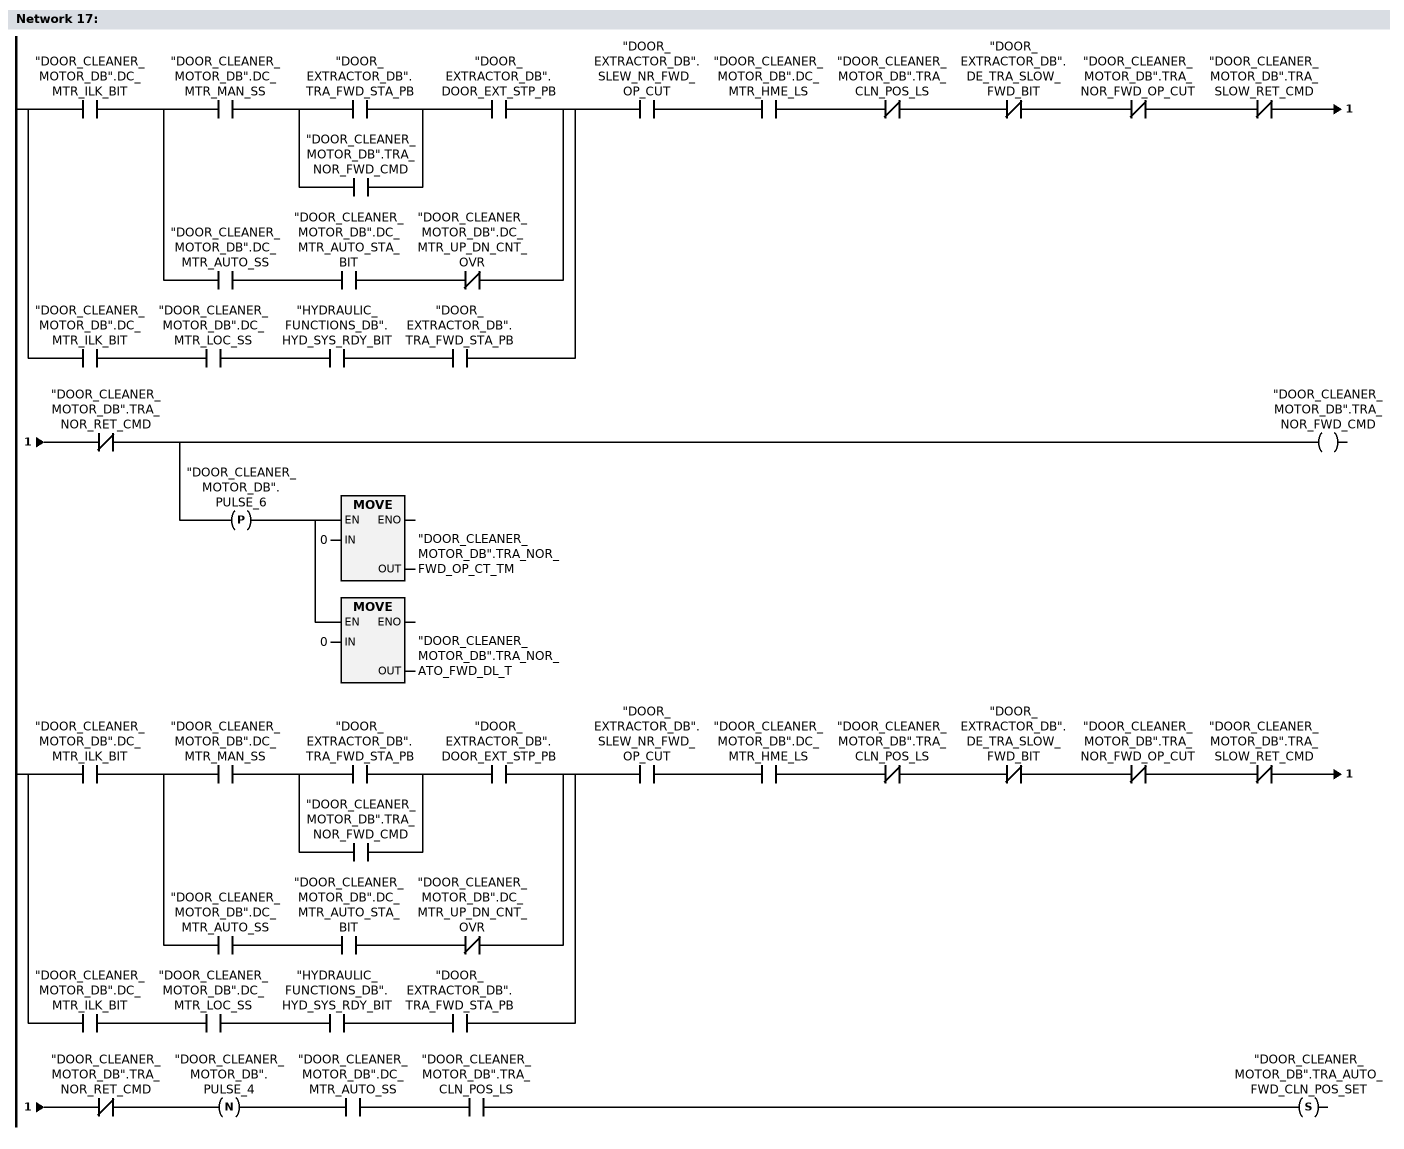
NETWORK
TITLE =
      A(;
      A     "DOOR_CLEANER_MOTOR_DB".DC_MTR_ILK_BIT;
      A(;
      A     "DOOR_CLEANER_MOTOR_DB".DC_MTR_MAN_SS;
      A(;
      O     "DOOR_EXTRACTOR_DB".TRA_FWD_STA_PB;
      O     "DOOR_CLEANER_MOTOR_DB".TRA_NOR_FWD_CMD;
      );
      A     "DOOR_EXTRACTOR_DB".DOOR_EXT_STP_PB;
      O;
      A     "DOOR_CLEANER_MOTOR_DB".DC_MTR_AUTO_SS;
      A     "DOOR_CLEANER_MOTOR_DB".DC_MTR_AUTO_STA_BIT;
      AN    "DOOR_CLEANER_MOTOR_DB".DC_MTR_UP_DN_CNT_OVR;
      );
      O;
      A     "DOOR_CLEANER_MOTOR_DB".DC_MTR_ILK_BIT;
      A     "DOOR_CLEANER_MOTOR_DB".DC_MTR_LOC_SS;
      A     "HYDRAULIC_FUNCTIONS_DB".HYD_SYS_RDY_BIT;
      A     "DOOR_EXTRACTOR_DB".TRA_FWD_STA_PB;
      );
      A     "DOOR_EXTRACTOR_DB".SLEW_NR_FWD_OP_CUT;
      A     "DOOR_CLEANER_MOTOR_DB".DC_MTR_HME_LS;
      AN    "DOOR_CLEANER_MOTOR_DB".TRA_CLN_POS_LS;
      AN    "DOOR_EXTRACTOR_DB".DE_TRA_SLOW_FWD_BIT;
      AN    "DOOR_CLEANER_MOTOR_DB".TRA_NOR_FWD_OP_CUT;
      AN    "DOOR_CLEANER_MOTOR_DB".TRA_SLOW_RET_CMD;
      AN    "DOOR_CLEANER_MOTOR_DB".TRA_NOR_RET_CMD;
      =     L 0.0;
      A     L 0.0;
      BLD   102;
      =     "DOOR_CLEANER_MOTOR_DB".TRA_NOR_FWD_CMD;
      A(;
      A     L 0.0;
      FN    "DOOR_CLEANER_MOTOR_DB".PULSE_4;
      );
      A     "DOOR_CLEANER_MOTOR_DB".DC_MTR_AUTO_SS;
      A     "DOOR_CLEANER_MOTOR_DB".TRA_CLN_POS_LS;
      S     "DOOR_CLEANER_MOTOR_DB".TRA_AUTO_FWD_CLN_POS_SET;
      A     L 0.0;
      FP    "DOOR_CLEANER_MOTOR_DB".PULSE_6;
      =     L 0.1;
      A     L 0.1;
      JNB   M012;
      L     0;
      T     "DOOR_CLEANER_MOTOR_DB".TRA_NOR_FWD_OP_CT_TM;
M012: NOP   0;
      A     L 0.1;
      JNB   M013;
      L     0;
      T     "DOOR_CLEANER_MOTOR_DB".TRA_NOR_ATO_FWD_DL_T;
M013: NOP   0;
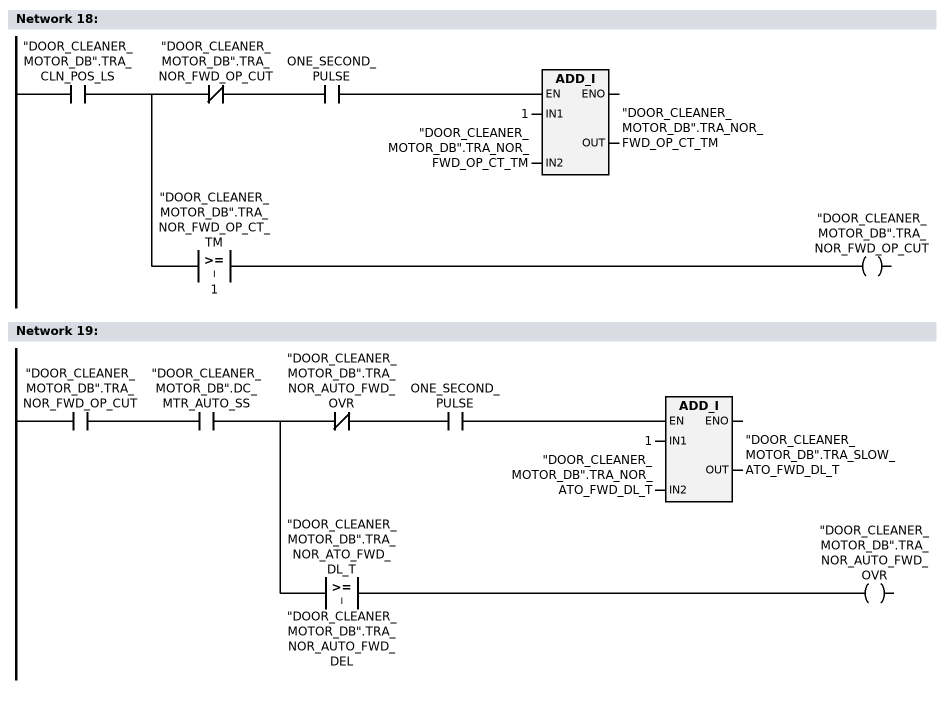
NETWORK
TITLE =
      A     "DOOR_CLEANER_MOTOR_DB".TRA_CLN_POS_LS;
      =     L 0.0;
      A     L 0.0;
      AN    "DOOR_CLEANER_MOTOR_DB".TRA_NOR_FWD_OP_CUT;
      A     "ONE_SECOND_PULSE";
      JNB   M014;
      L     1;
      L     "DOOR_CLEANER_MOTOR_DB".TRA_NOR_FWD_OP_CT_TM;
      +I;
      T     "DOOR_CLEANER_MOTOR_DB".TRA_NOR_FWD_OP_CT_TM;
M014: NOP   0;
      A     L 0.0;
      A(;
      L     "DOOR_CLEANER_MOTOR_DB".TRA_NOR_FWD_OP_CT_TM;
      L     1;
      >=I;
      );
      =     "DOOR_CLEANER_MOTOR_DB".TRA_NOR_FWD_OP_CUT;
NETWORK
TITLE =
      A     "DOOR_CLEANER_MOTOR_DB".TRA_NOR_FWD_OP_CUT;
      A     "DOOR_CLEANER_MOTOR_DB".DC_MTR_AUTO_SS;
      =     L 0.0;
      A     L 0.0;
      AN    "DOOR_CLEANER_MOTOR_DB".TRA_NOR_AUTO_FWD_OVR;
      A     "ONE_SECOND_PULSE";
      JNB   M015;
      L     1;
      L     "DOOR_CLEANER_MOTOR_DB".TRA_NOR_ATO_FWD_DL_T;
      +I;
      T     "DOOR_CLEANER_MOTOR_DB".TRA_SLOW_ATO_FWD_DL_T;
M015: NOP   0;
      A     L 0.0;
      A(;
      L     "DOOR_CLEANER_MOTOR_DB".TRA_NOR_ATO_FWD_DL_T;
      L     "DOOR_CLEANER_MOTOR_DB".TRA_NOR_AUTO_FWD_DEL;
      >=I;
      );
      =     "DOOR_CLEANER_MOTOR_DB".TRA_NOR_AUTO_FWD_OVR;
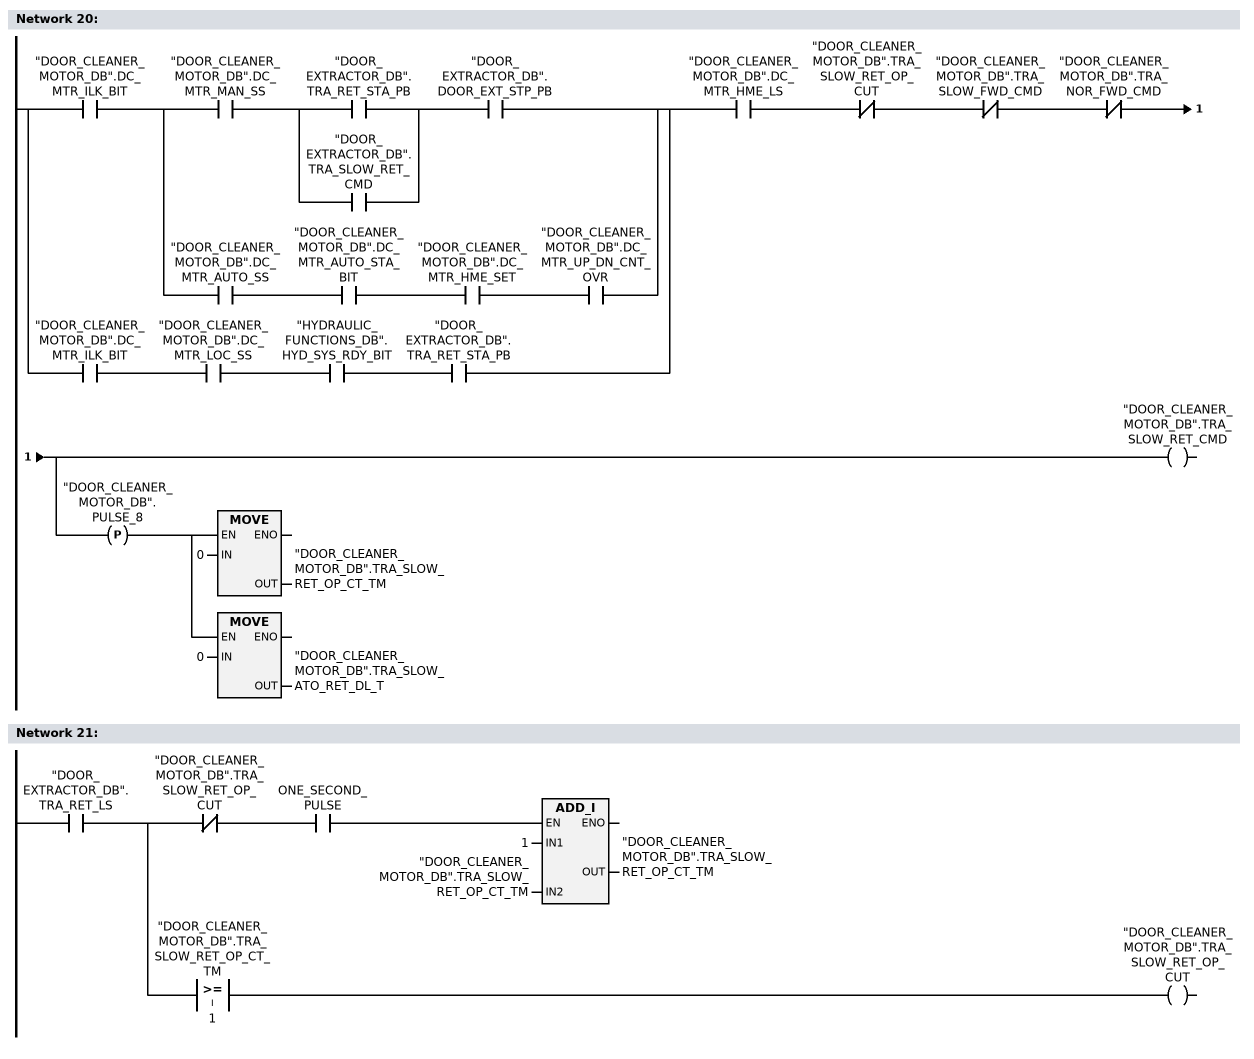
NETWORK
TITLE =
      A(;
      A     "DOOR_CLEANER_MOTOR_DB".DC_MTR_ILK_BIT;
      A(;
      A     "DOOR_CLEANER_MOTOR_DB".DC_MTR_MAN_SS;
      A(;
      O     "DOOR_EXTRACTOR_DB".TRA_RET_STA_PB;
      O     "DOOR_EXTRACTOR_DB".TRA_SLOW_RET_CMD;
      );
      A     "DOOR_EXTRACTOR_DB".DOOR_EXT_STP_PB;
      O;
      A     "DOOR_CLEANER_MOTOR_DB".DC_MTR_AUTO_SS;
      A     "DOOR_CLEANER_MOTOR_DB".DC_MTR_AUTO_STA_BIT;
      A     "DOOR_CLEANER_MOTOR_DB".DC_MTR_HME_SET;
      A     "DOOR_CLEANER_MOTOR_DB".DC_MTR_UP_DN_CNT_OVR;
      );
      O;
      A     "DOOR_CLEANER_MOTOR_DB".DC_MTR_ILK_BIT;
      A     "DOOR_CLEANER_MOTOR_DB".DC_MTR_LOC_SS;
      A     "HYDRAULIC_FUNCTIONS_DB".HYD_SYS_RDY_BIT;
      A     "DOOR_EXTRACTOR_DB".TRA_RET_STA_PB;
      );
      A     "DOOR_CLEANER_MOTOR_DB".DC_MTR_HME_LS;
      AN    "DOOR_CLEANER_MOTOR_DB".TRA_SLOW_RET_OP_CUT;
      AN    "DOOR_CLEANER_MOTOR_DB".TRA_SLOW_FWD_CMD;
      AN    "DOOR_CLEANER_MOTOR_DB".TRA_NOR_FWD_CMD;
      =     L 0.0;
      A     L 0.0;
      BLD   102;
      =     "DOOR_CLEANER_MOTOR_DB".TRA_SLOW_RET_CMD;
      A     L 0.0;
      FP    "DOOR_CLEANER_MOTOR_DB".PULSE_8;
      =     L 0.1;
      A     L 0.1;
      JNB   M016;
      L     0;
      T     "DOOR_CLEANER_MOTOR_DB".TRA_SLOW_RET_OP_CT_TM;
M016: NOP   0;
      A     L 0.1;
      JNB   M017;
      L     0;
      T     "DOOR_CLEANER_MOTOR_DB".TRA_SLOW_ATO_RET_DL_T;
M017: NOP   0;
NETWORK
TITLE =
      A     "DOOR_EXTRACTOR_DB".TRA_RET_LS;
      =     L 0.0;
      A     L 0.0;
      AN    "DOOR_CLEANER_MOTOR_DB".TRA_SLOW_RET_OP_CUT;
      A     "ONE_SECOND_PULSE";
      JNB   M018;
      L     1;
      L     "DOOR_CLEANER_MOTOR_DB".TRA_SLOW_RET_OP_CT_TM;
      +I;
      T     "DOOR_CLEANER_MOTOR_DB".TRA_SLOW_RET_OP_CT_TM;
M018: NOP   0;
      A     L 0.0;
      A(;
      L     "DOOR_CLEANER_MOTOR_DB".TRA_SLOW_RET_OP_CT_TM;
      L     1;
      >=I;
      );
      =     "DOOR_CLEANER_MOTOR_DB".TRA_SLOW_RET_OP_CUT;
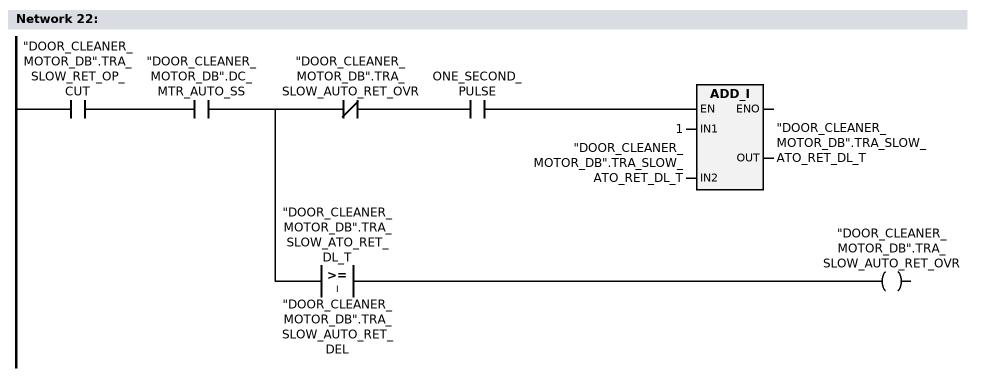
NETWORK
TITLE =
      A     "DOOR_CLEANER_MOTOR_DB".TRA_SLOW_RET_OP_CUT;
      A     "DOOR_CLEANER_MOTOR_DB".DC_MTR_AUTO_SS;
      =     L 0.0;
      A     L 0.0;
      AN    "DOOR_CLEANER_MOTOR_DB".TRA_SLOW_AUTO_RET_OVR;
      A     "ONE_SECOND_PULSE";
      JNB   M019;
      L     1;
      L     "DOOR_CLEANER_MOTOR_DB".TRA_SLOW_ATO_RET_DL_T;
      +I;
      T     "DOOR_CLEANER_MOTOR_DB".TRA_SLOW_ATO_RET_DL_T;
M019: NOP   0;
      A     L 0.0;
      A(;
      L     "DOOR_CLEANER_MOTOR_DB".TRA_SLOW_ATO_RET_DL_T;
      L     "DOOR_CLEANER_MOTOR_DB".TRA_SLOW_AUTO_RET_DEL;
      >=I;
      );
      =     "DOOR_CLEANER_MOTOR_DB".TRA_SLOW_AUTO_RET_OVR;
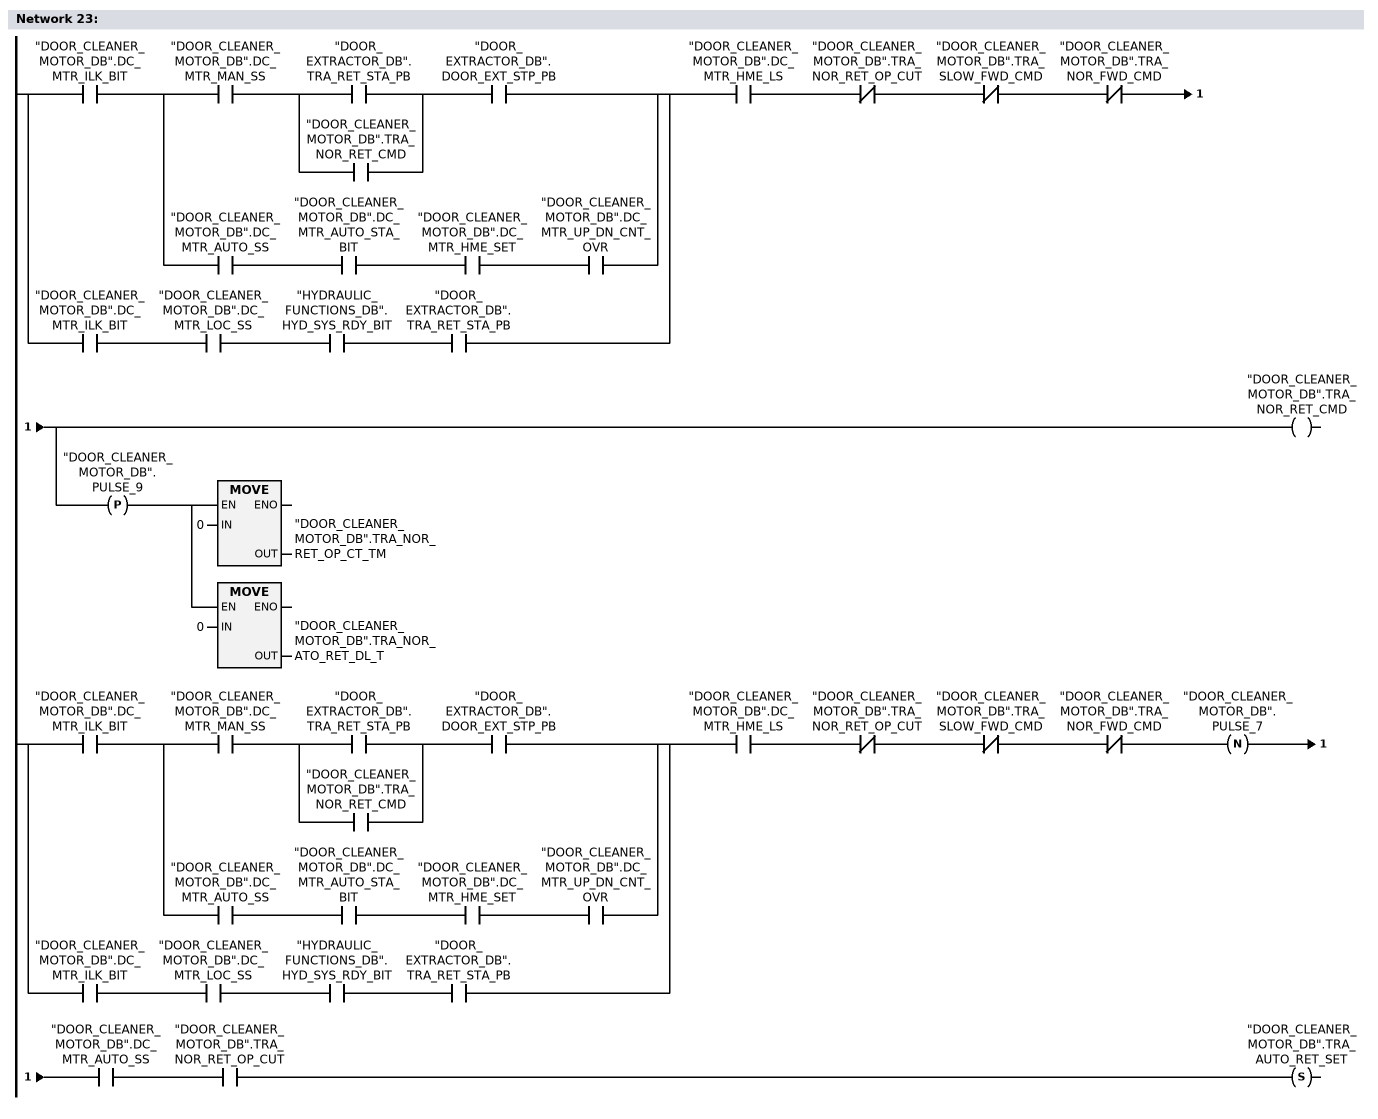
NETWORK
TITLE =
      A(;
      A     "DOOR_CLEANER_MOTOR_DB".DC_MTR_ILK_BIT;
      A(;
      A     "DOOR_CLEANER_MOTOR_DB".DC_MTR_MAN_SS;
      A(;
      O     "DOOR_EXTRACTOR_DB".TRA_RET_STA_PB;
      O     "DOOR_CLEANER_MOTOR_DB".TRA_NOR_RET_CMD;
      );
      A     "DOOR_EXTRACTOR_DB".DOOR_EXT_STP_PB;
      O;
      A     "DOOR_CLEANER_MOTOR_DB".DC_MTR_AUTO_SS;
      A     "DOOR_CLEANER_MOTOR_DB".DC_MTR_AUTO_STA_BIT;
      A     "DOOR_CLEANER_MOTOR_DB".DC_MTR_HME_SET;
      A     "DOOR_CLEANER_MOTOR_DB".DC_MTR_UP_DN_CNT_OVR;
      );
      O;
      A     "DOOR_CLEANER_MOTOR_DB".DC_MTR_ILK_BIT;
      A     "DOOR_CLEANER_MOTOR_DB".DC_MTR_LOC_SS;
      A     "HYDRAULIC_FUNCTIONS_DB".HYD_SYS_RDY_BIT;
      A     "DOOR_EXTRACTOR_DB".TRA_RET_STA_PB;
      );
      A     "DOOR_CLEANER_MOTOR_DB".DC_MTR_HME_LS;
      AN    "DOOR_CLEANER_MOTOR_DB".TRA_NOR_RET_OP_CUT;
      AN    "DOOR_CLEANER_MOTOR_DB".TRA_SLOW_FWD_CMD;
      AN    "DOOR_CLEANER_MOTOR_DB".TRA_NOR_FWD_CMD;
      =     L 0.0;
      A     L 0.0;
      BLD   102;
      =     "DOOR_CLEANER_MOTOR_DB".TRA_NOR_RET_CMD;
      A(;
      A     L 0.0;
      FN    "DOOR_CLEANER_MOTOR_DB".PULSE_7;
      );
      A     "DOOR_CLEANER_MOTOR_DB".DC_MTR_AUTO_SS;
      A     "DOOR_CLEANER_MOTOR_DB".TRA_NOR_RET_OP_CUT;
      S     "DOOR_CLEANER_MOTOR_DB".TRA_AUTO_RET_SET;
      A     L 0.0;
      FP    "DOOR_CLEANER_MOTOR_DB".PULSE_9;
      =     L 0.1;
      A     L 0.1;
      JNB   M020;
      L     0;
      T     "DOOR_CLEANER_MOTOR_DB".TRA_NOR_RET_OP_CT_TM;
M020: NOP   0;
      A     L 0.1;
      JNB   M021;
      L     0;
      T     "DOOR_CLEANER_MOTOR_DB".TRA_NOR_ATO_RET_DL_T;
M021: NOP   0;
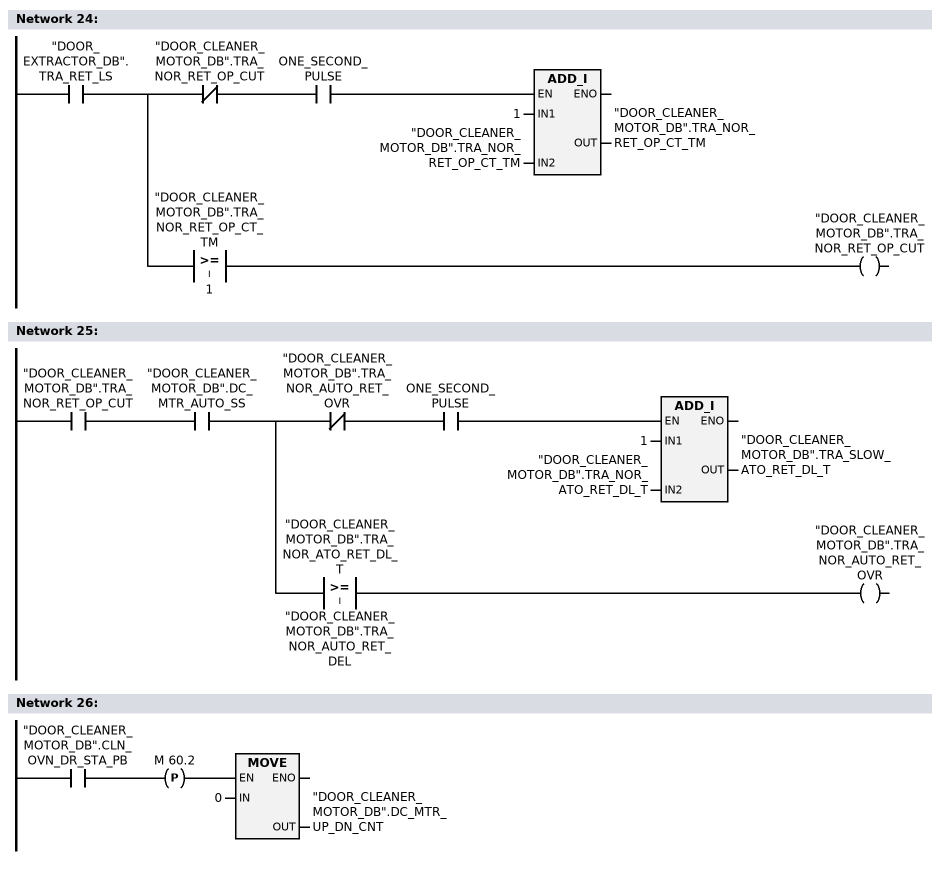
NETWORK
TITLE =
      A     "DOOR_EXTRACTOR_DB".TRA_RET_LS;
      =     L 0.0;
      A     L 0.0;
      AN    "DOOR_CLEANER_MOTOR_DB".TRA_NOR_RET_OP_CUT;
      A     "ONE_SECOND_PULSE";
      JNB   M022;
      L     1;
      L     "DOOR_CLEANER_MOTOR_DB".TRA_NOR_RET_OP_CT_TM;
      +I;
      T     "DOOR_CLEANER_MOTOR_DB".TRA_NOR_RET_OP_CT_TM;
M022: NOP   0;
      A     L 0.0;
      A(;
      L     "DOOR_CLEANER_MOTOR_DB".TRA_NOR_RET_OP_CT_TM;
      L     1;
      >=I;
      );
      =     "DOOR_CLEANER_MOTOR_DB".TRA_NOR_RET_OP_CUT;
NETWORK
TITLE =
      A     "DOOR_CLEANER_MOTOR_DB".TRA_NOR_RET_OP_CUT;
      A     "DOOR_CLEANER_MOTOR_DB".DC_MTR_AUTO_SS;
      =     L 0.0;
      A     L 0.0;
      AN    "DOOR_CLEANER_MOTOR_DB".TRA_NOR_AUTO_RET_OVR;
      A     "ONE_SECOND_PULSE";
      JNB   M023;
      L     1;
      L     "DOOR_CLEANER_MOTOR_DB".TRA_NOR_ATO_RET_DL_T;
      +I;
      T     "DOOR_CLEANER_MOTOR_DB".TRA_SLOW_ATO_RET_DL_T;
M023: NOP   0;
      A     L 0.0;
      A(;
      L     "DOOR_CLEANER_MOTOR_DB".TRA_NOR_ATO_RET_DL_T;
      L     "DOOR_CLEANER_MOTOR_DB".TRA_NOR_AUTO_RET_DEL;
      >=I;
      );
      =     "DOOR_CLEANER_MOTOR_DB".TRA_NOR_AUTO_RET_OVR;
NETWORK
TITLE =
      A     "DOOR_CLEANER_MOTOR_DB".CLN_OVN_DR_STA_PB;
      FP    M 60.2;
      JNB   M024;
      L     0;
      T     "DOOR_CLEANER_MOTOR_DB".DC_MTR_UP_DN_CNT;
M024: NOP   0;
END_FUNCTION

FUNCTION "PROFIBUS_COMMUNICATION" : VOID	// FC 13
AUTHOR : Kamillas
VERSION : 0.1
BEGIN
// (block stored without names or comments; labels and parameter names are numbered)
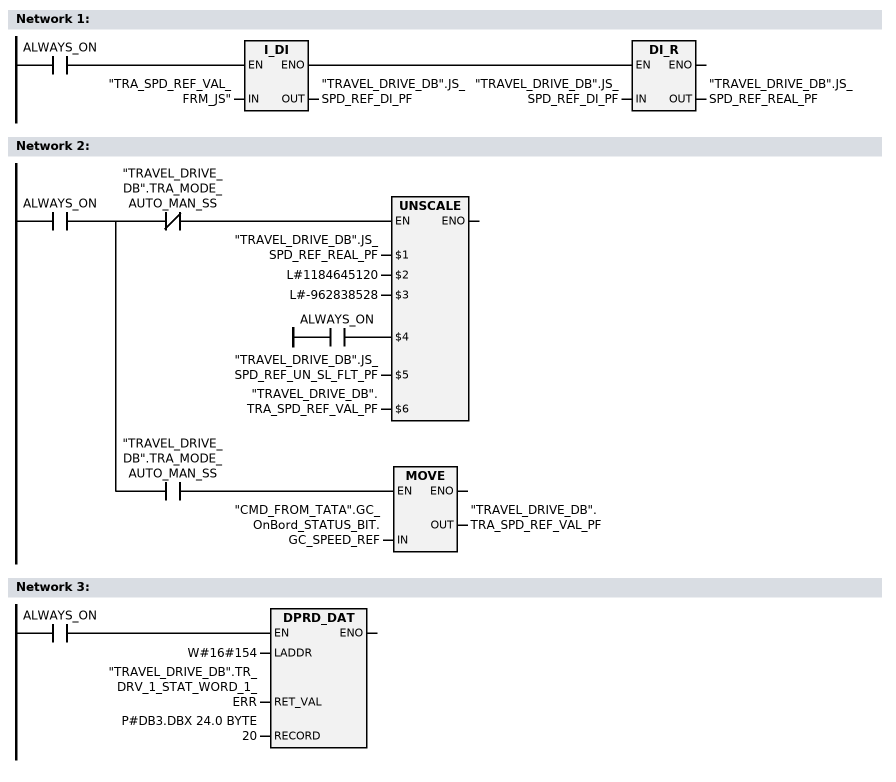
NETWORK
TITLE =
      A(;
      A     "ALWAYS_ON";
      JNB   M001;
      L     "TRA_SPD_REF_VAL_FRM_JS";
      ITD;
      T     "TRAVEL_DRIVE_DB".JS_SPD_REF_DI_PF;
      SET;
      SAVE;
      CLR;
M001: A     BR;
      );
      JNB   M002;
      L     "TRAVEL_DRIVE_DB".JS_SPD_REF_DI_PF;
      DTR;
      T     "TRAVEL_DRIVE_DB".JS_SPD_REF_REAL_PF;
M002: NOP   0;
NETWORK
TITLE =
      A     "ALWAYS_ON";
      =     L 0.0;
      A     "ALWAYS_ON";
      =     L 0.1;
      BLD   103;
      A     L 0.0;
      AN    "TRAVEL_DRIVE_DB".TRA_MODE_AUTO_MAN_SS;
      JNB   M003;
      CALL  "UNSCALE" (
           $1                       := "TRAVEL_DRIVE_DB".JS_SPD_REF_REAL_PF,
           $2                       := L#1184645120,
           $3                       := L#-962838528,
           $4                       := L 0.1,
           $5                       := "TRAVEL_DRIVE_DB".JS_SPD_REF_UN_SL_FLT_PF,
           $6                       := "TRAVEL_DRIVE_DB".TRA_SPD_REF_VAL_PF);
M003: NOP   0;
      A     L 0.0;
      A     "TRAVEL_DRIVE_DB".TRA_MODE_AUTO_MAN_SS;
      JNB   M004;
      L     "CMD_FROM_TATA".GC_OnBord_STATUS_BIT.GC_SPEED_REF;
      T     "TRAVEL_DRIVE_DB".TRA_SPD_REF_VAL_PF;
M004: NOP   0;
NETWORK
TITLE =
      A     "ALWAYS_ON";
      JNB   M005;
      CALL  "DPRD_DAT" (
           LADDR                    := W#16#154,
           RET_VAL                  := "TRAVEL_DRIVE_DB".TR_DRV_1_STAT_WORD_1_ERR,
           RECORD                   := P#DB3.DBX 24.0 BYTE 20);
M005: NOP   0;
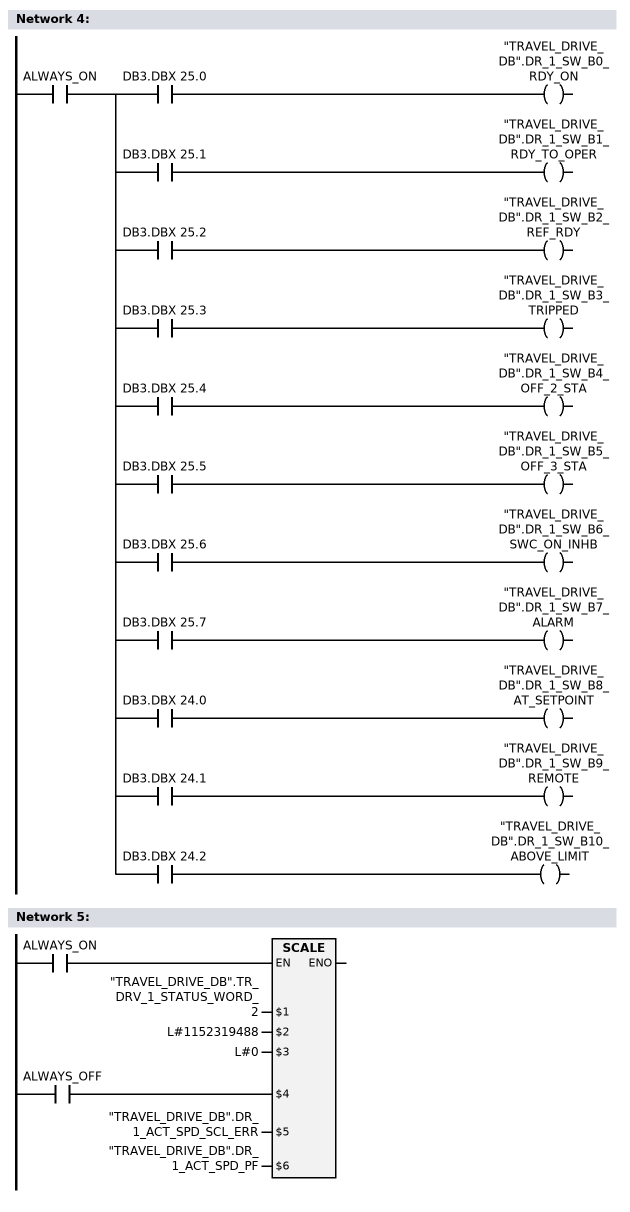
NETWORK
TITLE =
      A     "ALWAYS_ON";
      =     L 0.0;
      A     L 0.0;
      A     DB3.DBX 25.0;
      =     "TRAVEL_DRIVE_DB".DR_1_SW_B0_RDY_ON;
      A     L 0.0;
      A     DB3.DBX 25.1;
      =     "TRAVEL_DRIVE_DB".DR_1_SW_B1_RDY_TO_OPER;
      A     L 0.0;
      A     DB3.DBX 25.2;
      =     "TRAVEL_DRIVE_DB".DR_1_SW_B2_REF_RDY;
      A     L 0.0;
      A     DB3.DBX 25.3;
      =     "TRAVEL_DRIVE_DB".DR_1_SW_B3_TRIPPED;
      A     L 0.0;
      A     DB3.DBX 25.4;
      =     "TRAVEL_DRIVE_DB".DR_1_SW_B4_OFF_2_STA;
      A     L 0.0;
      A     DB3.DBX 25.5;
      =     "TRAVEL_DRIVE_DB".DR_1_SW_B5_OFF_3_STA;
      A     L 0.0;
      A     DB3.DBX 25.6;
      =     "TRAVEL_DRIVE_DB".DR_1_SW_B6_SWC_ON_INHB;
      A     L 0.0;
      A     DB3.DBX 25.7;
      =     "TRAVEL_DRIVE_DB".DR_1_SW_B7_ALARM;
      A     L 0.0;
      A     DB3.DBX 24.0;
      =     "TRAVEL_DRIVE_DB".DR_1_SW_B8_AT_SETPOINT;
      A     L 0.0;
      A     DB3.DBX 24.1;
      =     "TRAVEL_DRIVE_DB".DR_1_SW_B9_REMOTE;
      A     L 0.0;
      A     DB3.DBX 24.2;
      =     "TRAVEL_DRIVE_DB".DR_1_SW_B10_ABOVE_LIMIT;
NETWORK
TITLE =
      A     "ALWAYS_OFF";
      =     L 0.0;
      BLD   103;
      A     "ALWAYS_ON";
      JNB   M006;
      CALL  "SCALE" (
           $1                       := "TRAVEL_DRIVE_DB".TR_DRV_1_STATUS_WORD_2,
           $2                       := L#1152319488,
           $3                       := L#0,
           $4                       := L 0.0,
           $5                       := "TRAVEL_DRIVE_DB".DR_1_ACT_SPD_SCL_ERR,
           $6                       := "TRAVEL_DRIVE_DB".DR_1_ACT_SPD_PF);
M006: NOP   0;
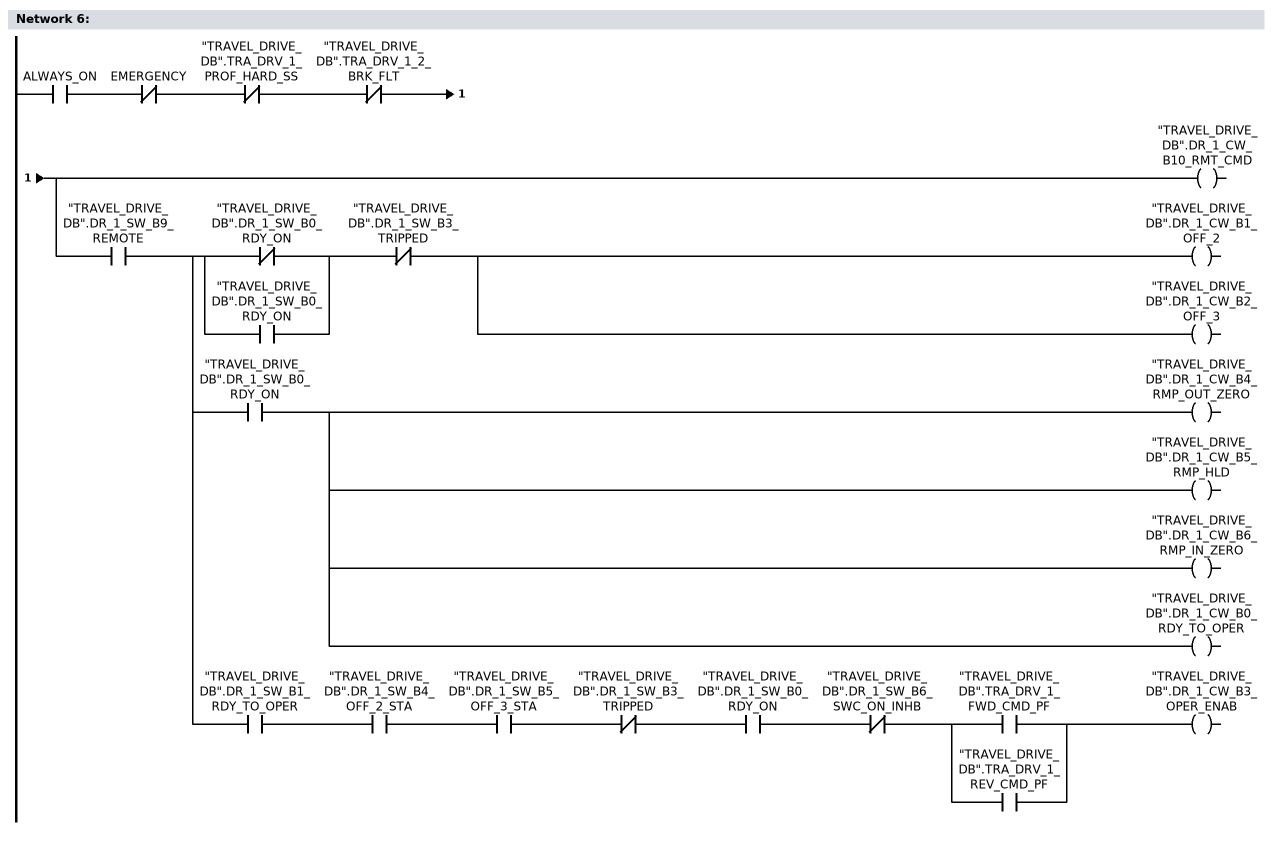
NETWORK
TITLE =
      A     "ALWAYS_ON";
      AN    "EMERGENCY";
      AN    "TRAVEL_DRIVE_DB".TRA_DRV_1_PROF_HARD_SS;
      AN    "TRAVEL_DRIVE_DB".TRA_DRV_1_2_BRK_FLT;
      =     L 0.0;
      A     L 0.0;
      BLD   102;
      =     "TRAVEL_DRIVE_DB".DR_1_CW_B10_RMT_CMD;
      A     L 0.0;
      A     "TRAVEL_DRIVE_DB".DR_1_SW_B9_REMOTE;
      =     L 0.1;
      A     L 0.1;
      A(;
      ON    "TRAVEL_DRIVE_DB".DR_1_SW_B0_RDY_ON;
      O     "TRAVEL_DRIVE_DB".DR_1_SW_B0_RDY_ON;
      );
      AN    "TRAVEL_DRIVE_DB".DR_1_SW_B3_TRIPPED;
      =     "TRAVEL_DRIVE_DB".DR_1_CW_B1_OFF_2;
      =     "TRAVEL_DRIVE_DB".DR_1_CW_B2_OFF_3;
      A     L 0.1;
      A     "TRAVEL_DRIVE_DB".DR_1_SW_B0_RDY_ON;
      =     "TRAVEL_DRIVE_DB".DR_1_CW_B4_RMP_OUT_ZERO;
      =     "TRAVEL_DRIVE_DB".DR_1_CW_B5_RMP_HLD;
      =     "TRAVEL_DRIVE_DB".DR_1_CW_B6_RMP_IN_ZERO;
      =     "TRAVEL_DRIVE_DB".DR_1_CW_B0_RDY_TO_OPER;
      A     L 0.1;
      A     "TRAVEL_DRIVE_DB".DR_1_SW_B1_RDY_TO_OPER;
      A     "TRAVEL_DRIVE_DB".DR_1_SW_B4_OFF_2_STA;
      A     "TRAVEL_DRIVE_DB".DR_1_SW_B5_OFF_3_STA;
      AN    "TRAVEL_DRIVE_DB".DR_1_SW_B3_TRIPPED;
      A     "TRAVEL_DRIVE_DB".DR_1_SW_B0_RDY_ON;
      AN    "TRAVEL_DRIVE_DB".DR_1_SW_B6_SWC_ON_INHB;
      A(;
      O     "TRAVEL_DRIVE_DB".TRA_DRV_1_FWD_CMD_PF;
      O     "TRAVEL_DRIVE_DB".TRA_DRV_1_REV_CMD_PF;
      );
      =     "TRAVEL_DRIVE_DB".DR_1_CW_B3_OPER_ENAB;
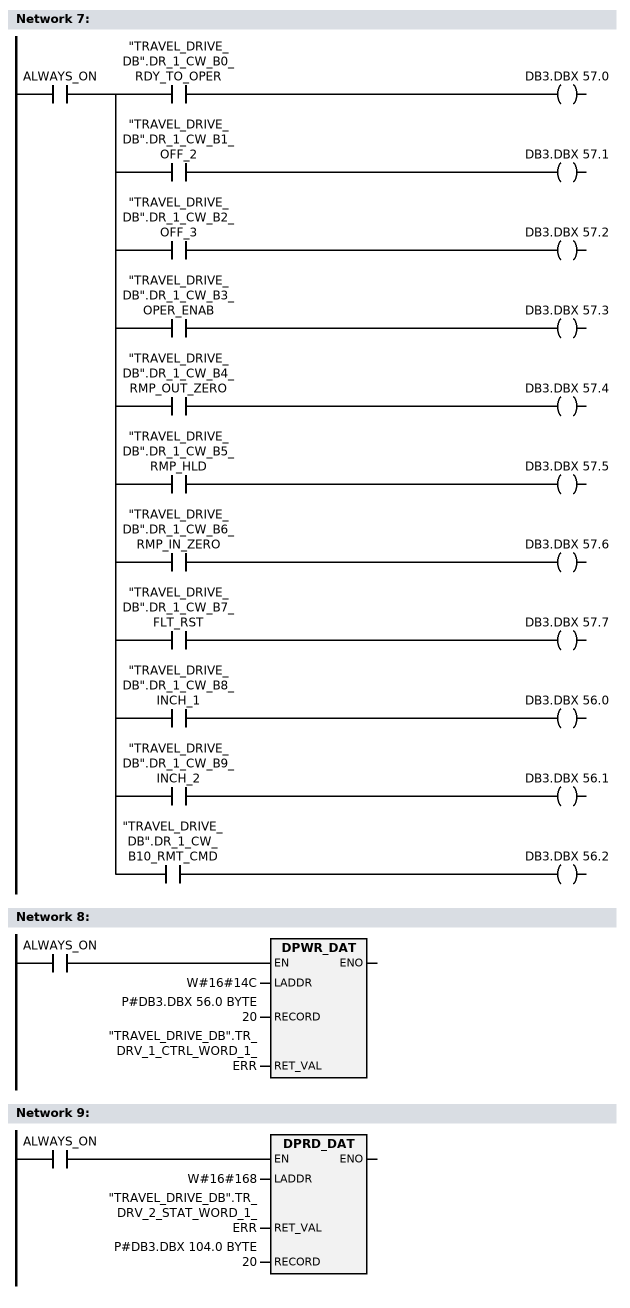
NETWORK
TITLE =
      A     "ALWAYS_ON";
      =     L 0.0;
      A     L 0.0;
      A     "TRAVEL_DRIVE_DB".DR_1_CW_B0_RDY_TO_OPER;
      =     DB3.DBX 57.0;
      A     L 0.0;
      A     "TRAVEL_DRIVE_DB".DR_1_CW_B1_OFF_2;
      =     DB3.DBX 57.1;
      A     L 0.0;
      A     "TRAVEL_DRIVE_DB".DR_1_CW_B2_OFF_3;
      =     DB3.DBX 57.2;
      A     L 0.0;
      A     "TRAVEL_DRIVE_DB".DR_1_CW_B3_OPER_ENAB;
      =     DB3.DBX 57.3;
      A     L 0.0;
      A     "TRAVEL_DRIVE_DB".DR_1_CW_B4_RMP_OUT_ZERO;
      =     DB3.DBX 57.4;
      A     L 0.0;
      A     "TRAVEL_DRIVE_DB".DR_1_CW_B5_RMP_HLD;
      =     DB3.DBX 57.5;
      A     L 0.0;
      A     "TRAVEL_DRIVE_DB".DR_1_CW_B6_RMP_IN_ZERO;
      =     DB3.DBX 57.6;
      A     L 0.0;
      A     "TRAVEL_DRIVE_DB".DR_1_CW_B7_FLT_RST;
      =     DB3.DBX 57.7;
      A     L 0.0;
      A     "TRAVEL_DRIVE_DB".DR_1_CW_B8_INCH_1;
      =     DB3.DBX 56.0;
      A     L 0.0;
      A     "TRAVEL_DRIVE_DB".DR_1_CW_B9_INCH_2;
      =     DB3.DBX 56.1;
      A     L 0.0;
      A     "TRAVEL_DRIVE_DB".DR_1_CW_B10_RMT_CMD;
      =     DB3.DBX 56.2;
NETWORK
TITLE =
      A     "ALWAYS_ON";
      JNB   M007;
      CALL  "DPWR_DAT" (
           LADDR                    := W#16#14C,
           RECORD                   := P#DB3.DBX 56.0 BYTE 20,
           RET_VAL                  := "TRAVEL_DRIVE_DB".TR_DRV_1_CTRL_WORD_1_ERR);
M007: NOP   0;
NETWORK
TITLE =
      A     "ALWAYS_ON";
      JNB   M008;
      CALL  "DPRD_DAT" (
           LADDR                    := W#16#168,
           RET_VAL                  := "TRAVEL_DRIVE_DB".TR_DRV_2_STAT_WORD_1_ERR,
           RECORD                   := P#DB3.DBX 104.0 BYTE 20);
M008: NOP   0;
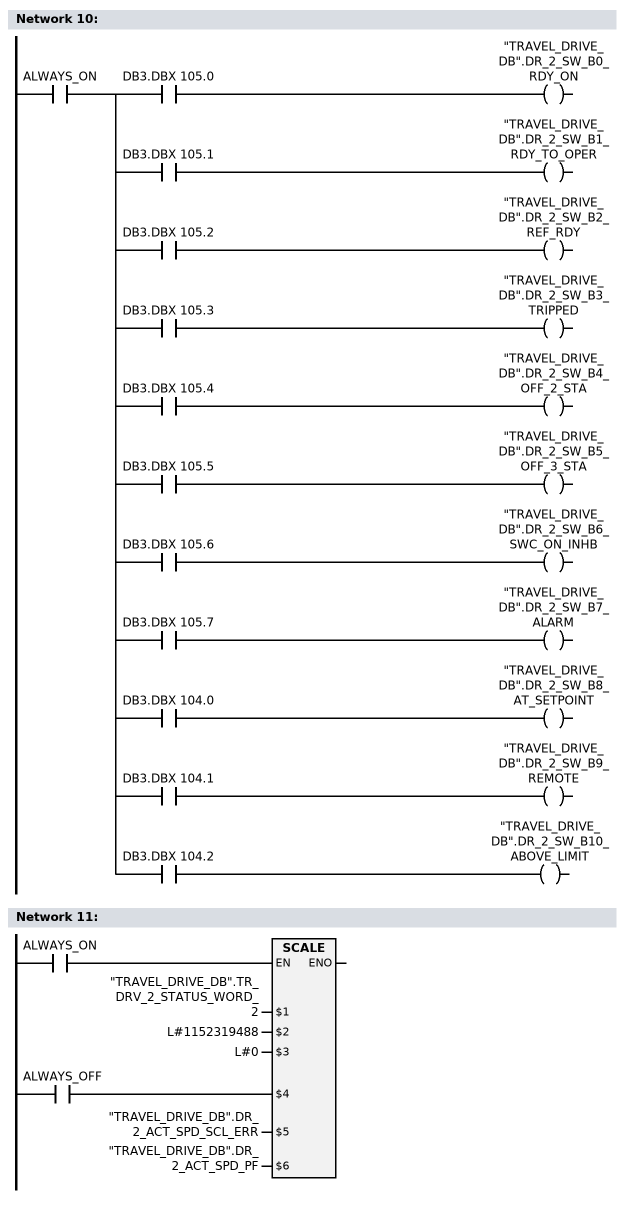
NETWORK
TITLE =
      A     "ALWAYS_ON";
      =     L 0.0;
      A     L 0.0;
      A     DB3.DBX 105.0;
      =     "TRAVEL_DRIVE_DB".DR_2_SW_B0_RDY_ON;
      A     L 0.0;
      A     DB3.DBX 105.1;
      =     "TRAVEL_DRIVE_DB".DR_2_SW_B1_RDY_TO_OPER;
      A     L 0.0;
      A     DB3.DBX 105.2;
      =     "TRAVEL_DRIVE_DB".DR_2_SW_B2_REF_RDY;
      A     L 0.0;
      A     DB3.DBX 105.3;
      =     "TRAVEL_DRIVE_DB".DR_2_SW_B3_TRIPPED;
      A     L 0.0;
      A     DB3.DBX 105.4;
      =     "TRAVEL_DRIVE_DB".DR_2_SW_B4_OFF_2_STA;
      A     L 0.0;
      A     DB3.DBX 105.5;
      =     "TRAVEL_DRIVE_DB".DR_2_SW_B5_OFF_3_STA;
      A     L 0.0;
      A     DB3.DBX 105.6;
      =     "TRAVEL_DRIVE_DB".DR_2_SW_B6_SWC_ON_INHB;
      A     L 0.0;
      A     DB3.DBX 105.7;
      =     "TRAVEL_DRIVE_DB".DR_2_SW_B7_ALARM;
      A     L 0.0;
      A     DB3.DBX 104.0;
      =     "TRAVEL_DRIVE_DB".DR_2_SW_B8_AT_SETPOINT;
      A     L 0.0;
      A     DB3.DBX 104.1;
      =     "TRAVEL_DRIVE_DB".DR_2_SW_B9_REMOTE;
      A     L 0.0;
      A     DB3.DBX 104.2;
      =     "TRAVEL_DRIVE_DB".DR_2_SW_B10_ABOVE_LIMIT;
NETWORK
TITLE =
      A     "ALWAYS_OFF";
      =     L 0.0;
      BLD   103;
      A     "ALWAYS_ON";
      JNB   M009;
      CALL  "SCALE" (
           $1                       := "TRAVEL_DRIVE_DB".TR_DRV_2_STATUS_WORD_2,
           $2                       := L#1152319488,
           $3                       := L#0,
           $4                       := L 0.0,
           $5                       := "TRAVEL_DRIVE_DB".DR_2_ACT_SPD_SCL_ERR,
           $6                       := "TRAVEL_DRIVE_DB".DR_2_ACT_SPD_PF);
M009: NOP   0;
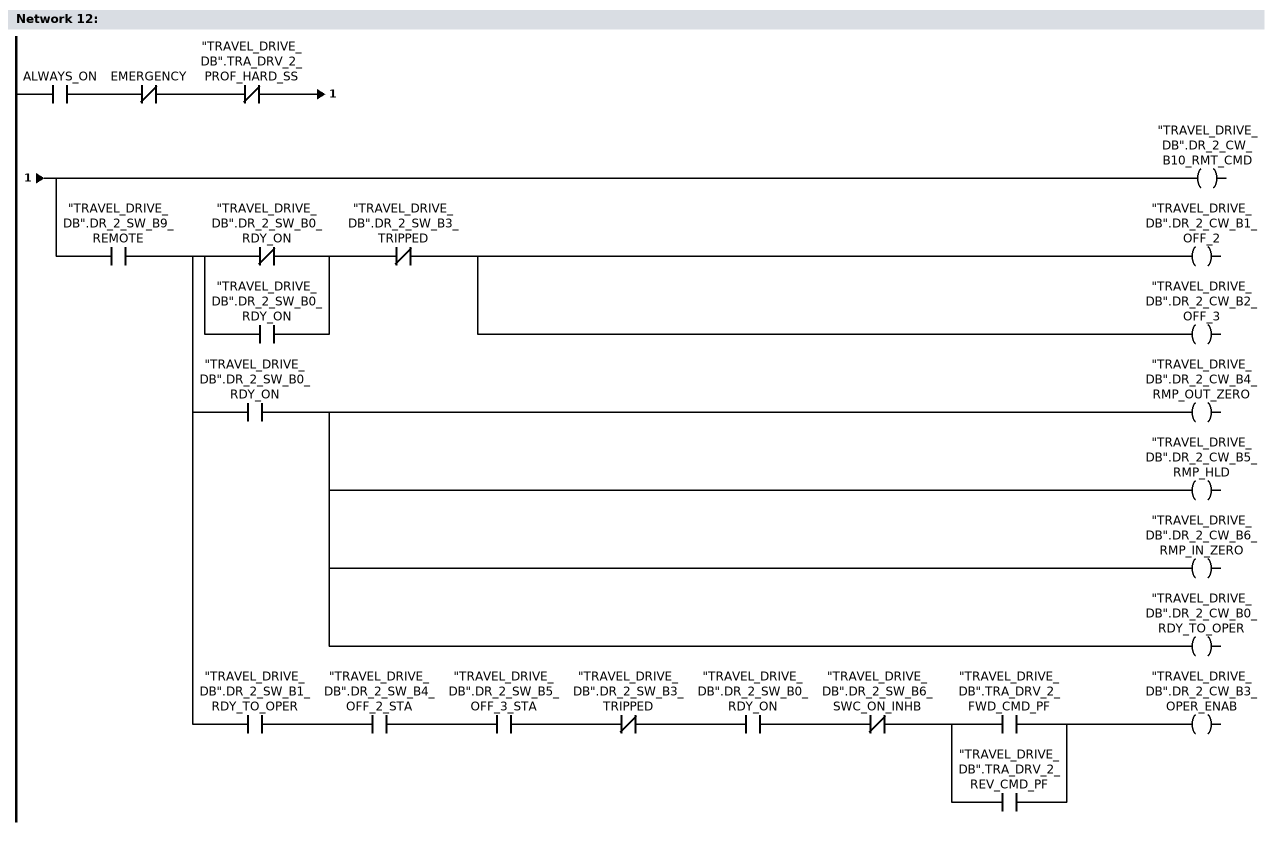
NETWORK
TITLE =
      A     "ALWAYS_ON";
      AN    "EMERGENCY";
      AN    "TRAVEL_DRIVE_DB".TRA_DRV_2_PROF_HARD_SS;
      =     L 0.0;
      A     L 0.0;
      BLD   102;
      =     "TRAVEL_DRIVE_DB".DR_2_CW_B10_RMT_CMD;
      A     L 0.0;
      A     "TRAVEL_DRIVE_DB".DR_2_SW_B9_REMOTE;
      =     L 0.1;
      A     L 0.1;
      A(;
      ON    "TRAVEL_DRIVE_DB".DR_2_SW_B0_RDY_ON;
      O     "TRAVEL_DRIVE_DB".DR_2_SW_B0_RDY_ON;
      );
      AN    "TRAVEL_DRIVE_DB".DR_2_SW_B3_TRIPPED;
      =     "TRAVEL_DRIVE_DB".DR_2_CW_B1_OFF_2;
      =     "TRAVEL_DRIVE_DB".DR_2_CW_B2_OFF_3;
      A     L 0.1;
      A     "TRAVEL_DRIVE_DB".DR_2_SW_B0_RDY_ON;
      =     "TRAVEL_DRIVE_DB".DR_2_CW_B4_RMP_OUT_ZERO;
      =     "TRAVEL_DRIVE_DB".DR_2_CW_B5_RMP_HLD;
      =     "TRAVEL_DRIVE_DB".DR_2_CW_B6_RMP_IN_ZERO;
      =     "TRAVEL_DRIVE_DB".DR_2_CW_B0_RDY_TO_OPER;
      A     L 0.1;
      A     "TRAVEL_DRIVE_DB".DR_2_SW_B1_RDY_TO_OPER;
      A     "TRAVEL_DRIVE_DB".DR_2_SW_B4_OFF_2_STA;
      A     "TRAVEL_DRIVE_DB".DR_2_SW_B5_OFF_3_STA;
      AN    "TRAVEL_DRIVE_DB".DR_2_SW_B3_TRIPPED;
      A     "TRAVEL_DRIVE_DB".DR_2_SW_B0_RDY_ON;
      AN    "TRAVEL_DRIVE_DB".DR_2_SW_B6_SWC_ON_INHB;
      A(;
      O     "TRAVEL_DRIVE_DB".TRA_DRV_2_FWD_CMD_PF;
      O     "TRAVEL_DRIVE_DB".TRA_DRV_2_REV_CMD_PF;
      );
      =     "TRAVEL_DRIVE_DB".DR_2_CW_B3_OPER_ENAB;
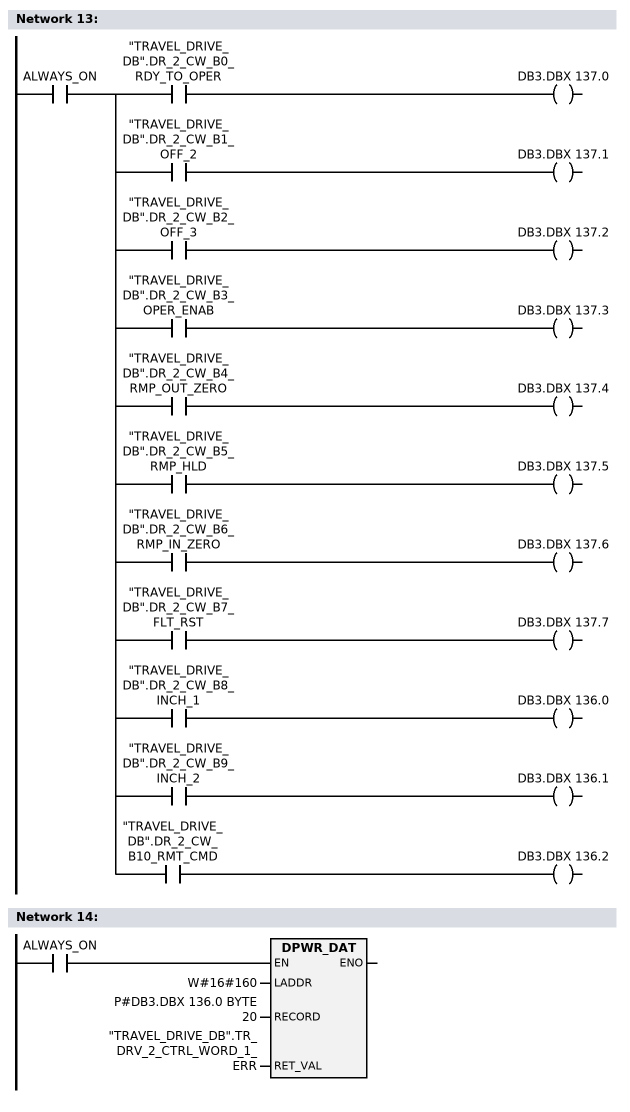
NETWORK
TITLE =
      A     "ALWAYS_ON";
      =     L 0.0;
      A     L 0.0;
      A     "TRAVEL_DRIVE_DB".DR_2_CW_B0_RDY_TO_OPER;
      =     DB3.DBX 137.0;
      A     L 0.0;
      A     "TRAVEL_DRIVE_DB".DR_2_CW_B1_OFF_2;
      =     DB3.DBX 137.1;
      A     L 0.0;
      A     "TRAVEL_DRIVE_DB".DR_2_CW_B2_OFF_3;
      =     DB3.DBX 137.2;
      A     L 0.0;
      A     "TRAVEL_DRIVE_DB".DR_2_CW_B3_OPER_ENAB;
      =     DB3.DBX 137.3;
      A     L 0.0;
      A     "TRAVEL_DRIVE_DB".DR_2_CW_B4_RMP_OUT_ZERO;
      =     DB3.DBX 137.4;
      A     L 0.0;
      A     "TRAVEL_DRIVE_DB".DR_2_CW_B5_RMP_HLD;
      =     DB3.DBX 137.5;
      A     L 0.0;
      A     "TRAVEL_DRIVE_DB".DR_2_CW_B6_RMP_IN_ZERO;
      =     DB3.DBX 137.6;
      A     L 0.0;
      A     "TRAVEL_DRIVE_DB".DR_2_CW_B7_FLT_RST;
      =     DB3.DBX 137.7;
      A     L 0.0;
      A     "TRAVEL_DRIVE_DB".DR_2_CW_B8_INCH_1;
      =     DB3.DBX 136.0;
      A     L 0.0;
      A     "TRAVEL_DRIVE_DB".DR_2_CW_B9_INCH_2;
      =     DB3.DBX 136.1;
      A     L 0.0;
      A     "TRAVEL_DRIVE_DB".DR_2_CW_B10_RMT_CMD;
      =     DB3.DBX 136.2;
NETWORK
TITLE =
      A     "ALWAYS_ON";
      JNB   M010;
      CALL  "DPWR_DAT" (
           LADDR                    := W#16#160,
           RECORD                   := P#DB3.DBX 136.0 BYTE 20,
           RET_VAL                  := "TRAVEL_DRIVE_DB".TR_DRV_2_CTRL_WORD_1_ERR);
M010: NOP   0;
END_FUNCTION

FUNCTION "TATA_COMMUNICATION" : VOID	// FC 14
VERSION : 0.1
BEGIN
// (block stored without names or comments; labels and parameter names are numbered)
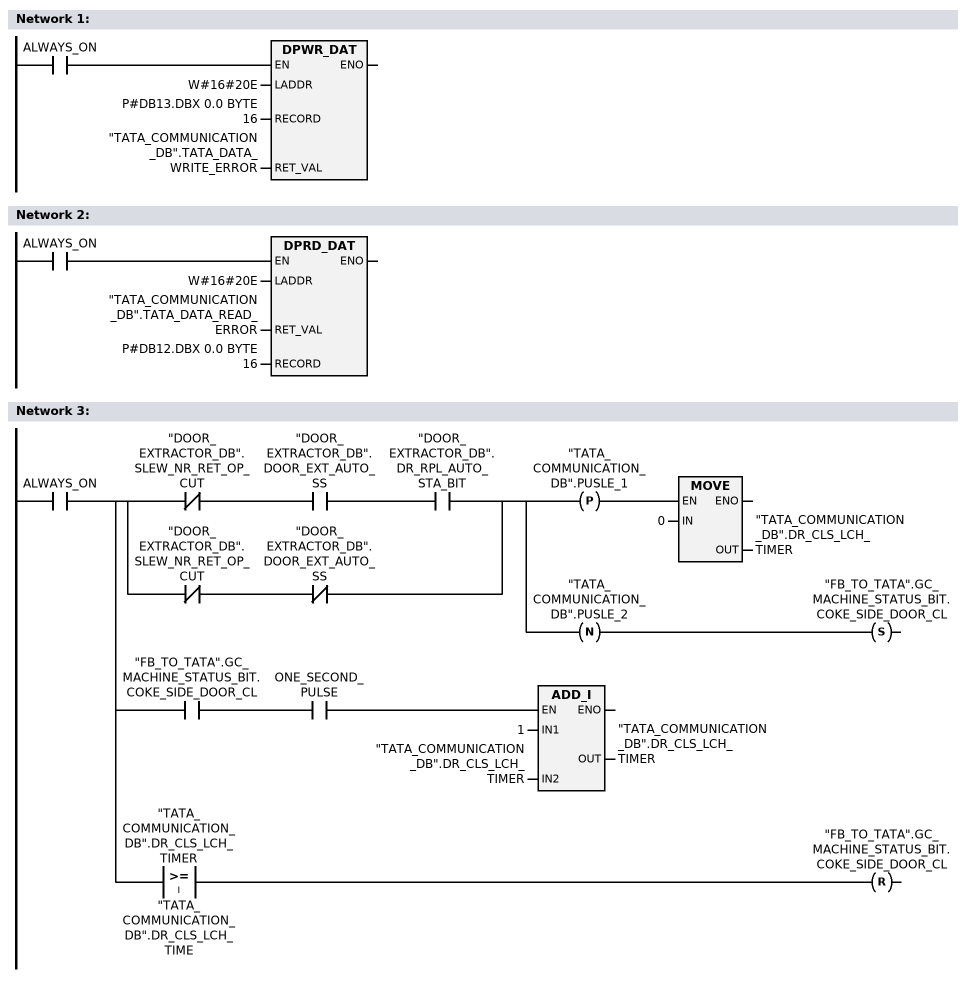
NETWORK
TITLE =
      A     "ALWAYS_ON";
      JNB   M001;
      CALL  "DPWR_DAT" (
           LADDR                    := W#16#20E,
           RECORD                   := P#DB13.DBX 0.0 BYTE 16,
           RET_VAL                  := "TATA_COMMUNICATION_DB".TATA_DATA_WRITE_ERROR);
M001: NOP   0;
NETWORK
TITLE =
      A     "ALWAYS_ON";
      JNB   M002;
      CALL  "DPRD_DAT" (
           LADDR                    := W#16#20E,
           RET_VAL                  := "TATA_COMMUNICATION_DB".TATA_DATA_READ_ERROR,
           RECORD                   := P#DB12.DBX 0.0 BYTE 16);
M002: NOP   0;
NETWORK
TITLE =
      A     "ALWAYS_ON";
      =     L 0.0;
      A     L 0.0;
      A(;
      AN    "DOOR_EXTRACTOR_DB".SLEW_NR_RET_OP_CUT;
      A     "DOOR_EXTRACTOR_DB".DOOR_EXT_AUTO_SS;
      A     "DOOR_EXTRACTOR_DB".DR_RPL_AUTO_STA_BIT;
      O;
      AN    "DOOR_EXTRACTOR_DB".SLEW_NR_RET_OP_CUT;
      AN    "DOOR_EXTRACTOR_DB".DOOR_EXT_AUTO_SS;
      );
      =     L 0.1;
      A     L 0.1;
      FP    "TATA_COMMUNICATION_DB".PUSLE_1;
      JNB   M003;
      L     0;
      T     "TATA_COMMUNICATION_DB".DR_CLS_LCH_TIMER;
M003: NOP   0;
      A     L 0.1;
      FN    "TATA_COMMUNICATION_DB".PUSLE_2;
      S     "FB_TO_TATA".GC_MACHINE_STATUS_BIT.COKE_SIDE_DOOR_CL;
      A     L 0.0;
      A     "FB_TO_TATA".GC_MACHINE_STATUS_BIT.COKE_SIDE_DOOR_CL;
      A     "ONE_SECOND_PULSE";
      JNB   M004;
      L     1;
      L     "TATA_COMMUNICATION_DB".DR_CLS_LCH_TIMER;
      +I;
      T     "TATA_COMMUNICATION_DB".DR_CLS_LCH_TIMER;
M004: NOP   0;
      A     L 0.0;
      A(;
      L     "TATA_COMMUNICATION_DB".DR_CLS_LCH_TIMER;
      L     "TATA_COMMUNICATION_DB".DR_CLS_LCH_TIME;
      >=I;
      );
      R     "FB_TO_TATA".GC_MACHINE_STATUS_BIT.COKE_SIDE_DOOR_CL;
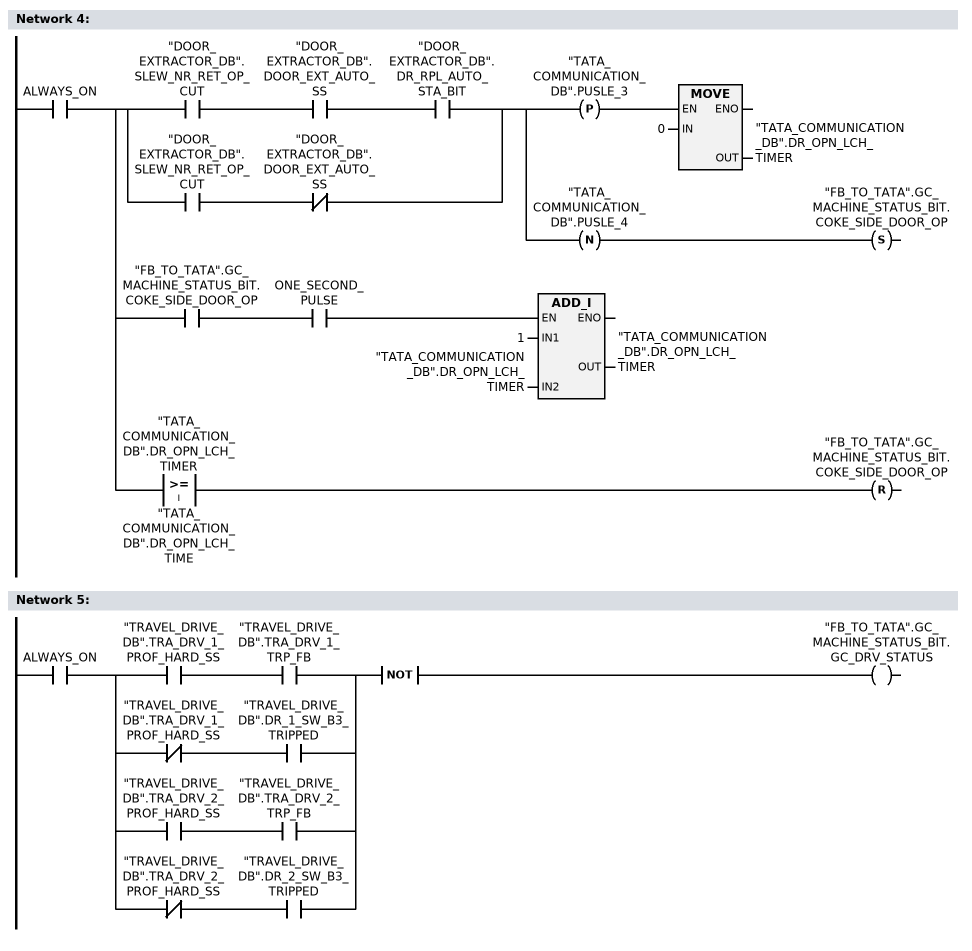
NETWORK
TITLE =
      A     "ALWAYS_ON";
      =     L 0.0;
      A     L 0.0;
      A(;
      A     "DOOR_EXTRACTOR_DB".SLEW_NR_RET_OP_CUT;
      A     "DOOR_EXTRACTOR_DB".DOOR_EXT_AUTO_SS;
      A     "DOOR_EXTRACTOR_DB".DR_RPL_AUTO_STA_BIT;
      O;
      A     "DOOR_EXTRACTOR_DB".SLEW_NR_RET_OP_CUT;
      AN    "DOOR_EXTRACTOR_DB".DOOR_EXT_AUTO_SS;
      );
      =     L 0.1;
      A     L 0.1;
      FP    "TATA_COMMUNICATION_DB".PUSLE_3;
      JNB   M005;
      L     0;
      T     "TATA_COMMUNICATION_DB".DR_OPN_LCH_TIMER;
M005: NOP   0;
      A     L 0.1;
      FN    "TATA_COMMUNICATION_DB".PUSLE_4;
      S     "FB_TO_TATA".GC_MACHINE_STATUS_BIT.COKE_SIDE_DOOR_OP;
      A     L 0.0;
      A     "FB_TO_TATA".GC_MACHINE_STATUS_BIT.COKE_SIDE_DOOR_OP;
      A     "ONE_SECOND_PULSE";
      JNB   M006;
      L     1;
      L     "TATA_COMMUNICATION_DB".DR_OPN_LCH_TIMER;
      +I;
      T     "TATA_COMMUNICATION_DB".DR_OPN_LCH_TIMER;
M006: NOP   0;
      A     L 0.0;
      A(;
      L     "TATA_COMMUNICATION_DB".DR_OPN_LCH_TIMER;
      L     "TATA_COMMUNICATION_DB".DR_OPN_LCH_TIME;
      >=I;
      );
      R     "FB_TO_TATA".GC_MACHINE_STATUS_BIT.COKE_SIDE_DOOR_OP;
NETWORK
TITLE =
      A     "ALWAYS_ON";
      A(;
      A     "TRAVEL_DRIVE_DB".TRA_DRV_1_PROF_HARD_SS;
      A     "TRAVEL_DRIVE_DB".TRA_DRV_1_TRP_FB;
      O;
      AN    "TRAVEL_DRIVE_DB".TRA_DRV_1_PROF_HARD_SS;
      A     "TRAVEL_DRIVE_DB".DR_1_SW_B3_TRIPPED;
      O;
      A     "TRAVEL_DRIVE_DB".TRA_DRV_2_PROF_HARD_SS;
      A     "TRAVEL_DRIVE_DB".TRA_DRV_2_TRP_FB;
      O;
      AN    "TRAVEL_DRIVE_DB".TRA_DRV_2_PROF_HARD_SS;
      A     "TRAVEL_DRIVE_DB".DR_2_SW_B3_TRIPPED;
      );
      NOT;
      =     "FB_TO_TATA".GC_MACHINE_STATUS_BIT.GC_DRV_STATUS;
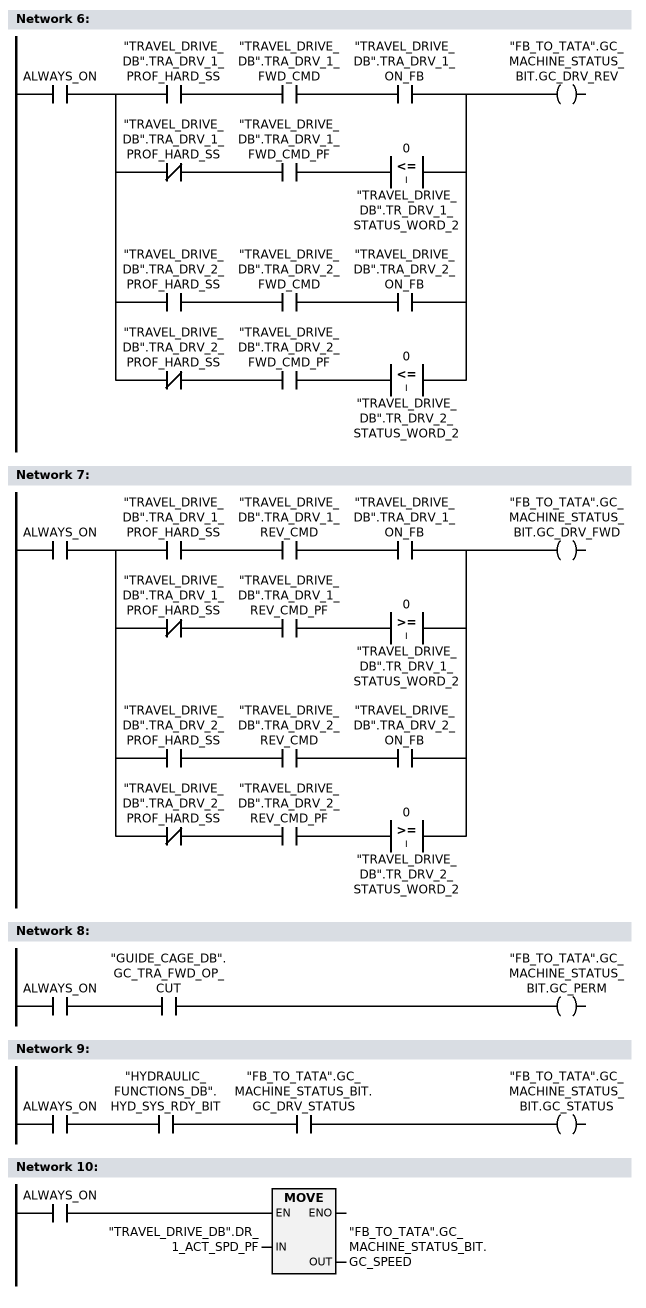
NETWORK
TITLE =
      A     "ALWAYS_ON";
      A(;
      A     "TRAVEL_DRIVE_DB".TRA_DRV_1_PROF_HARD_SS;
      A     "TRAVEL_DRIVE_DB".TRA_DRV_1_FWD_CMD;
      A     "TRAVEL_DRIVE_DB".TRA_DRV_1_ON_FB;
      O;
      AN    "TRAVEL_DRIVE_DB".TRA_DRV_1_PROF_HARD_SS;
      A     "TRAVEL_DRIVE_DB".TRA_DRV_1_FWD_CMD_PF;
      A(;
      L     0;
      L     "TRAVEL_DRIVE_DB".TR_DRV_1_STATUS_WORD_2;
      <=I;
      );
      O;
      A     "TRAVEL_DRIVE_DB".TRA_DRV_2_PROF_HARD_SS;
      A     "TRAVEL_DRIVE_DB".TRA_DRV_2_FWD_CMD;
      A     "TRAVEL_DRIVE_DB".TRA_DRV_2_ON_FB;
      O;
      AN    "TRAVEL_DRIVE_DB".TRA_DRV_2_PROF_HARD_SS;
      A     "TRAVEL_DRIVE_DB".TRA_DRV_2_FWD_CMD_PF;
      A(;
      L     0;
      L     "TRAVEL_DRIVE_DB".TR_DRV_2_STATUS_WORD_2;
      <=I;
      );
      );
      =     "FB_TO_TATA".GC_MACHINE_STATUS_BIT.GC_DRV_REV;
NETWORK
TITLE =
      A     "ALWAYS_ON";
      A(;
      A     "TRAVEL_DRIVE_DB".TRA_DRV_1_PROF_HARD_SS;
      A     "TRAVEL_DRIVE_DB".TRA_DRV_1_REV_CMD;
      A     "TRAVEL_DRIVE_DB".TRA_DRV_1_ON_FB;
      O;
      AN    "TRAVEL_DRIVE_DB".TRA_DRV_1_PROF_HARD_SS;
      A     "TRAVEL_DRIVE_DB".TRA_DRV_1_REV_CMD_PF;
      A(;
      L     0;
      L     "TRAVEL_DRIVE_DB".TR_DRV_1_STATUS_WORD_2;
      >=I;
      );
      O;
      A     "TRAVEL_DRIVE_DB".TRA_DRV_2_PROF_HARD_SS;
      A     "TRAVEL_DRIVE_DB".TRA_DRV_2_REV_CMD;
      A     "TRAVEL_DRIVE_DB".TRA_DRV_2_ON_FB;
      O;
      AN    "TRAVEL_DRIVE_DB".TRA_DRV_2_PROF_HARD_SS;
      A     "TRAVEL_DRIVE_DB".TRA_DRV_2_REV_CMD_PF;
      A(;
      L     0;
      L     "TRAVEL_DRIVE_DB".TR_DRV_2_STATUS_WORD_2;
      >=I;
      );
      );
      =     "FB_TO_TATA".GC_MACHINE_STATUS_BIT.GC_DRV_FWD;
NETWORK
TITLE =
      A     "ALWAYS_ON";
      A     "GUIDE_CAGE_DB".GC_TRA_FWD_OP_CUT;
      =     "FB_TO_TATA".GC_MACHINE_STATUS_BIT.GC_PERM;
NETWORK
TITLE =
      A     "ALWAYS_ON";
      A     "HYDRAULIC_FUNCTIONS_DB".HYD_SYS_RDY_BIT;
      A     "FB_TO_TATA".GC_MACHINE_STATUS_BIT.GC_DRV_STATUS;
      =     "FB_TO_TATA".GC_MACHINE_STATUS_BIT.GC_STATUS;
NETWORK
TITLE =
      A     "ALWAYS_ON";
      JNB   M007;
      L     "TRAVEL_DRIVE_DB".DR_1_ACT_SPD_PF;
      T     "FB_TO_TATA".GC_MACHINE_STATUS_BIT.GC_SPEED;
M007: NOP   0;
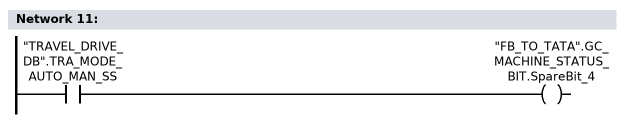
NETWORK
TITLE =
      A     "TRAVEL_DRIVE_DB".TRA_MODE_AUTO_MAN_SS;
      =     "FB_TO_TATA".GC_MACHINE_STATUS_BIT.SpareBit_4;
END_FUNCTION

// FC 105: know-how protected block, not included

// FC 106: know-how protected block, not included

DATA_BLOCK "MAIN_POWER_DB"	// DB 1
AUTHOR : Kamillas
VERSION : 0.1
  STRUCT
   MAIN_PWR_RDY_FOR_ON : BOOL ;	//MAIN POWER READY FOR ON
   MAIN_PWR_ON_FB : BOOL ;	//MAIN POWER ON FEED BACK
   CTRL_PWR_ON_FB : BOOL ;	//CONTROL POWER ON FEEDBACK
   MAIN_PWR_ON_PB : BOOL ;	//MAIN POWER ON PUSH BUTTON
   MAIN_PWR_OFF_PB : BOOL ;	//MAIN POWER OFF PUSH BUTTON
   LAMP_TEST_PB : BOOL ;	//LAMP TEST PUSH BUTTON
   ALARM_ACK_PB : BOOL ;	//ALARM ACKNOWLEDGE PUSH BUTTON
   MAIN_PWR_ON_CMD : BOOL ;	//MAIN POWER ON COMMAND
   MAIN_PWR_ON_IND : BOOL ;	//MAIN POWER ON INDICATOR
   CTRL_PWR_ON_IND : BOOL ;	//CONTROL POWER ON INDICATOR
   CTRL_SELECTION_CD : BOOL ;	//CONTROL SELECTRION CD
   MAIN_PWR_FLT : BOOL ;	//MAIN POWER FAULT
   CTRL_PWR_FLT : BOOL ;	//CTRL POWER FAULT
   MAIN_PWR_HEALTHY : BOOL ;	//MAIN POWER HEALTHY
   MAIN_PWR_FLT_TIMR : INT ;	//MAIN POWER FAULT TIMER
   MAIN_PWR_FLT_GEN_TIME : INT  := 3;	//MAIN POWER FAULT GENERATION TIME
   PULSE_1 : BOOL ;	//PULSE 1
   PULSE_2 : BOOL ;	//PULSE 2
   CTRL_PWR_FLT_TIMR : INT ;	//CONTROL POWER FAULT TIMER
   CTRL_PWR_FLT_GEN_TIME : INT  := 3;	//CONTROL POWER FAULT GENERATION TIME
   ALL_MECH_QUICK_STP : BOOL ;	//ALL MECHANICAL QUICK STOP
   CD_EMERGENCY_STOP : BOOL ;	//EMERGENCY STOP
   SERVICE_PF_STA_PB : BOOL ;	//SERVICE PLATFORM START PUSH BUTTON
   REP_MAN_SS : BOOL ;	//REPAIR MANUAL SELECTION
   SEMI_AUTO_SS : BOOL ;	//SEMI AUTO SELECTION
   TEST_BIT : BOOL ;	//TEST PURPOSE
  END_STRUCT ;	
BEGIN
   CTRL_PWR_FLT_GEN_TIME := 3;
END_DATA_BLOCK

DATA_BLOCK "HYDRAULIC_FUNCTIONS_DB"	// DB 2
AUTHOR : Kamillas
VERSION : 0.1
  STRUCT
   PUMP_1_RDY_FOR_STA : BOOL ;	//PUMP 1 READY FOR START
   PUMP_1_RUN_FB : BOOL ;	//PUMP 1 RUNNING FEEDBACK
   PUMP_1_OVR_LD_TRIP : BOOL ;	//PUMP 1 OVER LOAD TRIPPED
   PUMP_2_RDY_FOR_STA : BOOL ;	//PUMP 2 READY FOR START
   PUMP_2_RUN_FB : BOOL ;	//PUMP 2 RUNNING FEEDBACK
   PUMP_2_OVR_LD_TRIP : BOOL ;	//PUMP 2 OVER LOAD TRIPPED
   CIR_PUMP_RDY_FOR_STA : BOOL ;	//CIRCULATION PUMP READY FOR START
   CIR_PUMP_RUN_FB : BOOL ;	//CIRCULATION PUMP RUNNING FEEDBACK
   CIR_PUMP_OVR_LD_TRIP : BOOL ;	//CIRCULATION PUMP OVER LOAD TRIPPED
   COLR_FAN_RDY_FOR_STA : BOOL ;	//COOLER FAN READY FOR START
   COLR_FAN_RUN_FB : BOOL ;	//COOLER FAN RUNNING FEEDBACK
   COLR_FAN_OVR_LD_TRIP : BOOL ;	//COOLER FAN OVER LOAD TRIPPED
   CD_LCS_SS : BOOL ;	//CONTROL DESK / LOCAL CONTROL SELECTOR SWITCH
   PUMP_1_2_SS : BOOL ;	//PUMP 1 OR 2 SELECTOR SWITCH
   PUMP_1_STA_PB : BOOL ;	//PUMP 1 START PUSH BUTTON
   PUMP_1_STP_PB : BOOL ;	//PUMP 1 STOP PUSH BUTTON
   PUMP_2_STA_PB : BOOL ;	//PUMP 2 START PUSH BUTTON
   PUMP_2_STP_PB : BOOL ;	//PUMP 2 STOP PUSH BUTTON
   EMERGENCY_STOP_PB : BOOL ;	//EMERGENCY STOP PUSH BUTTON
   PUMP_1_2_SS_LCS : BOOL ;	//PUMP 1 OR 2 SELECTOR SWITCH LCS
   PUMP_1_STA_PB_LCS : BOOL ;	//PUMP 1 START PUSH BUTTON LCS
   PUMP_1_STP_PB_LCS : BOOL ;	//PUMP 1 STOP PUSH BUTTON LCS
   PUMP_2_STA_PB_LCS : BOOL ;	//PUMP 2 START PUSH BUTTON LCS
   PUMP_2_STP_PB_LCS : BOOL ;	//PUMP 2 STOP PUSH BUTTON LCS
   CIR_PUMP_STA_PB_LCS : BOOL ;	//CIRCULATION PUMP START PUSH BUTTON LCS
   CIR_PUMP_STP_PB_LCS : BOOL ;	//CIRCULATION PUMP STOP PUSH BUTTON LCS
   COLR_FAN_STA_PB_LCS : BOOL ;	//COOLER FAN START PUSH BUTTON LCS
   COLR_FAN_STP_PB_LCS : BOOL ;	//COOLER FAN STOP PUSH BUTTON LCS
   LAMP_TEST_PB_LCS_41 : BOOL ;	//LAMP TEST PUSH BUTTON LCS
   EMG_ACCM_STA_PB_LCS : BOOL ;	//EMERGENCY ACCUMULATOR START PB LCS
   EMG_ACCM_STP_PB_LCS : BOOL ;	//EMERGENCY ACCUMULATOR STOP PB LCS
   HTR_STA_PB_LCS : BOOL ;	//HEATER START PUSH BUTTON LCS
   HTR_STP_PB_LCS : BOOL ;	//HEATER STOP PUSH BUTTON LCS
   SHT_OF_VLV_LIN_1_FUL_OPN : BOOL ;	//SHUT OFF VALVE IN LINE 1 - FULLY OPEN
   SHT_OF_VLV_LIN_2_FUL_OPN : BOOL ;	//SHUT OFF VALVE IN LINE 2 - FULLY OPEN
   LOW_OIL_TEMP : BOOL ;	//LOW OIL TEMPERATURE - THERMOSTAT
   HIGH_OIL_TEMP : BOOL ;	//HIGH OIL TEMPERATURE - THERMOSTAT
   MAX_OIL_TEMP : BOOL ;	//MAXIMUM OIL TEMPERATURE - THERMOSTAT
   LOW_OIL_LEVEL : BOOL ;	//LOW OIL LEVEL - FLOAT SWITCH
   MIN_OIL_LEVEL : BOOL ;	//MINIMUM OIL LEVEL - FLOAT SWITCH
   RET_LIN_FLTR_CKD : BOOL ;	//RETURN LINE FILTER CHOKED
   LOW_OIL_PRESS : BOOL ;	//LOW OIL PRESSURE - PRESSURE SWITCH
   HIGH_OIL_PRESS : BOOL ;	//HIGH OIL PRESSURE - PRESSURE SWITCH
   PUMP_1_ON_CMD : BOOL ;	//PUMP 1 ON COMMAND
   PUMP_2_ON_CMD : BOOL ;	//PUMP 2 ON COMMAND
   CIR_PUMP_ON_CMD : BOOL ;	//CIRCULATION PUMP ON COMMAND
   CLR_FAN_ON_CMD : BOOL ;	//COOLER FAN ON COMMAND
   SYSTEM_RDY_IND : BOOL ;	//SYSTEM READY INDICATOR
   PUMP_1_ON_IND : BOOL ;	//PUMP 1 ON INDICATOR
   PUMP_2_ON_IND : BOOL ;	//PUMP 2 ON INDICATOR
   LCS_41_ON_IND_LCS : BOOL ;	//LCS 41 ON INDICATOR
   PUMP_1_ON_IND_LCS : BOOL ;	//PUMP 1 ON INDICATOR LCS
   PUMP_2_ON_IND_LCS : BOOL ;	//PUMP 2 ON INDICATOR LCS
   CIR_PUMP_ON_IND_LCS : BOOL ;	//CIRCULATION PUMP ON INDICATOR LCS
   CLR_FAN_ON_IND_LCS : BOOL ;	//COOLER FAN ON INDICATOR LCS
   HIGH_OIL_TEMP_IND_LCS : BOOL ;	//HIGH OIL TEMPERATURE INDICATOR LCS
   LOW_OIL_LEVEL_IND_LCS : BOOL ;	//LOW OIL LEVEL INDICATOR LCS
   LOW_OIL_TEMP_IND_LCS : BOOL ;	//LOW OIL TEMPERATURE INDICATOR LCS
   HTR_ON_IND_LCS : BOOL ;	//HEATER ON INDICATOR LCS
   FLTR_CHK_IND_LCS : BOOL ;	//FILTER CHOKE INDICATOR LCS
   ACCM_IN_OPER_IND_LCS : BOOL ;	//ACCUMULATOR IN OPERATION INDICATOR
   PRESS_REL_VLV_1_ON_CMD : BOOL ;	//PRESSURE RELIEF VALVE 1 ON COMMAND
   PRESS_REL_VLV_2_ON_CMD : BOOL ;	//PRESSURE RELIEF VALVE 2 ON COMMAND
   EMG_ACCM_ON_CMD : BOOL ;	//EMERGENCY ACCUMULLATOR ON COMMAND
   HYD_SYS_HEALTHY : BOOL ;	//HYDRAULIC SYSTEMS HEALTHY BIT
   PULSE_1 : BOOL ;	//PULSE 1
   PULSE_2 : BOOL ;	//PULSE 2
   PULSE_3 : BOOL ;	//PULSE 3
   PULSE_4 : BOOL ;	//PULSE 4
   PULSE_5 : BOOL ;	//PULSE 5
   PULSE_6 : BOOL ;	//PULSE 6
   HYD_PUMP_1_FLT : BOOL ;	//HYDRAULIC PUMP 1 FAULT
   HYD_PUMP_2_FLT : BOOL ;	//HYDRAULIC PUMP 2 FAULT
   HYD_PUMP_1_FLT_TMR : INT ;	//HYDRAULIC PUMP 1 FAULT TIMER
   HYD_PUMP_1_FLT_GEN_TIME : INT  := 3;	//HYDRAULIC PUMP 1 FAULT GEMERATION TIME
   HYD_PUMP_2_FLT_TMR : INT ;	//HYDRAULIC PUMP 2 FAULT TIMER
   HYD_PUMP_2_FLT_GEN_TIME2 : INT  := 3;	//HYDRAULIC PUMP 2 FAULT GEMERATION TIME
   PRS_REL_VLV_1_OPN_TMR : INT ;	//PRESSURE RELEIF VALVE 1 OPEN TIMER
   PRS_REL_VLV_1_OPN_ST_TIM : INT  := 8;	//PRESSURE RELEIF VALVE 1 OPEN SET TIME
   PRS_REL_VLV_2_OPN_TMR : INT ;	//PRESSURE RELEIF VALVE 2 OPEN TIMER
   PRS_REL_VLV_2_OPN_ST_TIM : INT  := 8;	//PRESSURE RELEIF VALVE 2 OPEN SET TIME
   CIR_PUMP_FLT : BOOL ;	//CIRCULATION PUMP 1 FAULT
   CLR_FAN_FLT : BOOL ;	//COOLER FAN FAULT
   CIR_PUMP_FLT_TMR : INT ;	//CIRCULATION PUMP FAULT TIMER
   CIR_PUMP_FLT_GEN_TIME : INT  := 3;	//CIRCULATION PUMP FAULT GEMERATION TIME
   CLR_FAN_FLT_TMR : INT ;	//HYDRAULIC PUMP 2 FAULT TIMER
   CLR_FAN_FLT_GEN_TIME : INT  := 3;	//COOLER FAN FAULT GEMERATION TIME
   HYD_SYS_RDY_BIT : BOOL ;	//HYDRAULIC SYSTEM READY BIT
   PUMP_1_ON_CMD_CD : BOOL ;	//PUMP 1 ON COMMAND FROM CD
   PUMP_1_ON_CMD_LCS : BOOL ;	//PUMP 1 ON COMMAND FROM LCS
   PUMP_2_ON_CMD_LCS : BOOL ;	//PUMP 2 ON COMMAND LCS
   PUMP_2_ON_CMD_CD : BOOL ;	//PUMP 2 ON COMMAND CD
  END_STRUCT ;	
BEGIN
   HYD_PUMP_1_FLT_GEN_TIME := 3;
   HYD_PUMP_2_FLT_GEN_TIME2 := 3;
   PRS_REL_VLV_1_OPN_ST_TIM := 3;
   PRS_REL_VLV_2_OPN_ST_TIM := 8;
   CIR_PUMP_FLT_GEN_TIME := 3;
   CLR_FAN_FLT_GEN_TIME := 3;
END_DATA_BLOCK

DATA_BLOCK "TRAVEL_DRIVE_DB"	// DB 3
AUTHOR : Kamillas
VERSION : 0.1
  STRUCT
   TRA_DRV_1_BRK_RDY_FOR_ST : BOOL ;	//TRAVEL GROUP 1 BREAK READY FOR START
   TRA_DRV_1_BRK_ON_FB : BOOL ;	//TRAVEL GROUP 1 BREAK ON FEEDBACK
   TRA_DRV_2_BRK_RDY_FOR_ST : BOOL ;	//TRAVEL GROUP 2 BREAK READY FOR START
   TRA_DRV_2_BRK_ON_FB : BOOL ;	//TRAVEL GROUP 2 BREAK ON FEEDBACK
   TRA_MODE_AUTO_MAN_SS : BOOL ;	//TRAVEL MODE AUTO/MANUAL BUTTON
   AUTO_POS_ACK : BOOL ;	//AUTO POSITION ACKNOWLEDGE
   TRA_DRV_1_PROF_HARD_SS : BOOL ;	//TRAVEL DRIVE 1 PROFIBUS/HARD WIRE SELECTRO SWITCH
   TRA_DRV_1_ON_FB : BOOL ;	//TRAVEL DRIVE 1 ON FEEDBACK
   TRA_DRV_1_RDY_FOR_STA : BOOL ;	//TRAVEL DRIVE 1 READY FOR START
   TRA_DRV_1_TRP_FB : BOOL ;	//TRAVEL DRIVE 1 TRIP FEEDBACK
   TRA_DRV_2_PROF_HARD_SS : BOOL ;	//TRAVEL DRIVE 2 PROFIBUS/HARD WIRE SELECTRO SWITCH
   TRA_DRV_2_ON_FB : BOOL ;	//TRAVEL DRIVE 2 ON FEEDBACK
   TRA_DRV_2_RDY_FOR_STA : BOOL ;	//TRAVEL DRIVE 2 READY FOR START
   TRA_DRV_2_TRP_FB : BOOL ;	//TRAVEL DRIVE 2 TRIP FEEDBACK
   LIMIT_SW_END_FWD_FB : BOOL ;	//LIMIT SWITCH END FORWARD FEEDBACK`
   LIMIT_SW_END_REV_FB : BOOL ;	//LIMIT SWITCH END REVERSE FEEDBACK
   TRA_DRV_1_ON_CMD : BOOL ;	//TRAVEL GROUP 1 ON COMMAND
   TRA_DRV_2_ON_CMD : BOOL ;	//TRAVEL GROUP 2 ON COMMAND
   TRA_DRV_1_BRK_ON_CMD : BOOL ;	//TRAVEL GROUP 1 BRAKE ON COMMAND
   TRA_DRV_2_BRK_ON_CMD : BOOL ;	//TRAVEL GROUP 2 BRAKE ON COMMAND
   TRA_PER_IND : BOOL ;	//TRAVEL PERMISSION INDICATOR
   AUTO_POS_ON : BOOL ;	//AUTO POSITION ON
   TRA_DRV_1_FWD_CMD : BOOL ;	//TRAVEL DRIVE 1 FORWARD COMMAND
   TRA_DRV_1_REV_CMD : BOOL ;	//TRAVEL DRIVE 1 REVERSE COMMAND
   TRA_DRV_2_FWD_CMD : BOOL ;	//TRAVEL DRIVE 2 FORWARD COMMAND
   TRA_DRV_2_REV_CMD : BOOL ;	//TRAVEL DRIVE 2 REVERSE COMMAND
   TRA_JOY_STK_FWD_POS : BOOL ;	//TRAVEL JOY STICK FOWRWARD POSITION
   TRA_JOY_STK_REV_POS : BOOL ;	//TRAVEL JOY DEAD REVERSE POSITION
   TRA_JOY_STK_HME_POS : BOOL ;	//TRAVEL JOY STICK HOME POSITION
   TRA_JOY_STK_DED_MAN_BTN : BOOL ;	//TRAVEL JOY DEAD MAN BUTTON
   TRA_ILK_BIT : BOOL ;	//TRAVEL OPERATIONS INTERLOCK BIT
   TRA_ILK_INM_BIT_1 : BOOL ;	//TRAVEL INTERLOCK INTERMEDIATE BIT 1
   TRA_ILK_INM_BIT_2 : BOOL ;	//TRAVEL INTERLOCK INTERMEDIATE BIT 2
   TRA_ILK_INM_BIT_3 : BOOL ;	//TRAVEL INTERLOCK INTERMEDIATE BIT 3
   TRA_DRV_1_2_BRK_FLT : BOOL ;	//TRAVEL DRIVE BREAK 1 AND 2 FAULT
   TRA_DRV_1_2_BRK_FLT_TMR : INT ;	//TRAVEL DRIVE BREAK 1 AND 2 FAULT TIMER
   JS_SPD_REF_DI : DINT ;	//JOY STICK SPEED REFERENCE IN DOUBLE INTEGER
   JS_SPD_REF_NEG_RMD : INT ;	//JOY STICK SPEED REFERENCE CONVERTERD TO POSITIVE VALUE
   JS_SPD_REF_REAL : REAL ;	//JOY STICK SPEED REFERENCE IN REAL(FLOATING POINT)
   JS_SPD_REF_UN_SL_FLT : WORD ;	//JOY STICK SPEED REFERENCE UNSCALLING FAULT
   TRA_SPD_REF_VAL : INT ;	//TRAVEL SPEED REFERENCE VALUE
   TRA_SPD_REF_VAL_FRM_JS : INT ;	//TRAVEL SPEED REFERENCE VALUW FROM JOYSTICK
   TR_DRV_1_STATUS_WORD_1 : INT ;	//TRAVEL DRIVE 1 PROFIBUS STATUS WORD 1
   TR_DRV_1_STATUS_WORD_2 : INT ;	//TRAVEL DRIVE 1 PROFIBUS STATUS WORD 2
   TR_DRV_1_STATUS_WORD_3 : INT ;	//TRAVEL DRIVE 1 PROFIBUS STATUS WORD 3
   TR_DRV_1_STATUS_WORD_4 : INT ;	//TRAVEL DRIVE 1 PROFIBUS STATUS WORD 4
   TR_DRV_1_STATUS_WORD_5 : INT ;	//TRAVEL DRIVE 1 PROFIBUS STATUS WORD 5
   TR_DRV_1_STATUS_WORD_6 : INT ;	//TRAVEL DRIVE 1 PROFIBUS STATUS WORD 6
   TR_DRV_1_STATUS_WORD_7 : INT ;	//TRAVEL DRIVE 1 PROFIBUS STATUS WORD 7
   TR_DRV_1_STATUS_WORD_8 : INT ;	//TRAVEL DRIVE 1 PROFIBUS STATUS WORD 8
   TR_DRV_1_STATUS_WORD_9 : INT ;	//TRAVEL DRIVE 1 PROFIBUS STATUS WORD 9
   TR_DRV_1_STATUS_WORD_10 : INT ;	//TRAVEL DRIVE 1 PROFIBUS STATUS WORD 10
   TR_DRV_1_STATUS_WORD_11 : INT ;	//TRAVEL DRIVE 1 PROFIBUS STATUS WORD 11
   TR_DRV_1_STATUS_WORD_12 : INT ;	//TRAVEL DRIVE 1 PROFIBUS STATUS WORD 12
   TR_DRV_1_STATUS_WORD_13 : INT ;	//TRAVEL DRIVE 1 PROFIBUS STATUS WORD 13
   TR_DRV_1_STATUS_WORD_14 : INT ;	//TRAVEL DRIVE 1 PROFIBUS STATUS WORD 14
   TR_DRV_1_STATUS_WORD_15 : INT ;	//TRAVEL DRIVE 1 PROFIBUS STATUS WORD 15
   TR_DRV_1_STATUS_WORD_16 : INT ;	//TRAVEL DRIVE 1 PROFIBUS STATUS WORD 16
   TR_DRV_1_CONTROL_WORD_1 : INT ;	//TRAVEL DRIVE 1 PROFIBUS CONTROL WORD 1
   TR_DRV_1_CONTROL_WORD_2 : INT ;	//TRAVEL DRIVE 1 PROFIBUS CONTROL WORD 2
   TR_DRV_1_CONTROL_WORD_3 : INT ;	//TRAVEL DRIVE 1 PROFIBUS CONTROL WORD 3
   TR_DRV_1_CONTROL_WORD_4 : INT ;	//TRAVEL DRIVE 1 PROFIBUS CONTROL WORD 4
   TR_DRV_1_CONTROL_WORD_5 : INT ;	//TRAVEL DRIVE 1 PROFIBUS CONTROL WORD 5
   TR_DRV_1_CONTROL_WORD_6 : INT ;	//TRAVEL DRIVE 1 PROFIBUS CONTROL WORD 6
   TR_DRV_1_CONTROL_WORD_7 : INT ;	//TRAVEL DRIVE 1 PROFIBUS CONTROL WORD 7
   TR_DRV_1_CONTROL_WORD_8 : INT ;	//TRAVEL DRIVE 1 PROFIBUS CONTROL WORD 8
   TR_DRV_1_CONTROL_WORD_9 : INT ;	//TRAVEL DRIVE 1 PROFIBUS CONTROL WORD 9
   TR_DRV_1_CONTROL_WORD_10 : INT ;	//TRAVEL DRIVE 1 PROFIBUS CONTROL WORD 10
   TR_DRV_1_CONTROL_WORD_11 : INT ;	//TRAVEL DRIVE 1 PROFIBUS CONTROL WORD 11
   TR_DRV_1_CONTROL_WORD_12 : INT ;	//TRAVEL DRIVE 1 PROFIBUS CONTROL WORD 12
   TR_DRV_1_CONTROL_WORD_13 : INT ;	//TRAVEL DRIVE 1 PROFIBUS CONTROL WORD 13
   TR_DRV_1_CONTROL_WORD_14 : INT ;	//TRAVEL DRIVE 1 PROFIBUS CONTROL WORD 14
   TR_DRV_1_CONTROL_WORD_15 : INT ;	//TRAVEL DRIVE 1 PROFIBUS CONTROL WORD 15
   TR_DRV_1_CONTROL_WORD_16 : INT ;	//TRAVEL DRIVE 1 PROFIBUS CONTROL WORD 16
   TR_DRV_1_STAT_WORD_1_ERR : INT ;	//TRAVEL DRIVE 1 DRIVE STATUS WORD 1 READ ERROR
   TR_DRV_1_STAT_WORD_2_ERR : INT ;	//TRAVEL DRIVE 1 DRIVE STATUS WORD 2 READ ERROR
   TR_DRV_1_STAT_WORD_3_ERR : INT ;	//TRAVEL DRIVE 1 DRIVE STATUS WORD 3 READ ERROR
   TR_DRV_1_STAT_WORD_4_ERR : INT ;	//TRAVEL DRIVE 1 DRIVE STATUS WORD 4 READ ERROR
   TR_DRV_1_CTRL_WORD_1_ERR : INT ;	//TRAVEL DRIVE 1 DRIVE CONTROL WORD 1 WRITE ERROR
   TR_DRV_1_CTRL_WORD_2_ERR : INT ;	//TRAVEL DRIVE 1 DRIVE CONTROL WORD 2 WRITE ERROR
   TR_DRV_1_CTRL_WORD_3_ERR : INT ;	//TRAVEL DRIVE 1 DRIVE CONTROL WORD 3 WRITE ERROR
   TR_DRV_1_CTRL_WORD_4_ERR : INT ;	//TRAVEL DRIVE 1 DRIVE CONTROL WORD 4 WRITE ERROR
   TR_DRV_2_STATUS_WORD_1 : INT ;	//TRAVEL DRIVE 2 PROFIBUS STATUS WORD 1
   TR_DRV_2_STATUS_WORD_2 : INT ;	//TRAVEL DRIVE 2 PROFIBUS STATUS WORD 2
   TR_DRV_2_STATUS_WORD_3 : INT ;	//TRAVEL DRIVE 2 PROFIBUS STATUS WORD 3
   TR_DRV_2_STATUS_WORD_4 : INT ;	//TRAVEL DRIVE 2 PROFIBUS STATUS WORD 4
   TR_DRV_2_STATUS_WORD_5 : INT ;	//TRAVEL DRIVE 2 PROFIBUS STATUS WORD 5
   TR_DRV_2_STATUS_WORD_6 : INT ;	//TRAVEL DRIVE 2 PROFIBUS STATUS WORD 6
   TR_DRV_2_STATUS_WORD_7 : INT ;	//TRAVEL DRIVE 2 PROFIBUS STATUS WORD 7
   TR_DRV_2_STATUS_WORD_8 : INT ;	//TRAVEL DRIVE 2 PROFIBUS STATUS WORD 8
   TR_DRV_2_STATUS_WORD_9 : INT ;	//TRAVEL DRIVE 2 PROFIBUS STATUS WORD 9
   TR_DRV_2_STATUS_WORD_10 : INT ;	//TRAVEL DRIVE 2 PROFIBUS STATUS WORD 10
   TR_DRV_2_STATUS_WORD_11 : INT ;	//TRAVEL DRIVE 2 PROFIBUS STATUS WORD 11
   TR_DRV_2_STATUS_WORD_12 : INT ;	//TRAVEL DRIVE 2 PROFIBUS STATUS WORD 12
   TR_DRV_2_STATUS_WORD_13 : INT ;	//TRAVEL DRIVE 2 PROFIBUS STATUS WORD 13
   TR_DRV_2_STATUS_WORD_14 : INT ;	//TRAVEL DRIVE 2 PROFIBUS STATUS WORD 14
   TR_DRV_2_STATUS_WORD_15 : INT ;	//TRAVEL DRIVE 2 PROFIBUS STATUS WORD 15
   TR_DRV_2_STATUS_WORD_16 : INT ;	//TRAVEL DRIVE 2 PROFIBUS STATUS WORD 16
   TR_DRV_2_CONTROL_WORD_1 : INT ;	//TRAVEL DRIVE 2 PROFIBUS CONTROL WORD 1
   TR_DRV_2_CONTROL_WORD_2 : INT ;	//TRAVEL DRIVE 2 PROFIBUS CONTROL WORD 2
   TR_DRV_2_CONTROL_WORD_3 : INT ;	//TRAVEL DRIVE 2 PROFIBUS CONTROL WORD 3
   TR_DRV_2_CONTROL_WORD_4 : INT ;	//TRAVEL DRIVE 2 PROFIBUS CONTROL WORD 4
   TR_DRV_2_CONTROL_WORD_5 : INT ;	//TRAVEL DRIVE 2 PROFIBUS CONTROL WORD 5
   TR_DRV_2_CONTROL_WORD_6 : INT ;	//TRAVEL DRIVE 2 PROFIBUS CONTROL WORD 6
   TR_DRV_2_CONTROL_WORD_7 : INT ;	//TRAVEL DRIVE 2 PROFIBUS CONTROL WORD 7
   TR_DRV_2_CONTROL_WORD_8 : INT ;	//TRAVEL DRIVE 2 PROFIBUS CONTROL WORD 8
   TR_DRV_2_CONTROL_WORD_9 : INT ;	//TRAVEL DRIVE 2 PROFIBUS CONTROL WORD 9
   TR_DRV_2_CONTROL_WORD_10 : INT ;	//TRAVEL DRIVE 2 PROFIBUS CONTROL WORD 10
   TR_DRV_2_CONTROL_WORD_11 : INT ;	//TRAVEL DRIVE 2 PROFIBUS CONTROL WORD 11
   TR_DRV_2_CONTROL_WORD_12 : INT ;	//TRAVEL DRIVE 2 PROFIBUS CONTROL WORD 12
   TR_DRV_2_CONTROL_WORD_13 : INT ;	//TRAVEL DRIVE 2 PROFIBUS CONTROL WORD 13
   TR_DRV_2_CONTROL_WORD_14 : INT ;	//TRAVEL DRIVE 2 PROFIBUS CONTROL WORD 14
   TR_DRV_2_CONTROL_WORD_15 : INT ;	//TRAVEL DRIVE 2 PROFIBUS CONTROL WORD 15
   TR_DRV_2_CONTROL_WORD_16 : INT ;	//TRAVEL DRIVE 2 PROFIBUS CONTROL WORD 16
   TR_DRV_2_STAT_WORD_1_ERR : INT ;	//TRAVEL DRIVE 2 DRIVE STATUS WORD 1 READ ERROR
   TR_DRV_2_STAT_WORD_2_ERR : INT ;	//TRAVEL DRIVE 2 DRIVE STATUS WORD 2 READ ERROR
   TR_DRV_2_STAT_WORD_3_ERR : INT ;	//TRAVEL DRIVE 2 DRIVE STATUS WORD 3 READ ERROR
   TR_DRV_2_STAT_WORD_4_ERR : INT ;	//TRAVEL DRIVE 2 DRIVE STATUS WORD 4 READ ERROR
   TR_DRV_2_CTRL_WORD_1_ERR : INT ;	//TRAVEL DRIVE 2 DRIVE CONTROL WORD 1 WRITE ERROR
   TR_DRV_2_CTRL_WORD_2_ERR : INT ;	//TRAVEL DRIVE 2 DRIVE CONTROL WORD 2 WRITE ERROR
   TR_DRV_2_CTRL_WORD_3_ERR : INT ;	//TRAVEL DRIVE 2 DRIVE CONTROL WORD 3 WRITE ERROR
   TR_DRV_2_CTRL_WORD_4_ERR : INT ;	//TRAVEL DRIVE 2 DRIVE CONTROL WORD 4 WRITE ERROR
   DR_1_RDY_TO_ON_PF : BOOL ;	//TRAVEL DRIVE 1 READY TO SWITCH ON - PROFIBUS
   DR_1_RDY_TO_OPER_PF : BOOL ;	//TRAVEL DRIVE 1 READY TO OPERATE BIT - PROFIBUS
   DR_1_ENAB_OPER_PF : BOOL ;	//TRAVEL DRIVE 1 ENABLE OPERATIONS - PROFIBUS
   DR_1_FLT_PF : BOOL ;	//TRAVEL DRIVE 1 FAULT - PROFIBUS
   DR_1_SPD_FB_PF : REAL ;	//TRAVEL DRIVE 1 SPEED FEED BACK FROM DRIVE - PROFIBUS
   DR_1_SPD_REF_DI_PF : DINT ;	//TRAVEL DRIVE 1 SPEED REFERENCE IN DOUBLE INTEGER - PROFIBUS
   DR_1_SPD_REF_NEG_RMD_PF : INT ;	//TRAVEL DRIVE 1 SPEED REFERENCE CONVERTERD TO POSITIVE VALUE - PROFIBUS
   DR_1_SPD_REF_REAL_PF : REAL ;	//TRAVEL DRIVE 1 SPEED REFERENCE IN REAL(FLOATING POINT) - PROFIBUS
   DR_1_SPD_RE_UN_SL_FLT_PF : WORD ;	//TRAVEL DRIVE 1 SPEED REFERENCE UNSCALLING FAULT - PROFIBUS
   DR_2_RDY_TO_ON_PF : BOOL ;	//TRAVEL DRIVE 2 READY TO SWITCH ON - PROFIBUS
   DR_2_RDY_TO_OPER_PF : BOOL ;	//TRAVEL DRIVE 2 READY TO OPERATE BIT - PROFIBUS
   DR_2_ENAB_OPER_PF : BOOL ;	//TRAVEL DRIVE 2 ENABLE OPERATIONS - PROFIBUS
   DR_2_FLT_PF : BOOL ;	//TRAVEL DRIVE 2 FAULT - PROFIBUS
   DR_2_SPD_FB_PF : REAL ;	//TRAVEL DRIVE 2 SPEED FEED BACK FROM DRIVE - PROFIBUS
   DR_2_SPD_REF_DI_PF : DINT ;	//TRAVEL DRIVE 2 SPEED REFERENCE IN DOUBLE INTEGER - PROFIBUS
   DR_2_SPD_REF_NEG_RMD_PF : INT ;	//TRAVEL DRIVE 2 SPEED REFERENCE CONVERTERD TO POSITIVE VALUE - PROFIBUS
   DR_2_SPD_REF_REAL_PF : REAL ;	//TRAVEL DRIVE 2 SPEED REFERENCE IN REAL(FLOATING POINT) - PROFIBUS
   DR_2_SPD_RE_UN_SL_FLT_PF : WORD ;	//TRAVEL DRIVE 2 SPEED REFERENCE UNSCALLING FAULT - PROFIBUS
   PULSE_1 : BOOL ;	//PULSE 1
   PULSE_2 : BOOL ;	//PULSE 2
   PULSE_3 : BOOL ;	//PULSE 3
   PULSE_4 : BOOL ;	//PULSE 4
   LIMIT_SW_END_EMG_FWD_FB : BOOL ;	//LIMIT SWITCH END EMWRGENCY FWD FEEDBACK
   LIMIT_SW_END_EMG_REV_FB : BOOL ;	//LIMIT SWITCH END EMERGENCY REVERSE FEEDBACK
   DR_1_CW_B0_RDY_TO_OPER : BOOL ;	//TRAVEL DRIVE 1 CONTROL WORD BIT 0 - READY TO OPERATE - OFF1 - PROFIBUS
   DR_1_CW_B1_OFF_2 : BOOL ;	//TRAVEL DRIVE 1 CONTROL WORD BIT 1 - OFF2 - PROFIBUS
   DR_1_CW_B2_OFF_3 : BOOL ;	//TRAVEL DRIVE 1 CONTROL WORD BIT 2 - OFF3 - PROFIBUS
   DR_1_CW_B3_OPER_ENAB : BOOL ;	//TRAVEL DRIVE 1 CONTROL WORD BIT 3 - OPERATION ENABLE - PROFIBUS
   DR_1_CW_B4_RMP_OUT_ZERO : BOOL ;	//TRAVEL DRIVE 1 CONTROL WORD BIT 4 - RAMP OUT ZERO - PROFIBUS
   DR_1_CW_B5_RMP_HLD : BOOL ;	//TRAVEL DRIVE 1 CONTROL WORD BIT 5 - RAMP HOLD - PROFIBUS
   DR_1_CW_B6_RMP_IN_ZERO : BOOL ;	//TRAVEL DRIVE 1 CONTROL WORD BIT 6 - RAMP IN ZERO - PROFIBUS
   DR_1_CW_B7_FLT_RST : BOOL ;	//TRAVEL DRIVE 1 CONTROL WORD BIT 7 - FAULT RESET - PROFIBUS
   DR_1_CW_B8_INCH_1 : BOOL ;	//TRAVEL DRIVE 1 CONTROL WORD BIT 8 - INCHING 1 - PROFIBUS
   DR_1_CW_B9_INCH_2 : BOOL ;	//TRAVEL DRIVE 1 CONTROL WORD BIT 9 - INCHING 2 - PROFIBUS
   DR_1_CW_B10_RMT_CMD : BOOL ;	//TRAVEL DRIVE 1 CONTROL WORD BIT 10 - REMOTE COMMAND - PROFIBUS
   DR_1_CW_B11 : BOOL ;	//TRAVEL DRIVE 1 CONTROL WORD BIT 11 - DRIVE SPECIFIC - PROFOBUS
   DR_1_CW_B12 : BOOL ;	//TRAVEL DRIVE 1 CONTROL WORD BIT 12 - DRIVE SPECIFIC - PROFOBUS
   DR_1_CW_B13 : BOOL ;	//TRAVEL DRIVE 1 CONTROL WORD BIT 13 - DRIVE SPECIFIC - PROFOBUS
   DR_1_CW_B14 : BOOL ;	//TRAVEL DRIVE 1 CONTROL WORD BIT 14 - DRIVE SPECIFIC - PROFOBUS
   DR_1_CW_B15 : BOOL ;	//TRAVEL DRIVE 1 CONTROL WORD BIT 15 - DRIVE SPECIFIC - PROFOBUS
   DR_1_SW_B0_RDY_ON : BOOL ;	//TRAVEL DRIVE 1 STATUS WORD BIT 0 - READY TO OPERATE - OFF1 - PROFIBUS
   DR_1_SW_B1_RDY_TO_OPER : BOOL ;	//TRAVEL DRIVE 1 STATUS WORD BIT 1 - REDY TO OPERATE - PROFIBUS
   DR_1_SW_B2_REF_RDY : BOOL ;	//TRAVEL DRIVE 1 STATUS WORD BIT 2 - ENABEL OPERATION - PROFIBUS
   DR_1_SW_B3_TRIPPED : BOOL ;	//TRAVEL DRIVE 1 STATUS WORD BIT 3 - FAULT - PROFIBUS
   DR_1_SW_B4_OFF_2_STA : BOOL ;	//TRAVEL DRIVE 1 STATUS WORD BIT 4 - OFF 2 STATUS - PROFIBUS
   DR_1_SW_B5_OFF_3_STA : BOOL ;	//TRAVEL DRIVE 1 STATUS WORD BIT 5 - OFF 3 STATUS - PROFIBUS
   DR_1_SW_B6_SWC_ON_INHB : BOOL ;	//TRAVEL DRIVE 1 STATUS WORD BIT 6 - SWITCH ON INHIBIT - PROFIBUS
   DR_1_SW_B7_ALARM : BOOL ;	//TRAVEL DRIVE 1 STATUS WORD BIT 7 - WARNING/ALARM - PROFIBUS
   DR_1_SW_B8_AT_SETPOINT : BOOL ;	//TRAVEL DRIVE 1 STATUS WORD BIT 8 - OPERATING - PROFIBUS
   DR_1_SW_B9_REMOTE : BOOL ;	//TRAVEL DRIVE 1 STATUS WORD BIT 9 - DRIVE CONTROL REMOTE\LOCAL - PROFIBUS
   DR_1_SW_B10_ABOVE_LIMIT : BOOL ;	//TRAVEL DRIVE 1 STATUS WORD BIT 10 - SPEED ABOVE LIMIT - PROFIBUS
   DR_1_SW_B11 : BOOL ;	//TRAVEL DRIVE 1 STATUS WORD BIT 11 - DRIVE SPECIFIC - PROFOBUS
   DR_1_SW_B12 : BOOL ;	//TRAVEL DRIVE 1 STATUS WORD BIT 12 - DRIVE SPECIFIC - PROFOBUS
   DR_1_SW_B13 : BOOL ;	//TRAVEL DRIVE 1 STATUS WORD BIT 13 - DRIVE SPECIFIC - PROFOBUS
   DR_1_SW_B14 : BOOL ;	//TRAVEL DRIVE 1 STATUS WORD BIT 14 - DRIVE SPECIFIC - PROFOBUS
   DR_1_SW_B15 : BOOL ;	//TRAVEL DRIVE 1 STATUS WORD BIT 15 - DRIVE SPECIFIC - PROFOBUS
   JS_SPD_REF_DI_PF : DINT ;	//JOY STICK SPEED REFERENCE IN DOUBLE INTEGER
   JS_SPD_REF_REAL_PF : REAL ;	//JOY STICK SPEED REFERENCE IN REAL(FLOATING POINT)
   JS_SPD_REF_UN_SL_FLT_PF : WORD ;	//JOY STICK SPEED REFERENCE UNSCALLING FAULT
   TRA_SPD_REF_VAL_PF : INT ;	//TRAVEL SPEED REFERENCE VALUE
   DR_2_CW_B0_RDY_TO_OPER : BOOL ;	//TRAVEL DRIVE 2 CONTROL WORD BIT 0 - READY TO OPERATE - OFF1 - PROFIBUS
   DR_2_CW_B1_OFF_2 : BOOL ;	//TRAVEL DRIVE 2 CONTROL WORD BIT 1 - OFF2 - PROFIBUS
   DR_2_CW_B2_OFF_3 : BOOL ;	//TRAVEL DRIVE 2 CONTROL WORD BIT 2 - OFF3 - PROFIBUS
   DR_2_CW_B3_OPER_ENAB : BOOL ;	//TRAVEL DRIVE 2 CONTROL WORD BIT 3 - OPERATION ENABLE - PROFIBUS
   DR_2_CW_B4_RMP_OUT_ZERO : BOOL ;	//TRAVEL DRIVE 2 CONTROL WORD BIT 4 - RAMP OUT ZERO - PROFIBUS
   DR_2_CW_B5_RMP_HLD : BOOL ;	//TRAVEL DRIVE 2 CONTROL WORD BIT 5 - RAMP HOLD - PROFIBUS
   DR_2_CW_B6_RMP_IN_ZERO : BOOL ;	//TRAVEL DRIVE 2 CONTROL WORD BIT 6 - RAMP IN ZERO - PROFIBUS
   DR_2_CW_B7_FLT_RST : BOOL ;	//TRAVEL DRIVE 2 CONTROL WORD BIT 7 - FAULT RESET - PROFIBUS
   DR_2_CW_B8_INCH_1 : BOOL ;	//TRAVEL DRIVE 2 CONTROL WORD BIT 8 - INCHING 1 - PROFIBUS
   DR_2_CW_B9_INCH_2 : BOOL ;	//TRAVEL DRIVE 2 CONTROL WORD BIT 9 - INCHING 2 - PROFIBUS
   DR_2_CW_B10_RMT_CMD : BOOL ;	//TRAVEL DRIVE 2 CONTROL WORD BIT 10 - REMOTE COMMAND - PROFIBUS
   DR_2_CW_B11 : BOOL ;	//TRAVEL DRIVE 2 CONTROL WORD BIT 11 - DRIVE SPECIFIC - PROFOBUS
   DR_2_CW_B12 : BOOL ;	//TRAVEL DRIVE 2 CONTROL WORD BIT 12 - DRIVE SPECIFIC - PROFOBUS
   DR_2_CW_B13 : BOOL ;	//TRAVEL DRIVE 2 CONTROL WORD BIT 13 - DRIVE SPECIFIC - PROFOBUS
   DR_2_CW_B14 : BOOL ;	//TRAVEL DRIVE 2 CONTROL WORD BIT 14 - DRIVE SPECIFIC - PROFOBUS
   DR_2_CW_B15 : BOOL ;	//TRAVEL DRIVE 2 CONTROL WORD BIT 15 - DRIVE SPECIFIC - PROFOBUS
   DR_2_SW_B0_RDY_ON : BOOL ;	//TRAVEL DRIVE 2 STATUS WORD BIT 0 - READY TO OPERATE - OFF1 - PROFIBUS
   DR_2_SW_B1_RDY_TO_OPER : BOOL ;	//TRAVEL DRIVE 2 STATUS WORD BIT 1 - REDY TO OPERATE - PROFIBUS
   DR_2_SW_B2_REF_RDY : BOOL ;	//TRAVEL DRIVE 2 STATUS WORD BIT 2 - ENABEL OPERATION - PROFIBUS
   DR_2_SW_B3_TRIPPED : BOOL ;	//TRAVEL DRIVE 2 STATUS WORD BIT 3 - FAULT - PROFIBUS
   DR_2_SW_B4_OFF_2_STA : BOOL ;	//TRAVEL DRIVE 2 STATUS WORD BIT 4 - OFF 2 STATUS - PROFIBUS
   DR_2_SW_B5_OFF_3_STA : BOOL ;	//TRAVEL DRIVE 2 STATUS WORD BIT 5 - OFF 3 STATUS - PROFIBUS
   DR_2_SW_B6_SWC_ON_INHB : BOOL ;	//TRAVEL DRIVE 2 STATUS WORD BIT 6 - SWITCH ON INHIBIT - PROFIBUS
   DR_2_SW_B7_ALARM : BOOL ;	//TRAVEL DRIVE 2 STATUS WORD BIT 7 - WARNING/ALARM - PROFIBUS
   DR_2_SW_B8_AT_SETPOINT : BOOL ;	//TRAVEL DRIVE 2 STATUS WORD BIT 8 - OPERATING - PROFIBUS
   DR_2_SW_B9_REMOTE : BOOL ;	//TRAVEL DRIVE 2 STATUS WORD BIT 9 - DRIVE CONTROL REMOTE\LOCAL - PROFIBUS
   DR_2_SW_B10_ABOVE_LIMIT : BOOL ;	//TRAVEL DRIVE 2 STATUS WORD BIT 10 - SPEED ABOVE LIMIT - PROFIBUS
   DR_2_SW_B11 : BOOL ;	//TRAVEL DRIVE 2 STATUS WORD BIT 11 - DRIVE SPECIFIC - PROFOBUS
   DR_2_SW_B12 : BOOL ;	//TRAVEL DRIVE 2 STATUS WORD BIT 12 - DRIVE SPECIFIC - PROFOBUS
   DR_2_SW_B13 : BOOL ;	//TRAVEL DRIVE 2 STATUS WORD BIT 13 - DRIVE SPECIFIC - PROFOBUS
   DR_2_SW_B14 : BOOL ;	//TRAVEL DRIVE 2 STATUS WORD BIT 14 - DRIVE SPECIFIC - PROFOBUS
   DR_2_SW_B15 : BOOL ;	//TRAVEL DRIVE 2 STATUS WORD BIT 15 - DRIVE SPECIFIC - PROFOBUS
   DR_1_ACT_SPD_PF : REAL ;	//TRAVEL DRIVE 1 ACTUAL SPEED - PROFIBUS
   DR_1_ACT_SPD_SCL_ERR : WORD ;	//TRAVEL DRIVE 1 ACTUAL SPEED SCALING ERROR - PROFIBUS
   DR_2_ACT_SPD_PF : REAL ;	//TRAVEL DRIVE 2 ACTUAL SPEED - PROFIBUS
   DR_2_ACT_SPD_SCL_ERR : WORD ;	//TRAVEL DRIVE 2 ACTUAL SPEED SCALING ERROR - PROFIBUS
   LT_ALARM : BOOL ;	//LONG TRAVEL ALARM
   LT_SIREN : BOOL ;	//LONG TRAVEL SIREN
   TRA_DRV_1_FWD_CMD_PF : BOOL ;	//TRAVEL DRIVE 1 FORWARD COMMAND THROUGH PROFIBUS
   TRA_DRV_1_REV_CMD_PF : BOOL ;	//TRAVEL DRIVE 1 REVERSE COMMAND THROUGH PROFIBUS
   TRA_DRV_2_FWD_CMD_PF : BOOL ;	//TRAVEL DRIVE 2 FORWARD COMMAND THROUGH PROFIBUS
   TRA_DRV_2_REV_CMD_PF : BOOL ;	//TRAVEL DRIVE 2 REVERSE COMMAND THROUGH PROFIBUS
   TRA_ILK_BYPASS : BOOL ;	//TRAVEL INTERLOCK BYPASS INPUT
   TRA_FWD_CHNG_OVR_DEL : BOOL ;	//TRAVEL DRIVE FORWARD CHANGE OVER DELAY
   TRA_REV_CHNG_OVR_DEL : BOOL ;	//TRAVEL DRIVE REVERSE CHANGE OVER DELAY
  END_STRUCT ;	
BEGIN
END_DATA_BLOCK

DATA_BLOCK "AIR_COMPRESSOR_DB"	// DB 4
AUTHOR : Kamillas
VERSION : 0.1
  STRUCT
   AC_MTR_RDY_FOR_STA : BOOL ;	//AIR COMPRESSOR MOTOR READY FOR START
   AC_MTR_RUN_FB : BOOL ;	//AIR COMPRESSOR MOTOR RUN FEED BACK
   AC_MTR_OLR_TRIP_FB : BOOL ;	//AIR COMPRESSOR MOTOR TRIP FEED BACK
   AC_MTR_STA_PB : BOOL ;	//AIR COMPRESSOR MOTOR START PUSH BUTTON
   AC_MTR_STP_PB : BOOL ;	//AIR COMPRESSOR MOTOR STOP PUSH BUTTON
   AC_MTR_ON_CMD : BOOL ;	//AIR COMPRESSOR MOTOR ON COMMAND
   AC_MTR_ON_IND : BOOL ;	//AIR COMPRESSOR MOTOR ON INDICATOR
   AC_MTR_FLT : BOOL ;	//AIR COMPRESSOR MOTOR FAULT
   AC_MTR_FLT_TMR : INT ;	//AIR COMPRESSOR MOTOR FAULT TIMER
   AC_MTR_FLT_GEN_TIME : INT  := 3;	//AIR COMPRESSOR MOTOR FAULT GEMERATION TIME
   PULSE_1 : BOOL ;	//PULSE 1
   PULSE_2 : BOOL ;	//PULSE 2
   PULSE_3 : BOOL ;	//PULSE 3
   PULSE_4 : BOOL ;	//PULSE 4
   PULSE_5 : BOOL ;	//PULSE 5
   PULSE_6 : BOOL ;	//PULSE 6
   PULSE_7 : BOOL ;	//PULSE 7
   PULSE_8 : BOOL ;	//PULSE 8
   COMP_PRE_SW : BOOL ;	//COMPRESSOR PRESSURE SWITCH FEEDBACK
   AC_MTR_ON_CMD_WIT_PRE : BOOL ;	//AIR COMPRESSOR MOTOR ON COMMAND WITH PRESSURE SWITCH
  END_STRUCT ;	
BEGIN
   AC_MTR_FLT_GEN_TIME := 3;
END_DATA_BLOCK

DATA_BLOCK "HOOD_SYSTEM_DB"	// DB 5
AUTHOR : Kamillas
VERSION : 0.1
  STRUCT
   IDF_DRV_PROFI_HW_SS : BOOL ;	//ID FAN DRIVE PROFIBUS/HARDWIRE CONNECTION
   IDF_DRV_ON_FB : BOOL ;	//ID FAN DRIVE ON FEEDBACK
   IDF_DRV_RDY_FOR_STA : BOOL ;	//ID FAN DRIVE READY FOR START
   IDF_DRV_TRIP_FB : BOOL ;	//ID FAN DRIVE TRIP FEED BACK
   WTR_PMP_MTR_ON_FB : BOOL ;	//WATER PUMP MOTOR ON FEEDBACK
   WTR_PMP_MTR_RDY_FOR_STA : BOOL ;	//WATER PUMP MOTOR READY FOR START
   WTR_PMP_MTR_TRIP_FB : BOOL ;	//WATER PUMP MOTOR TRIP FEED BACK
   HOOD_STA_PB : BOOL ;	//HOOD START PUSH BUTTON
   HOOD_STP_PB : BOOL ;	//HOOD STOP PUSH BUTTON
   IDF_DRV_LS_HS_SEL : BOOL ;	//ID FAN DRIVE LOW SPEED/HIGH SPEED SELECTION
   WTR_LEV_LOW_LEV_SWH : BOOL ;	//WATER LEVEL LOW LEVEL SWITCH
   IDF_DRV_HIGH_SPD_CMD : BOOL ;	//ID FAN DRIVE HIGH SPEED COMMAND
   IDF_DRV_LOW_SPD_CMD : BOOL ;	//ID FAN DRIVE LOW SPEED COMMAND
   IDF_DRV_REV_ON_CMD : BOOL ;	//ID FAN DRIVE REVERSE ON COMMADN COMMAND
   WTR_PMP_MTR_ON_CMD : BOOL ;	//WATER PUMP MOTOR ON COMMAND
   HOOD_ON_IND : BOOL ;	//HOOD ON INDICATOR
   IDF_DRV_STATUS_WORD_1 : INT ;	//ID FAN PROFIBUS STATUS WORD 1
   IDF_DRV_STATUS_WORD_2 : INT ;	//ID FAN PROFIBUS STATUS WORD 2
   IDF_DRV_STATUS_WORD_3 : INT ;	//ID FAN PROFIBUS STATUS WORD 3
   IDF_DRV_STATUS_WORD_4 : INT ;	//ID FAN PROFIBUS STATUS WORD 4
   IDF_DRV_STATUS_WORD_5 : INT ;	//ID FAN PROFIBUS STATUS WORD 5
   IDF_DRV_STATUS_WORD_6 : INT ;	//ID FAN PROFIBUS STATUS WORD 6
   IDF_DRV_STATUS_WORD_7 : INT ;	//ID FAN PROFIBUS STATUS WORD 7
   IDF_DRV_STATUS_WORD_8 : INT ;	//ID FAN PROFIBUS STATUS WORD 8
   IDF_DRV_STATUS_WORD_9 : INT ;	//ID FAN PROFIBUS STATUS WORD 9
   IDF_DRV_STATUS_WORD_10 : INT ;	//ID FAN PROFIBUS STATUS WORD 10
   IDF_DRV_STATUS_WORD_11 : INT ;	//ID FAN PROFIBUS STATUS WORD 11
   IDF_DRV_STATUS_WORD_12 : INT ;	//ID FAN PROFIBUS STATUS WORD 12
   IDF_DRV_STATUS_WORD_13 : INT ;	//ID FAN PROFIBUS STATUS WORD 13
   IDF_DRV_STATUS_WORD_14 : INT ;	//ID FAN PROFIBUS STATUS WORD 14
   IDF_DRV_STATUS_WORD_15 : INT ;	//ID FAN PROFIBUS STATUS WORD 15
   IDF_DRV_STATUS_WORD_16 : INT ;	//ID FAN PROFIBUS STATUS WORD 16
   IDF_DRV_CONTROL_WORD_1 : INT ;	//ID FAN PROFIBUS CONTROL WORD 1
   IDF_DRV_CONTROL_WORD_2 : INT ;	//ID FAN PROFIBUS CONTROL WORD 2
   IDF_DRV_CONTROL_WORD_3 : INT ;	//ID FAN PROFIBUS CONTROL WORD 3
   IDF_DRV_CONTROL_WORD_4 : INT ;	//ID FAN PROFIBUS CONTROL WORD 4
   IDF_DRV_CONTROL_WORD_5 : INT ;	//ID FAN PROFIBUS CONTROL WORD 5
   IDF_DRV_CONTROL_WORD_6 : INT ;	//ID FAN PROFIBUS CONTROL WORD 6
   IDF_DRV_CONTROL_WORD_7 : INT ;	//ID FAN PROFIBUS CONTROL WORD 7
   IDF_DRV_CONTROL_WORD_8 : INT ;	//ID FAN PROFIBUS CONTROL WORD 8
   IDF_DRV_CONTROL_WORD_9 : INT ;	//ID FAN PROFIBUS CONTROL WORD 9
   IDF_DRV_CONTROL_WORD_10 : INT ;	//ID FAN PROFIBUS CONTROL WORD 10
   IDF_DRV_CONTROL_WORD_11 : INT ;	//ID FAN PROFIBUS CONTROL WORD 11
   IDF_DRV_CONTROL_WORD_12 : INT ;	//ID FAN PROFIBUS CONTROL WORD 12
   IDF_DRV_CONTROL_WORD_13 : INT ;	//ID FAN PROFIBUS CONTROL WORD 13
   IDF_DRV_CONTROL_WORD_14 : INT ;	//ID FAN PROFIBUS CONTROL WORD 14
   IDF_DRV_CONTROL_WORD_15 : INT ;	//ID FAN PROFIBUS CONTROL WORD 15
   IDF_DRV_CONTROL_WORD_16 : INT ;	//ID FAN PROFIBUS CONTROL WORD 16
   IDF_DRV_STAT_WORD_1_E : INT ;	//ID FAN DRIVE STATUS WORD 1 READ ERROR
   IDF_DRV_STAT_WORD_2_E : INT ;	//ID FAN DRIVE STATUS WORD 2 READ ERROR
   IDF_DRV_STAT_WORD_3_E : INT ;	//ID FAN DRIVE STATUS WORD 3 READ ERROR
   IDF_DRV_STAT_WORD_4_E : INT ;	//ID FAN DRIVE STATUS WORD 4 READ ERROR
   IDF_DRV_CTRL_WORD_1_E : INT ;	//ID FAN DRIVE CONTROL WORD 1 WRITE ERROR
   IDF_DRV_CTRL_WORD_2_E : INT ;	//ID FAN DRIVE CONTROL WORD 2 WRITE ERROR
   IDF_DRV_CTRL_WORD_3_E : INT ;	//ID FAN DRIVE CONTROL WORD 3 WRITE ERROR
   IDF_DRV_CTRL_WORD_4_E : INT ;	//ID FAN DRIVE CONTROL WORD 4 WRITE ERROR
   IDF_DRV_RDY_TO_OPER_P : BOOL ;	//ID FAN DRIVE READY TO OPERATE BIT - PROFIBUS
   IDF_DRV_ENAB_OPER_PF : BOOL ;	//ID FAN DRIVE ENABLE OPERATIONS - PROFIBUS
   IDF_DRV_FLT_PF : BOOL ;	//ID FAN DRIVE FAULT - PROFIBUS
   IDF_DRV_SPD_FB_PF : REAL ;	//ID FAN DRIVE SPEED FEED BACK FROM DRIVE - PROFIBUS
   IDF_SPD_REF_DI_PF : DINT ;	//ID FAN SPEED REFERENCE IN DOUBLE INTEGER - PROFIBUS
   IDF_SPD_REF_NEG_RMD_P : INT ;	//ID FAN SPEED REFERENCE CONVERTERD TO POSITIVE VALUE - PROFIBUS
   IDF_SPD_REF_REAL_PF : REAL ;	//ID FAN SPEED REFERENCE IN REAL(FLOATING POINT) - PROFIBUS
   IDF_SPD_REF_UN_SL_FLT : WORD ;	//ID FAN SPEED REFERENCE UNSCALLING FAULT - PROFIBUS
   PULSE_1 : BOOL ;	//PULSE 1
   PULSE_2 : BOOL ;	//PULSE 2
   PULSE_3 : BOOL ;	//PULSE 3
   PULSE_4 : BOOL ;	//PULSE 4
   PULSE_5 : BOOL ;	//PULSE 5
   PULSE_6 : BOOL ;	//PULSE 6
   PULSE_7 : BOOL ;	//PULSE 7
   PULSE_8 : BOOL ;	//PULSE 8
   HOOD_SYS_ILK : BOOL ;	//HOOD SYSTEM INTERLOCK
   IDF_DRV_FLT : BOOL ;	//ID FAN DRIVE FAULT
   IDF_DRV_FLT_TMR : INT ;	//ID FAN DRIVE FAULT TIMER
   IDF_DRV_FLT_GEN_TIME : INT  := 3;	//IF FAN DRIVE FAULT GEMERATION TIME
   WTR_PMP_FLT : BOOL ;	//WATER PUMP MOTOR FAULT
   WTR_PMP_FLT_TMR : INT ;	//WATER PUMP FAULT TIMER
   WTR_PMP_FLT_GEN_TIME : INT  := 3;	//WATER PUMP FAULT GEMERATION TIME
   IDF_DRV_LOW_SPD_OVR : BOOL ;	//ID FAN DRIVE LOW SPEED OVER
   IDF_DRV_LOW_SPD_TMR : INT ;	//ID FAN DRIVE LOW SPEED TIMER
   IDF_DRV_LOW_SPD_OVR_TIME : INT  := 3;	//IF FAN DRIVE LOW SPEED OVER GENERATION TIME
   HOOD_SYS_IN_REPAIR_MAN : BOOL ;	//HOOD SYSTEM IN REPAIR AND MANUAL MODE
   HOOD_SYS_IN_AUTO : BOOL ;	//HOOD SYSTEM IN AUTO MODE
   HIGH_SPEED_SEL_IN_R_M : BOOL ;	//HIGH SPEED SELECTION IN REPAIR AND MANUAL
   ID_FAN_HS_CMD : BOOL ;	//ID FAN HIGH SPEED COMMAND
   ID_FAN_LS_CMD : BOOL ;	//ID FAN LOW SPEED COMMAND
   PULSE_10 : BOOL ;	//ID FAN LOW SPEED RESET NEG EDGE
  END_STRUCT ;	
BEGIN
   IDF_DRV_FLT_GEN_TIME := 3;
   WTR_PMP_FLT_GEN_TIME := 3;
   IDF_DRV_LOW_SPD_OVR_TIME := 3;
END_DATA_BLOCK

DATA_BLOCK "DOOR_EXTRACTOR_DB"	// DB 6
AUTHOR : Kamillas
VERSION : 0.1
  STRUCT
   DOOR_EXT_LOC_SS : BOOL ;	//DOOR EXTRACTOR LOCAL SELECTOR SWITCH
   DOOR_EXT_MAN_SS : BOOL ;	//DOOR EXTRACTOR MANUAL SELECTOR SWITCH
   DOOR_EXT_AUTO_SS : BOOL ;	//DOOR EXTRACTOR AUTO SELECTOR SWITCH
   DOOR_EXT_STP_PB : BOOL ;	//DOOR EXTRACTOR STOP PUSH BUTTON
   SLEW_FWD_STA_PB : BOOL ;	//SLEW FORWARD START PUSH BUTTON
   SLEW_RET_STA_PB : BOOL ;	//SLEW RETRACT START
   VER_COMP_FWD_STA_PB : BOOL ;	//VERTICAL COMPENSATION FORWARD START PUSH BUTTON
   VER_COMP_RET_STA_PB : BOOL ;	//VERTICAL COMPENSATION RETRACT START PUSH BUTTON
   TRA_FWD_STA_PB : BOOL ;	//TRAVEL FORWARD START PUSH BUTTON
   TRA_RET_STA_PB : BOOL ;	//TRAVEL RETRACT START PUSH BUTTON
   MAIN_STK_UP_STA_PB : BOOL ;	//MAIN STROKE UP START PUSH BUTTON
   MAIN_STK_UP_DN_PB : BOOL ;	//MAIN STROKE DOWN START PUSH BUTTON
   FIN_STK_UP_STA_PB : BOOL ;	//FINAL STROKE UP START PUSH BUTTON
   FIN_STK_DN_PB : BOOL ;	//FINAL STROKE DOWN START PUSH BUTTON
   PRE_STK_UP_STA_PB : BOOL ;	//PRE STROKE UP START PUSH BUTTON
   PRE_STK_DN_PB : BOOL ;	//PRE STROKE DOWN START PUSH BUTTON
   DR_SPNG_LK_STA_PB : BOOL ;	//DOOR SPRING PRESSURE START PUSH BUTTON
   DR_SPNG_UNLK_STA_PB : BOOL ;	//DOOR SPRING PRESSURE RELEASE START PUSH BUTTON
   DR_LCH_TURN_UP_PB : BOOL ;	//DOOR LATCH TURNING LOCK PUSH BUTTON
   DR_LCH_TURN_DN_PB : BOOL ;	//DOOR LATCH TURNING UNLOCK PUSH BUTTON
   EMERGENCY_PB_LCS_73 : BOOL ;	//EMERGENCY PUSHBUTTON LCS-73
   SLEW_FWD_STA_PB_LCS : BOOL ;	//SLEW FORWARD START PUSH BUTTON LCS
   SLEW_RET_STA_PB_LCS : BOOL ;	//SLEW RETRACT START PUSHBUTTON LCS
   VER_COMP_FWD_STA_PB_LCS : BOOL ;	//VERTICAL COMPENSATION FORWARD START LCS PUSH BUTTON
   VER_COMP_RET_STA_PB_LCS : BOOL ;	//VERTICAL COMPENSATION RETRACT START LCS PUSH BUTTON
   TRA_FWD_STA_PB_LCS : BOOL ;	//TRAVEL FORWARD START LCS  PUSH BUTTON
   TRA_RET_STA_PB_LCS : BOOL ;	//TRAVEL BACK START LCS  PUSH BUTTON
   MAIN_STK_UP_STA_PB_LCS : BOOL ;	//MAIN STROKE UP START LCS PUSH BUTTON
   MAIN_STK_DN_STA_PB_LCS : BOOL ;	//MAIN STROKE DN START LCS PUSH BUTTON
   FIN_STK_UP_STA_PB_LCS : BOOL ;	//FINAL STROKE UP START LCS  PUSH BUTTON
   FIN_STK_DN_STA_PB_LCS : BOOL ;	//FINAL STROKE DOWN START LCS PUSH BUTTON
   PRE_STK_UP_STA_PB_LCS : BOOL ;	//PREE STROKE UP START LCS PUSH BUTTON
   PRE_STK_DN_STA_PB_LCS : BOOL ;	//PREE STROKE DN START LCS PUSH BUTTON
   DR_SPNG_LK_STA_PB_LCS : BOOL ;	//DOOR SPRING LOCK START PUSH BUTTON LCS
   DR_SPNG_UNLK_STA_PB_LCS : BOOL ;	//DOOR SPRING UNLOCK  START PUSH BUTTON LCS
   LAMP_TEST_PB_LCS_73 : BOOL ;	//LAMP TEST PUSHBUTTON LCS-73
   DR_LCH_TURN_UP_PB_LCS : BOOL ;	//DOOR LATCH LOCK PUSH BUTTON LCS
   DR_LCH_TURN_DN_PB_LCS : BOOL ;	//DOOR LATCH UNLOCK PUSH BUTTON LCS
   DR_LCH_TURN_HOME_PB_LCS : BOOL ;	//DOOR LATCH HOME PUSH BUTTON LCS
   SLEW_SLOW_FWD_LS : BOOL ;	//SLEW SLOW FORWARD LIMIT SWITCH
   SLEW_SLOW_RET_LS : BOOL ;	//SLEW SLOW RETRACT LIMIT SWITCH
   SLEW_NOR_FWD_LS : BOOL ;	//SLEW NORMAL FORWARD LIMIT SWITCH
   SLEW_NOR_RET_LS : BOOL ;	//SLEW NORMAL RETRACT LIMIT SWITCH
   TRA_SLOW_FWD_LS : BOOL ;	//TRAVEL SLOW FORWARD LIMIT  SWITCH
   TRA_SLOW_RET_LS : BOOL ;	//TRAVEL SLOW RETRACT LIMIT  SWITCH
   TRA_FWD_LS : BOOL ;	//TRAVEL FORWARD LIMIT SWIITCH
   TRA_RET_LS : BOOL ;	//TRAVEL RETRACT LIMIT SWIITCH
   FOR_LS_TRAVEL : BOOL ;	//FORWARD LIMIT SWITCH TRAVEL
   DOOR_ON_HOOK_LS : BOOL ;	//DOOR ON HOOK LIMITSWTCH
   DOOR_FIX_LOC_FB_PR_SWT : BOOL ;	//DOOR FIX LOCKED FEEDBACK PRESSURE SWITCH
   DR_LCH_TURN_UP_LS : BOOL ;	//DOOR LATCH TURNING UP LIMIT SWICH
   DR_LCH_TURN_DN_LS : BOOL ;	//DOOR LATCH TURNING DOWN LIMIT SWICH
   SPRING_PRESS : BOOL ;	//SPRING PRESS
   SLEW_SLOW_FWD_CMD : BOOL ;	//SLEW SLOW FORWARD COMMAND
   SLEW_SLOW_RET_CMD : BOOL ;	//SLEW SLOW RETRACT COMMAND
   SLEW_NOR_FWD_COMMAND : BOOL ;	//SLEW NORMAL FORWARD COMMAND
   SLEW_NOR_RET_COMMAND : BOOL ;	//SLEW NORMAL RETRACT COMMAND
   VER_COMP_FWD_CMD : BOOL ;	//VERTICAL COMPENSATION FORWARD COMMAND
   VER_COMP_RET_CMD : BOOL ;	//VERTICAL COMPENSATION RETRACT COMMAND
   VER_COMP_RELIVE_CMD : BOOL ;	//VERTICAL COMPENSTAION RELIVE  COOMMAND
   TRA_SLOW_FWD_CMD : BOOL ;	//TRAVEL SLOW FORWARD COMMAND
   TRA_SLOW_RET_CMD : BOOL ;	//TRAVEL SLOW RETRACT COMMAND
   TRA_NOR_FWD_CMD : BOOL ;	//TRAVEL NORMAL FORWARD COMMAND
   TRA_NOR_RET_CMD : BOOL ;	//TRAVEL NORMAL RETRACT COMMAND
   TRA_RELIVE_CMD : BOOL ;	//TRAVEL RELIVE COOMMAND
   MAIN_STK_UP_CMD : BOOL ;	//MANUAL STROKE UP COMMAND
   MAIN_STK_DN_CMD : BOOL ;	//MANUAL STROKE DN COMMAND
   PRE_STK_UP_CMD : BOOL ;	//PRE STROKE UP COMMAND
   PRE_STK_DN_CMD : BOOL ;	//PRE STROKE DN COMMAND
   DR_SPNG_LK_CMD : BOOL ;	//DOOR SPRING PRESS LOCK COMMAND
   DR_SPNG_UNLK_CMD : BOOL ;	//DOOR SPRING PRESS UNLOCK COMMAND
   DR_LCH_TURN_UP_CMD : BOOL ;	//DOOR LATCH TURNING UP COMMAND
   DR_LCH_TURN_DN_CMD : BOOL ;	//DOOR LATCH TURNING DOWN COMMADN
   SLEW_SLOW_FWD_IND : BOOL ;	//SLEW SLOW FORWARD INDICATOR
   SLEW_SLOW_RET_IND : BOOL ;	//SLEW SLOW RETRACT INDICATOR
   VER_COMP_FWD_IND : BOOL ;	//VERTICAL COMPENSATION FORWARD INDICATOR
   VER_COMP_RET_IND : BOOL ;	//VERTICAL COMPENSATION RETRACT INDICATOR
   TRA_FWD_IND : BOOL ;	//TRAVEL FORWARD INDICATOR
   TRA_RET_IND : BOOL ;	//TRAVEL BACK INDICATOR
   MAIN_STK_UP_IND : BOOL ;	//FINAL STROKE  UP INDICATION
   MAIN_STK_DN_IND : BOOL ;	//FINAL STROKE  DOWN  INDICATOR
   FIN_STK_UP_IND : BOOL ;	//FINAL STROKE  UP INDICATOR
   FIN_STK_DN_IND : BOOL ;	//FINAL STROKE  DOWN INDICATOR
   PRE_STK_UP_IND : BOOL ;	//PRE STROKE  UP INDICATION
   PRE_STK_DN_IND : BOOL ;	//PRE STROKE  DOWN INDICATOR
   DR_SPNG_LK_IND : BOOL ;	//DOOR SPRING PRESS LOCK INDICATOR
   DR_SPNG_UNLK_IND : BOOL ;	//DOOR SPRING PRESS UNLOCK INDICATOR
   DOOR_FIX_LOCK_IND : BOOL ;	//DOOR FIX LOCK INDICATOR
   DOOR_FIX_UNLK_IND : BOOL ;	//DOOR FIX UNLOCK INDICATOR
   DOOR_FIX_UNLK_IND1 : BOOL ;	//DOOR FIX UNLOCK INDICATOR
   LCS_73_ON_IND : BOOL ;	//LCS-73_ON_INDICATOR
   SLEW_SLOW_FWD_IND_LCS : BOOL ;	//SLEW SLOW FORWARD INDICATOR LCS
   SLEW_SLOW_RET_IND_LCS : BOOL ;	//SLEW SLOW RETRACT INDICATOR LCS
   VER_COMP_FWD_IND_LCS : BOOL ;	//VERTICAL COMPENSATION FORWARD INDICATOR LCS
   VER_COMP_RET_IND_LCS : BOOL ;	//VERTICAL COMPENSATION RETRACT INDICATOR LCS
   TRA_FWD_IND_LCS : BOOL ;	//TRAVEL FORWARD INDICATOR
   TRA_RET_IND_LCS : BOOL ;	//TRAVEL BACK INDICATOR LCS
   MAIN_STK_UP_IND_LCS : BOOL ;	//FINAL STROKE UP INDICATION LCS
   MAIN_STK_DN_IND_LCS : BOOL ;	//FINAL STROKE DOWN  INDICATOR LCS
   FIN_STK_UP_IND_LCS : BOOL ;	//FINAL STROKE UP INDICATOR LCS
   FIN_STK_DN_IND_LCS : BOOL ;	//FINAL STROKE DOWN INDICATOR LCS
   PRE_STK_UP_IND_LCS : BOOL ;	//PRE STROKE UP INDICATION LCS
   PRE_STK_DN_IND_LCS : BOOL ;	//PRE STROKE DOWN INDICATOR LCS
   DR_LCH_TURN_HOME_IND_LCS : BOOL ;	//DOOR LATCH HOME INDICATION LCS
   DR_LCH_TURN_UP_IND_LCS : BOOL ;	//DOOR LATCH TURNING UP INDICATOR LCS
   DR_LCH_TURN_DN_IND_LCS : BOOL ;	//DOOR LATCH TURNING DOWN INDICATOR LCS
   DOOR_FIX_LOCK_IND_LCS : BOOL ;	//DOOR FIX LOCK INDICATOR LCS
   DOOR_FIX_UNLK_IND_LCS : BOOL ;	//DOOR FIX UNLOCK INDICATOR LCS
   SLEW_SL_FWD_OP_CUT : BOOL ;	//SLEW SLOW FORWARD OUTPUT CUT
   SLEW_SL_FWD_FLT_TMR : INT ;	//SLEW SLOW FORWARD FAULT TIMER
   SLEW_SL_FWD_FLT_GEN : INT  := 8;	//SLEW SLOW FORWARD FAULT GENERATION TIME
   SLEW_SL_FWD_OP_CT_TM : INT ;	//SLEW SLOW FORWARD OUTPUT CUT TIMER
   SLEW_SL_FWD_FLT : BOOL ;	//SLEW SLOW FORWARD FAULT
   SLEW_SL_AUTO_FWD_OVR : BOOL ;	//SLEW SLOW AUTO FORWARD OVER
   SLEW_SL_AUTO_FWD_DEL : INT  := 3;	//SLEW SLOW AUTO FORWARD OVER DELAY
   SLEW_SL_ATO_FWD_DL_T : INT ;	//SLEW SLOW AUTO FORWARD OVER DELAY TIMER
   SLEW_NR_FWD_OP_CUT : BOOL ;	//SLEW NORMAL FORWARD OUTPUT CUT
   SLEW_NR_FWD_FLT_TMR : INT ;	//SLEW NORMAL FORWARD FAULT TIMER
   SLEW_NR_FWD_FLT_GEN : INT  := 8;	//SLEW NORMAL FORWARD FAULT GENERATION TIME
   SLEW_NR_FWD_OP_CT_TM : INT ;	//SLEW NORMAL FORWARD OUTPUT CUT TIMER
   SLEW_NR_FWD_FLT : BOOL ;	//SLEW NORMAL FORWARD FAULT
   SLEW_NR_AUTO_FWD_OVR : BOOL ;	//SLEW NORMAL AUTO FORWARD OVER
   SLEW_NR_AUTO_FWD_DEL : INT  := 3;	//SLEW NORMAL AUTO FORWARD OVER DELAY
   SLEW_NR_ATO_FWD_DL_T : INT ;	//SLEW NORMAL AUTO FORWARD OVER DELAY TIMER
   PULSE_1 : BOOL ;	//PULSE 1
   PULSE_2 : BOOL ;	//PULSE 2
   PULSE_3 : BOOL ;	//PULSE 3
   PULSE_4 : BOOL ;	//PULSE 4
   PULSE_5 : BOOL ;	//PULSE 5
   PULSE_6 : BOOL ;	//PULSE 6
   PULSE_7 : BOOL ;	//PULSE 7
   PULSE_8 : BOOL ;	//PULSE 8
   PULSE_9 : BOOL ;	//PULSE 9
   PULSE_10 : BOOL ;	//PULSE 10
   PULSE_11 : BOOL ;	//PULSE 11
   PULSE_12 : BOOL ;	//PULSE 12
   PULSE_13 : BOOL ;	//PULSE 13
   PULSE_14 : BOOL ;	//PULSE 14
   PULSE_15 : BOOL ;	//PULSE 15
   PULSE_16 : BOOL ;	//PULSE 16
   SLEW_NR_RET_OP_CUT : BOOL ;	//SLEW NORMAL RETRACT OUTPUT CUT
   SLEW_NR_RET_FLT_TMR : INT ;	//SLEW NORMAL RETRACT FAULT TIMER
   SLEW_NR_RET_FLT_GEN : INT  := 8;	//SLEW NORMAL RETRACT FAULT GENERATION TIME
   SLEW_NR_RET_OP_CT_TM : INT ;	//SLEW NORMAL RETRACT RETRACT OUTPUT CUT TIMER
   SLEW_NR_RET_FLT : BOOL ;	//SLEW NORMAL RETRACT RETRACT FAULT
   SLEW_NR_AUTO_RET_OVR : BOOL ;	//SLEW NORMAL AUTO RETRACT OVER
   SLEW_NR_AUTO_RET_DEL : INT  := 3;	//SLEW NORMAL AUTO RETRACT OVER DELAY
   SLEW_NR_ATO_RET_DL_T : INT ;	//SLEW NORMAL AUTO RETRACT OVER DELAY TIMER
   VER_COMP_FWD_OP_CUT : BOOL ;	//VERTICAL COMPENSATION FORWARD OUTPUT CUT
   VER_COMP_FWD_FLT_TMR : INT ;	//VERTICAL COMPENSATION FORWARD FAULT TIMER
   VER_COMP_FWD_FLT_GEN : INT  := 8;	//VERTICAL COMPENSATION FORWARD FAULT GENERATION TIME
   VER_COMP_FWD_OP_CT_TM : INT ;	//VERTICAL COMPENSATION FORWARD OUTPUT CUT TIMER
   VER_COMP_FWD_FLT : BOOL ;	//VERTICAL COMPENSATION FORWARD FAULT
   VER_COMP_AUTO_FWD_OVR : BOOL ;	//VERTICAL COMPENSATION AUTO FORWARD OVER
   VER_COMP_AUTO_FWD_DEL : INT  := 3;	//VERTICAL COMPENSATION AUTO FORWARD OVER DELAY
   VER_COMP_ATO_FWD_DL_T : INT ;	//VERTICAL COMPENSATION AUTO FORWARD OVER DELAY TIMER
   VER_COMP_RET_OP_CUT : BOOL ;	//VERTICAL COMPENSATION RETRACT OUTPUT CUT
   VER_COMP_RET_FLT_TMR : INT ;	//VERTICAL COMPENSATION RETRACT FAULT TIMER
   VER_COMP_RET_FLT_GEN : INT  := 8;	//VERTICAL COMPENSATION RETRACT FAULT GENERATION TIME
   VER_COMP_RET_OP_CT_TM : INT ;	//VERTICAL COMPENSATION RETRACT OUTPUT CUT TIMER
   VER_COMP_RET_FLT : BOOL ;	//VERTICAL COMPENSATION RETRACT FAULT
   VER_COMP_AUTO_RET_OVR : BOOL ;	//VERTICAL COMPENSATION AUTO RETRACT OVER
   VER_COMP_AUTO_RET_DEL : INT  := 3;	//VERTICAL COMPENSATION AUTO RETRACT OVER DELAY
   VER_COMP_ATO_RET_DL_T : INT ;	//VERTICAL COMPENSATION AUTO RETRACT OVER DELAY TIMER
   TRA_SLOW_FWD_OP_CUT : BOOL ;	//TRAVEL SLOW FORWARD OUTPUT CUT
   TRA_SLOW_FWD_FLT_TMR : INT ;	//TRAVEL SLOW FORWARD FAULT TIMER
   TRA_SLOW_FWD_FLT_GEN : INT  := 8;	//TRAVEL SLOW FORWARD FAULT GENERATION TIME
   TRA_SLOW_FWD_OP_CT_TM : INT ;	//TRAVEL SLOW FORWARD OUTPUT CUT TIMER
   TRA_SLOW_FWD_FLT : BOOL ;	//TRAVEL SLOW FORWARD FAULT
   TRA_SLOW_AUTO_FWD_OVR : BOOL ;	//TRAVEL SLOW AUTO FORWARD OVER
   TRA_SLOW_AUTO_FWD_DEL : INT  := 3;	//TRAVEL SLOW AUTO FORWARD OVER DELAY
   TRA_SLOW_ATO_FWD_DL_T : INT ;	//TRAVEL SLOW AUTO FORWARD OVER DELAY TIMER
   TRA_SLOW_RET_OP_CUT : BOOL ;	//TRAVEL SLOW RETRACT OUTPUT CUT
   TRA_SLOW_RET_FLT_TMR : INT ;	//TRAVEL SLOW RETRACT FAULT TIMER
   TRA_SLOW_RET_FLT_GEN : INT  := 8;	//TRAVEL SLOW RETRACT FAULT GENERATION TIME
   TRA_SLOW_RET_OP_CT_TM : INT ;	//TRAVEL SLOW RETRACT OUTPUT CUT TIMER
   TRA_SLOW_RET_FLT : BOOL ;	//TRAVEL SLOW RETRACT FAULT
   TRA_SLOW_AUTO_RET_OVR : BOOL ;	//TRAVEL SLOW AUTO RETRACT OVER
   TRA_SLOW_AUTO_RET_DEL : INT  := 3;	//TRAVEL SLOW AUTO RETRACT OVER DELAY
   TRA_SLOW_ATO_RET_DL_T : INT ;	//TRAVEL SLOW AUTO RETRACT OVER DELAY TIMER
   TRA_NOR_FWD_OP_CUT : BOOL ;	//TRAVEL NORMAL FORWARD OUTPUT CUT
   TRA_NOR_FWD_FLT_TMR : INT ;	//TRAVEL NORMAL FORWARD FAULT TIMER
   TRA_NOR_FWD_FLT_GEN : INT  := 8;	//TRAVEL NORMAL FORWARD FAULT GENERATION TIME
   TRA_NOR_FWD_OP_CT_TM : INT ;	//TRAVEL NORMAL FORWARD OUTPUT CUT TIMER
   TRA_NOR_FWD_FLT : BOOL ;	//TRAVEL NORMAL FORWARD FAULT
   TRA_NOR_AUTO_FWD_OVR : BOOL ;	//TRAVEL NORMAL AUTO FORWARD OVER
   TRA_NOR_AUTO_FWD_DEL : INT  := 3;	//TRAVEL NORMAL AUTO FORWARD OVER DELAY
   TRA_NOR_ATO_FWD_DL_T : INT ;	//TRAVEL NORMAL AUTO FORWARD OVER DELAY TIMER
   TRA_NOR_RET_OP_CUT : BOOL ;	//TRAVEL NORMAL RETRACT OUTPUT CUT
   TRA_NOR_RET_FLT_TMR : INT ;	//TRAVEL NORMAL RETRACT FAULT TIMER
   TRA_NOR_RET_FLT_GEN : INT  := 8;	//TRAVEL NORMAL RETRACT FAULT GENERATION TIME
   TRA_NOR_RET_OP_CT_TM : INT ;	//TRAVEL NORMAL RETRACT OUTPUT CUT TIMER
   TRA_NOR_RET_FLT : BOOL ;	//TRAVEL NORMAL RETRACT FAULT
   TRA_NOR_AUTO_RET_OVR : BOOL ;	//TRAVEL NORMAL AUTO RETRACT OVER
   TRA_NOR_AUTO_RET_DEL : INT  := 3;	//TRAVEL NORMAL AUTO RETRACT OVER DELAY
   TRA_NOR_ATO_RET_DL_T : INT ;	//TRAVEL NORMAL AUTO RETRACT OVER DELAY TIMER
   MAIN_STK_UP_OP_CUT : BOOL ;	//MAIN STROK UP OUTPUT CUT
   MAIN_STK_UP_FLT_TMR : INT ;	//MAIN STROK UP FAULT TIMER
   MAIN_STK_UP_FLT_GEN : INT  := 8;	//MAIN STROK UP FAULT GENERATION TIME
   MAIN_STK_UP_OP_CT_TM : INT ;	//MAIN STROK UP OUTPUT CUT TIMER
   MAIN_STK_UP_FLT : BOOL ;	//MAIN STROK UP FAULT
   MAIN_STK_AUTO_UP_OVR : BOOL ;	//MAIN STROK AUTO UP OVER
   MAIN_STK_AUTO_UP_DEL : INT  := 3;	//MAIN STROK AUTO UP OVER DELAY
   MAIN_STK_ATO_UP_DL_T : INT ;	//MAIN STROK AUTO UP OVER DELAY TIMER
   MAIN_STK_DN_OP_CUT : BOOL ;	//MAIN STROK DOWN OUTPUT CUT
   MAIN_STK_DN_FLT_TMR : INT ;	//MAIN STROK DOWN FAULT TIMER
   MAIN_STK_DN_FLT_GEN : INT  := 8;	//MAIN STROK DOWN FAULT GENERATION TIME
   MAIN_STK_DN_OP_CT_TM : INT ;	//MAIN STROK DOWN OUTPUT CUT TIMER
   MAIN_STK_DN_FLT : BOOL ;	//MAIN STROK DOWN FAULT
   MAIN_STK_AUTO_DN_OVR : BOOL ;	//MAIN STROK AUTO DOWN OVER
   MAIN_STK_AUTO_DN_DEL : INT  := 3;	//MAIN STROK AUTO DOWN OVER DELAY
   MAIN_STK_ATO_DN_DL_T : INT ;	//MAIN STROK AUTO DOWN OVER DELAY TIMER
   PRE_STK_UP_OP_CUT : BOOL ;	//PRE STROK UP OUTPUT CUT
   PRE_STK_UP_FLT_TMR : INT ;	//PRE STROK UP FAULT TIMER
   PRE_STK_UP_FLT_GEN : INT  := 8;	//PRE STROK UP FAULT GENERATION TIME
   PRE_STK_UP_OP_CT_TM : INT ;	//PRE STROK UP OUTPUT CUT TIMER
   PRE_STK_UP_FLT : BOOL ;	//PRE STROK UP FAULT
   PRE_STK_AUTO_UP_OVR : BOOL ;	//PRE STROK AUTO UP OVER
   PRE_STK_AUTO_UP_DEL : INT  := 3;	//PRE STROK AUTO UP OVER DELAY
   PRE_STK_ATO_UP_DL_T : INT ;	//PRE STROK AUTO UP OVER DELAY TIMER
   PRE_STK_DN_OP_CUT : BOOL ;	//PRE STROK DOWN OUTPUT CUT
   PRE_STK_DN_FLT_TMR : INT ;	//PRE STROK DOWN FAULT TIMER
   PRE_STK_DN_FLT_GEN : INT  := 8;	//PRE STROK DOWN FAULT GENERATION TIME
   PRE_STK_DN_OP_CT_TM : INT ;	//PRE STROK DOWN OUTPUT CUT TIMER
   PRE_STK_DN_FLT : BOOL ;	//PRE STROK DOWN FAULT
   PRE_STK_AUTO_DN_OVR : BOOL ;	//PRE STROK AUTO DOWN OVER
   PRE_STK_AUTO_DN_DEL : INT  := 3;	//PRE STROK AUTO DOWN OVER DELAY
   PRE_STK_ATO_DN_DL_T : INT ;	//PRE STROK AUTO DOWN OVER DELAY TIMER
   FIN_STK_UP_OP_CUT : BOOL ;	//FINAL STROK UP OUTPUT CUT
   FIN_STK_UP_FLT_TMR : INT ;	//FINAL STROK UP FAULT TIMER
   FIN_STK_UP_FLT_GEN : INT  := 8;	//FINAL STROK UP FAULT GENERATION TIME
   FIN_STK_UP_OP_CT_TM : INT ;	//FINAL STROK UP OUTPUT CUT TIMER
   FIN_STK_UP_FLT : BOOL ;	//FINAL STROK UP FAULT
   FIN_STK_AUTO_UP_OVR : BOOL ;	//FINAL STROK AUTO UP OVER
   FIN_STK_AUTO_UP_DEL : INT  := 3;	//FINAL STROK AUTO UP OVER DELAY
   FIN_STK_ATO_UP_DL_T : INT ;	//FINAL STROK AUTO UP OVER DELAY TIMER
   FIN_STK_DN_OP_CUT : BOOL ;	//FINAL STROK DOWN OUTPUT CUT
   FIN_STK_DN_FLT_TMR : INT ;	//FINAL STROK DOWN FAULT TIMER
   FIN_STK_DN_FLT_GEN : INT  := 8;	//FINAL STROK DOWN FAULT GENERATION TIME
   FIN_STK_DN_OP_CT_TM : INT ;	//FINAL STROK DOWN OUTPUT CUT TIMER
   FIN_STK_DN_FLT : BOOL ;	//FINAL STROK DOWN FAULT
   FIN_STK_AUTO_DN_OVR : BOOL ;	//FINAL STROK AUTO DOWN OVER
   FIN_STK_AUTO_DN_DEL : INT  := 3;	//FINAL STROK AUTO DOWN OVER DELAY
   FIN_STK_ATO_DN_DL_T : INT ;	//FINAL STROK AUTO DOWN OVER DELAY TIMER
   FIN_STK_UP_CMD : BOOL ;	//FINAL STROKE UP COMMAND
   FIN_STK_DN_CMD : BOOL ;	//FINAL STROKE DOWN COMMAND
   DR_SPNG_LK_OP_CUT : BOOL ;	//DOOR SPRING PRESSURE LOCK OUTPUT CUT
   DR_SPNG_LK_FLT_TMR : INT ;	//DOOR SPRING PRESSURE LOCK FAULT TIMER
   DR_SPNG_LK_FLT_GEN : INT  := 8;	//DOOR SPRING PRESSURE LOCK FAULT GENERATION TIME
   DR_SPNG_LK_OP_CT_TM : INT ;	//DOOR SPRING PRESSURE LOCK OUTPUT CUT TIMER
   DR_SPNG_LK_FLT : BOOL ;	//DOOR SPRING PRESSURE LOCK FAULT
   DR_SPNG_AUTO_LK_OVR : BOOL ;	//DOOR SPRING AUTO PRESSURE LOCK OVER
   DR_SPNG_AUTO_LK_DEL : INT  := 3;	//DOOR SPRING AUTO PRESSURE LOCK OVER DELAY
   DR_SPNG_ATO_LK_DL_T : INT ;	//DOOR SPRING AUTO PRESSURE LOCK OVER DELAY TIMER
   DR_SPNG_UNLK_OP_CUT : BOOL ;	//DOOR SPRING PRESSURE UNLOCK OUTPUT CUT
   DR_SPNG_UNLK_FLT_TMR : INT ;	//DOOR SPRING PRESSURE UNLOCK FAULT TIMER
   DR_SPNG_UNLK_FLT_GEN : INT  := 8;	//DOOR SPRING PRESSURE UNLOCK FAULT GENERATION TIME
   DR_SPNG_UNLK_OP_CT_TM : INT ;	//DOOR SPRING PRESSURE UNLOCK OUTPUT CUT TIMER
   DR_SPNG_UNLK_FLT : BOOL ;	//DOOR SPRING PRESSURE UNLOCK FAULT
   DR_SPNG_AUTO_UNLK_OVR : BOOL ;	//DOOR SPRING AUTO PRESSURE UNLOCK OVER
   DR_SPNG_AUTO_UNLK_DEL : INT  := 3;	//DOOR SPRING AUTO PRESSURE UNLOCK OVER DELAY
   DR_SPNG_ATO_UNLK_DL_T : INT ;	//DOOR SPRING AUTO PRESSURE UNLOCK OVER DELAY TIMER
   PULSE_17 : BOOL ;	//PULSE 17
   PULSE_18 : BOOL ;	//PULSE 18
   PULSE_19 : BOOL ;	//PULSE 19
   PULSE_20 : BOOL ;	//PULSE 20
   PULSE_21 : BOOL ;	//PULSE 21
   PULSE_22 : BOOL ;	//PULSE 22
   PULSE_23 : BOOL ;	//PULSE 23
   PULSE_24 : BOOL ;	//PULSE 24
   PULSE_25 : BOOL ;	//PULSE 25
   PULSE_26 : BOOL ;	//PULSE 26
   PULSE_27 : BOOL ;	//PULSE 27
   PULSE_28 : BOOL ;	//PULSE 28
   PULSE_29 : BOOL ;	//PULSE 29
   PULSE_30 : BOOL ;	//PULSE 30
   DR_LCH_UP_OP_CUT : BOOL ;	//DOOR LATCH UP OUTPUT CUT
   DR_LCH_UP_FLT_TMR : INT ;	//DOOR LATCH UP FAULT TIMER
   DR_LCH_UP_FLT_GEN : INT  := 8;	//DOOR LATCH UP FAULT GENERATION TIME
   DR_LCH_UP_OP_CT_TM : INT ;	//DOOR LATCH UP OUTPUT CUT TIMER
   DR_LCH_UP_FLT : BOOL ;	//DOOR LATCH UP FAULT
   DR_LCH_AUTO_UP_OVR : BOOL ;	//DOOR LATCH AUTO PRESSURE UP OVER
   DR_LCH_AUTO_UP_DEL : INT  := 3;	//DOOR LATCH AUTO PRESSURE UP OVER DELAY
   DR_LCH_ATO_UP_DL_T : INT ;	//DOOR LATCH AUTO PRESSURE UP OVER DELAY TIMER
   DR_LCH_DN_OP_CUT : BOOL ;	//DOOR LATCH DOWN OUTPUT CUT
   DR_LCH_DN_FLT_TMR : INT ;	//DOOR LATCH DOWN FAULT TIMER
   DR_LCH_DN_FLT_GEN : INT  := 8;	//DOOR LATCH DOWN FAULT GENERATION TIME
   DR_LCH_DN_OP_CT_TM : INT ;	//DOOR LATCH DOWN OUTPUT CUT TIMER
   DR_LCH_DN_FLT : BOOL ;	//DOOR LATCH DOWN FAULT
   DR_LCH_AUTO_DN_OVR : BOOL ;	//DOOR SPRING AUTO PRESSURE DOWN OVER
   DR_LCH_AUTO_DN_DEL : INT  := 3;	//DOOR SPRING AUTO PRESSURE DOWN OVER DELAY
   DR_LCH_ATO_DN_DL_T : INT ;	//DOOR SPRING AUTO PRESSURE DOWN OVER DELAY TIMER
   TRA_SLOW_FWD_IND : BOOL ;	//TRAVEL SLOW FORWARD INDICATOR
   TRA_SLOW_RET_IND : BOOL ;	//TRAVEL SLOW RETRACT INDICATOR
   TRA_SLOW_FWD_IND_LCS : BOOL ;	//TRAVEL SLOW FORWARD INDICATOR LCS
   TRA_SLOW_RET_IND_LCS : BOOL ;	//TRAVEL RETRACT INDICATOR LCS
   SLEW_FWD_IND : BOOL ;	//SLEW NORMAL FORWARD INDICATOR
   SLEW_RET_IND : BOOL ;	//SLEW NORMAL RETRACT INDICATOR
   SLEW_FWD_IND_LCS : BOOL ;	//SLEW NORMAL FORWARD INDICATOR LCS
   SLEW_RET_IND_LCS : BOOL ;	//SLEW NORMAL RETRACT INDICATOR LCS
   DR_SPNG_LK_IND_LCS : BOOL ;	//DOOR SPRING PRESS LOCK INDICATOR LCS
   DR_SPNG_UNLK_IND_LCS : BOOL ;	//DOOR SPRING PRESS UNLOCK INDICATOR LCS
   DE_TRA_SLOW_FWD_BIT : BOOL ;	//DOOR EXTRACTOR TRAVEL SLOW FORWARD START BIT
   DOR_EXT_RPL_ILK_BIT : BOOL ;	//DOOR EXTRACTOR/REPLACE INTERLOCK BIT
   DR_EXT_AUTO_STA_BIT : BOOL ;	//DOOR EXTRACTOR AUTO START BIT
   EXT_OVEN_DOR_AUTO_STA_PB : BOOL ;	//EXTRACT OVEN DOOR AUTO START PUSH BUTTON
   DR_EXT_RPL_AUTO_STP_PB : BOOL ;	//DOOR EXTRACTOR/REPLACE AUTO STOP PUSH BUTTON
   RPL_OVEN_DOR_AUTO_STA_PB : BOOL ;	//REPLACE OVEN DOOR AUTO START PUSH BUTTON
   VER_COMP_LDT_SCLD_VLU : REAL ;	//VERTICAL COMPENSATION LDT SCALED VALUE
   VER_COMP_LDT_SLNG_ERR : WORD ;	//VERTICAL COMPENSATION LDT SCALING ERROR
   DR_RPL_AUTO_STA_BIT : BOOL ;	//DOOR REPLACE AUTO START BIT
   PULSE_31 : BOOL ;	//PULSE 31
   PULSE_32 : BOOL ;	//PULSE 32
   PULSE_33 : BOOL ;	//PULSE 33
   PULSE_34 : BOOL ;	//PULSE 34
   PULSE_35 : BOOL ;	//PULSE 35
   PULSE_36 : BOOL ;	//PULSE 36
   PULSE_37 : BOOL ;	//PULSE 37
   PULSE_38 : BOOL ;	//PULSE 38
   PULSE_39 : BOOL ;	//PULSE 39
   PULSE_40 : BOOL ;	//PULSE 40
   PULSE_41 : BOOL ;	//PULSE 41
   PULSE_42 : BOOL ;	//PULSE 42
   PULSE_43 : BOOL ;	//PULSE 43
   PULSE_44 : BOOL ;	//PULSE 44
   PULSE_45 : BOOL ;	//PULSE 45
   PULSE_46 : BOOL ;	//PULSE 46
   PULSE_47 : BOOL ;	//PULSE 47
   PULSE_48 : BOOL ;	//PULSE 48
   PULSE_49 : BOOL ;	//PULSE 49
   PULSE_50 : BOOL ;	//PULSE 50
   PRE_STK_UP_LR : BOOL ;	//PRE STROKE UP LIMIT READHED
   PRE_STK_DN_LR : BOOL ;	//PRE STROKE DOWN LIMIT READHED
   MAIN_STK_FWD_LR : BOOL ;	//MAIN STROKE UP LIMIT READHED
   MAIN_STK_DN_LR : BOOL ;	//MAIN STROKE DOWN LIMIT READHED
   FIN_STK_FWD_LR : BOOL ;	//FINAL STROKE UP LIMIT READHED
   FIN_STK_DN_LR : BOOL ;	//FINAL STROKE DOWN LIMIT READHED
   EXT_OVEN_DOR_IND : BOOL ;	//EEXTRACT OVEN DOOR INDICATOR
   RPL_OVEN_DOR_IND : BOOL ;	//REPLACE OVEN DOOR INDICATOR
   SLEW_AUTO_FWD_SET : BOOL ;	//SLWE AUTO FORWARD SET
   SLEW_AUTO_RET_SET : BOOL ;	//SLWE AUTO RETRACT SET
   VER_COMP_AUTO_FWD_SET : BOOL ;	//VERTICAL COMPENSATION AUTO FORWARD SET
   VER_COMP_AUTO_RET_SET : BOOL ;	//VERTICAL COMPENSATION AUTO RETRACT SET
   TRA_AUTO_FWD_SET : BOOL ;	//TRAVEL AUTO FORWARD SET
   TRA_AUTO_RET_SET : BOOL ;	//TRAVEL AUTO RETRACT SET
   PRE_STK_AUTO_FWD_SET : BOOL ;	//PRE STROK AUTO FORWARD SET
   PRE_STK_AUTO_RET_SET : BOOL ;	//PRE STROK AUTO RETRACT SET
   MAIN_STK_AUTO_FWD_SET : BOOL ;	//MAIN STROK AUTO FORWARD SET
   MAIN_STK_AUTO_RET_SET : BOOL ;	//MAIN STROK AUTO RETRACT SET
   FIN_STK_AUTO_FWD_SET : BOOL ;	//FINAL STROK AUTO FORWARD SET
   FIN_STK_AUTO_RET_SET : BOOL ;	//FINAL STROK AUTO RETRACT SET
   DR_SPNG_AUTO_PRSD_SET : BOOL ;	//DOOR SPING AUTO PRESSED SET
   DR_SRNG_AUTO_RLSD_SET : BOOL ;	//DOOR SPING AUTO RELESED SET
   DR_LCH_TURN_AUTO_UP_SET : BOOL ;	//DOOR LATCH TURN AUTO UP BIT
   DR_LCH_TURN_AUTO_DN_SET : BOOL ;	//DOOR LATCH TURN AUTO DOWN BIT
   DR_LFT_LDT_SCLD_VLU : REAL ;	//DOOR LIFTING LDT SCALED VALUE
   DR_LFT_LDT_SLNG_ERR : WORD ;	//DOOR LIFTING LDT SCALING ERROR
   VER_COMP_VALUE : REAL ;	//VERTICAL COMPENSATION VALUE
   VER_COMP_LDT_REAL : REAL ;	//VERTICAL COMPENSATION LDT REAL VALUE
   DR_LFT_LDT_REAL : REAL ;	//DOOR LIFTING LDT REAL VALUE
   VER_COMP_UNSCLD_VLU : INT ;	//VERTICAL COMPENSATION UNSCALED VALUE
   DR_LFT_UNSCLD_VLU : INT ;	//DOOR LIFTER UNSCALED VALUE
   PRE_STK_UP_LDT_VLU : REAL ;	//PRE STROKE UP LDT VALUE
   MAIN_STK_UP_LDT_VLU : REAL ;	//MAIN STROKE UP LDT VALUE
   FIN_STK_UP_LDT_VLU : REAL ;	//FIN STROKE UP LDT VALUE
   PRE_STK_DN_LDT_VLU : REAL ;	//PRE STROKE DOWN LDT VALUE
   MAIN_STK_DN_LDT_VLU : REAL ;	//MAIN STROKE DOWN LDT VALUE
   FIN_STK_DN_LDT_VLU : REAL ;	//FIN STROKE DOWN LDT VALUE
   VER_COMP_FWD_LIM_VALUE : REAL ;	//VERTICAL COMPENSATION FORWARD LIMIT VALUE
   DOOR_FIX_REL_FB : BOOL ;	//DOOR RELEASE FEEDBACK
   DR_LCH_TURN_UP_IND : BOOL ;	//DOOR LATCH LOCK INDICATOR CD
   DR_LCH_TURN_DN_IND : BOOL ;	//DOOR LATCH UNLOCK INDICATOR CD
   VER_COMP_LR : BOOL ;	//VERTICAL COMPENSATION LIMIT REACHED
   DR_EXTR_HME_POS : BOOL ;	//DOOR EXTRACTOR HOME POSITION REACHED
   DR_EXT_AUTO_OPER_FIN : BOOL ;	//DOOR EXTRACTOR AUTO OPERATIONS FINISHED
   DR_RPL_AUTO_OPER_FIN : BOOL ;	//DOOR REPLACE AUTO OPERATIONS FINISHED
   TRA_RELEVE_VLV : BOOL ;	//TRAVEL RELEVE VALVE
   VER_COMP_RELEVE_VLV : BOOL ;	//VERTICAL COMPENSATION RELEVE VALVE
   SLEW_SL_RET_OP_CUT : BOOL ;	//SLEW SLOW RETRACT OUTPUT CUT
   SLEW_SL_RET_FLT_TMR : INT ;	//SLEW SLOW RETRACT FAULT TIMER
   SLEW_SL_RET_FLT_GEN : INT  := 8;	//SLEW SLOW RETRACT FAULT GENERATION TIME
   SLEW_SL_RET_OP_CT_TM : INT ;	//SLEW SLOW RETRACT OUTPUT CUT TIMER
   SLEW_SL_RET_FLT : BOOL ;	//SLEW SLOW RETRACT FAULT
   SLEW_SL_AUTO_RET_OVR : BOOL ;	//SLEW SLOW AUTO RETRACT OVER
   SLEW_SL_AUTO_RET_DEL : INT  := 3;	//SLEW SLOW AUTO RETRACT OVER DELAY
   SLEW_SL_ATO_RET_DL_T : INT ;	//SLEW SLOW AUTO RETRACT OVER DELAY TIMER
   SLEW_SL_RET_SET_BIT : BOOL ;	//SLEW SLOW RETRACT BIT
   VER_COMP_FWD_BYPASS : BOOL ;	//VERTICAL COMPENSATION FORWARD BYPASS BIT
   VER_COMP_REV_BYPASS : BOOL ;	//VERTICAL COMPENSATION REVERSE BYPASS BIT
   LDT_TMR_SS : BOOL ;	//LDT OR TIMER SELECTOR SWITCH
   PRE_STK_UP_TIM_OP_CUT : BOOL ;	//PRE STROKE UP TIMER OPERATION COMPLETE
   PRE_STK_DN_TIM_OP_CUT : BOOL ;	//PRE STROKE DOWN TIMER OPERATION COMPLETE
   MAIN_STK_UP_TIM_OP_CUT : BOOL ;	//MAIN STROKE UP TIMER OPERATION COMPLETE
   MAIN_STK_DN_TIM_OP_CUT : BOOL ;	//MAIN STROKE DOWN TIMER OPERATION COMPLETE
   FIN_STK_UP_TIM_OP_CUT : BOOL ;	//FINAL STROKE UP TIMER OPERATION COMPLETE
   FIN_STK_DN_TIM_OP_CUT : BOOL ;	//FINAL STROKE DOWN TIMER OPERATION COMPLETE
   VER_COMP_LDT_TMR_SS : BOOL ;	//VERTICAL COMPENSATION LDT TIMER SELECTOR
   VER_COMP_TMR_FWD_OP_CUT : BOOL ;	//VERTICAL COMPENSATION FORWARD TIMER SET
   VER_COMP_TMR_RET_OP_CUT : BOOL ;	//VERTICAL COMPENSATION RETRACT TIMER SET
  END_STRUCT ;	
BEGIN
   SLEW_SL_FWD_FLT_GEN := 8;
   SLEW_SL_AUTO_FWD_DEL := 3;
   SLEW_NR_FWD_FLT_GEN := 8;
   SLEW_NR_AUTO_FWD_DEL := 3;
   SLEW_NR_RET_FLT_GEN := 8;
   SLEW_NR_AUTO_RET_DEL := 3;
   VER_COMP_FWD_FLT_GEN := 8;
   VER_COMP_AUTO_FWD_DEL := 3;
   VER_COMP_RET_FLT_GEN := 8;
   VER_COMP_AUTO_RET_DEL := 3;
   TRA_SLOW_FWD_FLT_GEN := 8;
   TRA_SLOW_AUTO_FWD_DEL := 3;
   TRA_SLOW_RET_FLT_GEN := 8;
   TRA_SLOW_AUTO_RET_DEL := 3;
   TRA_NOR_FWD_FLT_GEN := 8;
   TRA_NOR_AUTO_FWD_DEL := 3;
   TRA_NOR_RET_FLT_GEN := 8;
   TRA_NOR_AUTO_RET_DEL := 3;
   MAIN_STK_UP_FLT_GEN := 8;
   MAIN_STK_AUTO_UP_DEL := 3;
   MAIN_STK_DN_FLT_GEN := 8;
   MAIN_STK_AUTO_DN_DEL := 3;
   PRE_STK_UP_FLT_GEN := 8;
   PRE_STK_AUTO_UP_DEL := 3;
   PRE_STK_DN_FLT_GEN := 8;
   PRE_STK_AUTO_DN_DEL := 3;
   FIN_STK_UP_FLT_GEN := 8;
   FIN_STK_AUTO_UP_DEL := 3;
   FIN_STK_DN_FLT_GEN := 8;
   FIN_STK_AUTO_DN_DEL := 3;
   DR_SPNG_LK_FLT_GEN := 8;
   DR_SPNG_AUTO_LK_DEL := 3;
   DR_SPNG_UNLK_FLT_GEN := 8;
   DR_SPNG_AUTO_UNLK_DEL := 3;
   DR_LCH_UP_FLT_GEN := 8;
   DR_LCH_AUTO_UP_DEL := 3;
   DR_LCH_DN_FLT_GEN := 8;
   DR_LCH_AUTO_DN_DEL := 3;
   SLEW_SL_RET_FLT_GEN := 8;
   SLEW_SL_AUTO_RET_DEL := 3;
END_DATA_BLOCK

DATA_BLOCK "SERVICE_PLATFORM_DB"	// DB 7
AUTHOR : Kamillas
VERSION : 0.1
  STRUCT
   SP_TRA_FWD_STA_PB : BOOL ;	//SERVICE PLATFORM TRAVEL FORWARD START PUSH BUTTON
   SP_TRA_REV_STA_PB : BOOL ;	//SERVICE PLATFORM TRAVEL REVERSE START PUSH BUTTON
   SP_TRA_FWD_STA_PB_LCS : BOOL ;	//SERVICE PLATFORM TRAVEL FORWARD START PUSH BUTTON LCS
   SP_TRA_REV_STA_PB_LCS : BOOL ;	//SERVICE PLATFORM TRAVEL REVERSE START PUSH BUTTON LCS
   SP_TRA_FWD_LS : BOOL ;	//SERVICE PLATFORM TRAVEL FORWARD LIMIT SWITCH
   SP_TRA_REV_LS : BOOL ;	//SERVICE PLATFORM TRAVEL REVERSE LIMIT SWITCH
   SP_TRA_FWD_CMD : BOOL ;	//SERVICE PLATFORM TRAVEL FORWARD COMMAND
   SP_TRA_REV_CMD : BOOL ;	//SERVICE PLATFORM TRAVEL REVERSE COMMAND
   SP_TRA_FWD_IND : BOOL ;	//SERVICE PLATFORM TRAVEL FORWARD INDICATOR
   SP_TRA_REV_IND : BOOL ;	//SERVICE PLATFORM TRAVEL REVERSE INDICATOR
   SP_TRA_FWD_IND_LCS : BOOL ;	//SERVICE PLATFORM TRAVEL FORWARD INDICATOR LCS
   SP_TRA_REV_IND_LCS : BOOL ;	//SERVICE PLATFORM TRAVEL REVERSE INDICATOR LCS
   SP_TRA_FWD_OP_CUT : BOOL ;	//SERVICE PLATFORM TRAVEL FORWARD OUTPUT CUT
   SP_TRA_FWD_OP_CUT_TMR : INT ;	//SERVICE PLATFORM TRAVEL FORWARD OUTPUT CUT TIMER
   SP_TRA_AUTO_FWD_OVR : BOOL ;	//SERVICE PLATFORM TRAVEL AUTO FORWARD OVER
   SP_TRA_AUTO_FWD_DEL : INT  := 3;	//SERVICE PLATFORM TRAVEL AUTO FORWARD OVER DELAY
   SP_TRA_AUTO_FWD_DEL_TMR : INT ;	//SERVICE PLATFORM TRAVEL AUTO FORWARD OVER DELAY TIMER
   SP_TRA_AUTO_FWD_SET : BOOL ;	//SERVICE PLATFORM AUTO FORWARD SET
   SP_TRA_RET_OP_CUT : BOOL ;	//SERVICE PLATFORM TRAVEL RETRACT OUTPUT CUT
   SP_TRA_RET_OP_CUT_TMR : INT ;	//SERVICE PLATFORM TRAVEL RETRACT OUTPUT CUT TIMER
   SP_TRA_AUTO_RET_OVR : BOOL ;	//SERVICE PLATFORM TRAVEL AUTO RETRACT OVER
   SP_TRA_AUTO_RET_DEL : INT  := 3;	//SERVICE PLATFORM TRAVEL AUTO RETRACT OVER DELAY
   SP_TRA_AUTO_RET_DEL_TMR : INT ;	//SERVICE PLATFORM TRAVEL AUTO RETRACT OVER DELAY TIMER
   SP_TRA_AUTO_RET_SET : BOOL ;	//SERVICE PLATFORM AUTO RETRACT SET
   SP_ILK_BIT : BOOL ;	//SERVICE PLATFORM INTERLOCK BIT
   PULSE_1 : BOOL ;	//PULSE 1
   PULSE_2 : BOOL ;	//PULSE 2
   PULSE_3 : BOOL ;	//PULSE 3
   PULSE_4 : BOOL ;	//PULSE 4
   PULSE_5 : BOOL ;	//PULSE 5
   PULSE_6 : BOOL ;	//PULSE 6
   PULSE_7 : BOOL ;	//PULSE 7
   PULSE_8 : BOOL ;	//PULSE 8
   SP_AUTO_SS : BOOL ;	//SERVICE PLATFORM AUTO MODE SELECTOR SWITCH
   SP_MAN_SS : BOOL ;	//SERVICE PLATFORM MANUAL MODE SELECTOR SWITCH
   SP_LOC_SS : BOOL ;	//SERVICE PLATFORM LOCAL MODE SELECTOR SWITCH
   SP_AUTO_STA_PB : BOOL ;	//SERVICE PLATFORM AUTO START PUSH BUTTON
   SP_STP_PB : BOOL ;	//SERVICE PLATFORM STOP PUSH BUTTON
   SP_HME_POS_BIT : BOOL ;	//SERVICE PLATFORM HOME POSITION BIT
   SP_AUTO_STA_BIT : BOOL ;	//SERVICE PLATFORM AUTO START BIT
   SP_AUTO_STP_PB : BOOL ;	//SERVICE PLATFORM AUTO STOP PUSH BUTTON
   SP_AUTO_IND : BOOL ;	//SERVICE PLATFORM AUTO PROCESS INDICATOR
  END_STRUCT ;	
BEGIN
   SP_TRA_AUTO_FWD_DEL := 3;
   SP_TRA_AUTO_RET_DEL := 3;
END_DATA_BLOCK

DATA_BLOCK "JAMB_CLEANER_DB"	// DB 8
AUTHOR : Kamillas
VERSION : 0.1
  STRUCT
   JC_CAR_TRA_FWD_LS : BOOL ;	//JAMB CLEANER CARRIAGE TRAVEL FORWARD LIMIT SWITCH
   JC_CAR_TRA_RET_LS : BOOL ;	//JAMB CLEANER CARRIAGE TRAVEL RETRACT LIMIT SWITCH
   JC_VER_CLNR_UP_LS : BOOL ;	//JAMB CLEANER VERTICAL CLEANER UP LIMIT SWITCH
   JC_VER_CLNR_DN_LS : BOOL ;	//JAMB CLEANER VERTICAL CLEANER DOWN LIMIT SWITCH
   JC_VER_CLNR_HME_LS : BOOL ;	//JAMB CLEANER VERTICAL CLEANER HOME LIMIT SWITCH
   JC_CRA_TRA_FWD_STA_PB : BOOL ;	//JAMB CLEANER CARRIAGE TRAVEL FORWARD PUSH BUTTON
   JC_CRA_TRA_RET_STA_PB : BOOL ;	//JAMB CLEANER CARRIAGE TRAVEL RETRACT PUSH BUTTON
   JC_VC_UP_STA_PB : BOOL ;	//JAMB CLEANER VERTICAL CLEANER UP START PUSH BUTTON
   JC_VC_DN_STA_PB : BOOL ;	//JAMB CLEANER VERTICAL CLEANER DOWN START PUSH BUTTON
   JC_STP_PB : BOOL ;	//JAMB CLEANER OPERATIONS STOP PUSH BUTTON
   JC_VC_HME_STA_PB : BOOL ;	//JAMB CLEANER VERTICAL CLEANER HOME START PUSH BUTTON
   JC_CAR_TRA_FWD_CMD : BOOL ;	//JAMB CLEANER CARRIAGE TRAVEL FORWARD COMMAND
   JC_CAR_TRA_RET_CMD : BOOL ;	//JAMB CLEANER CARRIAGE TRAVEL RETRACT COMMAND
   JC_VC_UP_CMD : BOOL ;	//JAMB CLEANER VERTICAL CLEANER UP COMMAND
   JC_VC_DN_CMD : BOOL ;	//JAMB CLEANER VERTICAL CLEANER DOWN COMMAND
   JC_CAR_TRA_FWD_IND : BOOL ;	//JAMB CLEANER CARRIAGE TRAVEL FORWARD INDICATOR
   JC_CAR_TRA_RET_IND : BOOL ;	//JAMB CLEANER CARRIAGE TRAVEL RETRACT INDICATOR
   JC_VC_UP_IND : BOOL ;	//JAMB CLEANER VERTICAL CLEANER UP INDICATOR
   JC_VC_DN_IND : BOOL ;	//JAMB CLEANER VERTICAL CLEANER DOWN INDICATOR
   JC_VC_HME_IND : BOOL ;	//JAMB CLEANER VERTICAL CLEANER HOME INDIATOR
   CLN_OVN_JMB_STA_PB : BOOL ;	//CLEAN OVEN JAMB AUTO START PUSH BUTTON
   CLN_OVN_JMB_STP_PB : BOOL ;	//CLEAN OVEN JAMB AUTO STOP PUSH BUTTON
   CLN_OVN_JMB_IND : BOOL ;	//CLEAN OVEN JAMB AUTO INDICATOR
   JC_TRA_FWD_OP_CUT : BOOL ;	//JAMB CLEANER TRAVEL FORWARD OUTPUT CUT
   JC_TRA_FWD_OP_CUT_TMR : INT ;	//JAMB CLEANER TRAVEL FORWARD OUTPUT CUT TIMER
   JC_TRA_AUTO_FWD_OVR : BOOL ;	//JAMB CLEANER TRAVEL AUTO FORWARD OVER
   JC_TRA_AUTO_FWD_DEL : INT  := 3;	//JAMB CLEANER TRAVEL AUTO FORWARD OVER DELAY
   JC_TRA_AUTO_FWD_DEL_TMR : INT ;	//JAMB CLEANER TRAVEL AUTO FORWARD OVER DELAY TIMER
   JC_TRA_AUTO_FWD_SET : BOOL ;	//JAMB CLEANER AUTO TRAVEL FORWARD SET
   JC_TRA_RET_OP_CUT : BOOL ;	//JAMB CLEANER TRAVEL RETRACT OUTPUT CUT
   JC_TRA_RET_OP_CUT_TMR : INT ;	//JAMB CLEANER TRAVEL RETRACT OUTPUT CUT TIMER
   JC_TRA_AUTO_RET_OVR : BOOL ;	//JAMB CLEANER TRAVEL AUTO RETRACT OVER
   JC_TRA_AUTO_RET_DEL : INT  := 3;	//JAMB CLEANER TRAVEL AUTO RETRACT OVER DELAY
   JC_TRA_AUTO_RET_DEL_TMR : INT ;	//JAMB CLEANER TRAVEL AUTO RETRACT OVER DELAY TIMER
   JC_TRA_AUTO_RET_SET : BOOL ;	//JAMB CLEANER AUTO TRAVEL RETRACT SET
   JC_VC_FWD_OP_CUT : BOOL ;	//JAMB CLEANER VERTICAL CLEANER FORWARD OUTPUT CUT
   JC_VC_FWD_OP_CUT_TMR : INT ;	//JAMB CLEANER VERTICAL CLEANER FORWARD OUTPUT CUT TIMER
   JC_VC_AUTO_FWD_OVR : BOOL ;	//JAMB CLEANER VERTICAL CLEANER AUTO FORWARD OVER
   JC_VC_AUTO_FWD_DEL : INT  := 3;	//JAMB CLEANER VERTICAL CLEANER AUTO FORWARD OVER DELAY
   JC_VC_AUTO_FWD_DEL_TMR : INT ;	//JAMB CLEANER VERTICAL CLEANER AUTO FORWARD OVER DELAY TIMER
   JC_VC_AUTO_FWD_SET : BOOL ;	//JAMB CLEANER AUTO VERTICAL CLEANER FORWARD SET
   JC_VC_RET_OP_CUT : BOOL ;	//JAMB CLEANER VERTICAL CLEANER RETRACT OUTPUT CUT
   JC_VC_RET_OP_CUT_TMR : INT ;	//JAMB CLEANER VERTICAL CLEANER RETRACT OUTPUT CUT TIMER
   JC_VC_AUTO_RET_OVR : BOOL ;	//JAMB CLEANER VERTICAL CLEANER AUTO RETRACT OVER
   JC_VC_AUTO_RET_DEL : INT  := 3;	//JAMB CLEANER VERTICAL CLEANER AUTO RETRACT OVER DELAY
   JC_VC_AUTO_RET_DEL_TMR : INT ;	//JAMB CLEANER VERTICAL CLEANER AUTO RETRACT OVER DELAY TIMER
   JC_VC_AUTO_RET_SET : BOOL ;	//JAMB CLEANER AUTO VERTICAL CLEANER RETRACT SET
   JC_AUTO_SS : BOOL ;	//JAMB CLEANER AUTO MODE SELECTOR SWITCH
   JC_MAN_SS : BOOL ;	//JAMB CLEANER MANUAL MODE SELECTOR SWITCH
   JC_LOC_SS : BOOL ;	//JAMB CLEANER LOCAL MODE SELECTOR SWITCH
   JC_AUTO_STA_PB : BOOL ;	//JAMB CLEANER AUTO START PUSH BUTTON
   JC_ILK_BIT : BOOL ;	//JAMB CLEANER INTERLOCK BIT
   PULSE_1 : BOOL ;	//PULSE 1
   PULSE_2 : BOOL ;	//PULSE 2
   PULSE_3 : BOOL ;	//PULSE 3
   PULSE_4 : BOOL ;	//PULSE 4
   PULSE_5 : BOOL ;	//PULSE 5
   PULSE_6 : BOOL ;	//PULSE 6
   PULSE_7 : BOOL ;	//PULSE 7
   PULSE_8 : BOOL ;	//PULSE 8
   PULSE_9 : BOOL ;	//PULSE 9
   PULSE_10 : BOOL ;	//PULSE 10
   PULSE_11 : BOOL ;	//PULSE 11
   PULSE_12 : BOOL ;	//PULSE 12
   PULSE_13 : BOOL ;	//PULSE 13
   PULSE_14 : BOOL ;	//PULSE 14
   PULSE_15 : BOOL ;	//PULSE 15
   PULSE_16 : BOOL ;	//PULSE 16
   JC_HME_POS_BIT : BOOL ;	//JAMB CLEANER HOME POSITION BIT
   JC_VC_HME_OP_CUT : BOOL ;	//JAMB CLEANER VERTICAL CLEANER HOME OUTPUT CUT
   JC_VC_HME_OP_CUT_TMR : INT ;	//JAMB CLEANER VERTICAL CLEANER HOME OUTPUT CUT TIMER
   JC_VC_AUTO_HME_OVR : BOOL ;	//JAMB CLEANER VERTICAL CLEANER AUTO HOME OVER
   JC_VC_AUTO_HME_DEL : INT  := 3;	//JAMB CLEANER VERTICAL CLEANER AUTO HOME OVER DELAY
   JC_VC_AUTO_HME_DEL_TMR : INT ;	//JAMB CLEANER VERTICAL CLEANER AUTO HOME OVER DELAY TIMER
   JC_VC_AUTO_HME_SET : BOOL ;	//JAMB CLEANER AUTO VERTICAL CLEANER HOME SET
   JC_VC_HME_CMD : BOOL ;	//JAMB CLEANER AUTO VERTICAL CLEANER HOME COMMADN
   JC_AUTO_STA : BOOL ;	//JAMB CLEANER AUTO START BIT
   JC_CLN_OVN_JAMB_IND : BOOL ;	//CLEAN OVEN JAMB INDICATOR
   JC_CLN_OVN_JAMB_FIN : BOOL ;	//CLEAN OVEN JAMB FINISHED BIT
   JC_UP_DN_CNT : INT ;	//JAMB CLEANER UP/DOWN COUNT
   JC_UP_DN_CNT_SET : INT  := 3;	//JAMB CLEANER UP/DOWN COUNT SET POINT
   JC_UP_DN_CNT_OVR : BOOL ;	//JAMB CLEANER UP/DOWN COUNT OVER
  END_STRUCT ;	
BEGIN
   JC_TRA_AUTO_FWD_DEL := 3;
   JC_TRA_AUTO_RET_DEL := 3;
   JC_VC_AUTO_FWD_DEL := 3;
   JC_VC_AUTO_RET_DEL := 3;
   JC_VC_AUTO_HME_DEL := 3;
   JC_UP_DN_CNT_SET := 2;
END_DATA_BLOCK

DATA_BLOCK "GUIDE_CAGE_DB"	// DB 9
AUTHOR : Kamillas
VERSION : 0.1
  STRUCT
   GC_TRA_FWD_LS : BOOL ;	//GUIDE CAGE TRAVEL FORWARD LIMIT SWITCH
   GC_TRA_RET_LS : BOOL ;	//GUIDE CAGE TRAVEL RETRACT LIMIT SWITCH
   GC_AUTO_SS : BOOL ;	//GUIDE CAGE AUTO SELECTOR SWITCH
   GC_MAN_SS : BOOL ;	//GUIDE CAGE MANUAL SELECTOR SWITCH
   GC_TRA_FWD_STA_PB : BOOL ;	//GUIDE CAGE TRAVEL FORWARD START PUSH BUTTON
   GC_TRA_RET_STA_PB : BOOL ;	//GUIDE CAGE TRAVEL RETRACT START PUSH BUTTON
   GC_STP_PB : BOOL ;	//GUIDE CAGE AUTO STOP PUSH BUTTON
   GC_TRA_AUTO_STA_PB : BOOL ;	//GUIDE CAGE TRAVEL AUTO START PUSH BUTTON
   GC_TRA_AUTO_STP_PB : BOOL ;	//GUIDE CAGE TRAVEL AUTO STOP PUSH BUTTON
   GC_TRA_FWD_CMD : BOOL ;	//GUIDE CAGE TRAVEL FORWARD COMMAND
   GC_TRA_RET_CMD : BOOL ;	//GUIDE CAGE TRAVEL RETRACT COMMAND
   GC_TRA_FWD_IND : BOOL ;	//GUIDE CAGE TRAVEL FORWARD INDICATOR
   GC_TRA_RET_IND : BOOL ;	//GUIDE CAGE TRAVEL RETRACT INDICATOR
   GC_TRA_AUTO_IND : BOOL ;	//GUIDE CAGE AUTO OPERATION INDICATOR
   GC_TRA_FWD_OP_CUT : BOOL ;	//GUIDE CAGE TRAVEL FORWARD OUTPUT CUT
   GC_TRA_FWD_OP_CUT_TMR : INT ;	//GUIDE CAGE TRAVEL FORWARD OUTPUT CUT TIMER
   GC_TRA_AUTO_FWD_OVR : BOOL ;	//GUIDE CAGE TRAVEL AUTO FORWARD OVER
   GC_TRA_AUTO_FWD_DEL : INT  := 3;	//GUIDE CAGE TRAVEL AUTO FORWARD OVER DELAY
   GC_TRA_AUTO_FWD_DEL_TMR : INT ;	//GUIDE CAGE TRAVEL AUTO FORWARD OVER DELAY TIMER
   GC_TRA_AUTO_FWD_SET : BOOL ;	//GUIDE CAGE AUTO TRAVEL FORWARD SET
   GC_TRA_RET_OP_CUT : BOOL ;	//GUIDE CAGE TRAVEL RETRACT OUTPUT CUT
   GC_TRA_RET_OP_CUT_TMR : INT ;	//GUIDE CAGE TRAVEL RETRACT OUTPUT CUT TIMER
   GC_TRA_AUTO_RET_OVR : BOOL ;	//GUIDE CAGE TRAVEL AUTO RETRACT OVER
   GC_TRA_AUTO_RET_DEL : INT  := 3;	//GUIDE CAGE TRAVEL AUTO RETRACT OVER DELAY
   GC_TRA_AUTO_RET_DEL_TMR : INT ;	//GUIDE CAGE TRAVEL AUTO RETRACT OVER DELAY TIMER
   GC_TRA_AUTO_RET_SET : BOOL ;	//GUIDE CAGE AUTO TRAVEL RETRACT SET
   GC_AUTO_STA_PB : BOOL ;	//GUIDE CAGE AUTO START PUSH BUTTON
   GC_ILK_BIT : BOOL ;	//GUIDE CAGE INTERLOCK BIT
   PULSE_1 : BOOL ;	//PULSE 1
   PULSE_2 : BOOL ;	//PULSE 2
   PULSE_3 : BOOL ;	//PULSE 3
   PULSE_4 : BOOL ;	//PULSE 4
   PULSE_5 : BOOL ;	//PULSE 5
   PULSE_6 : BOOL ;	//PULSE 6
   PULSE_7 : BOOL ;	//PULSE 7
   PULSE_8 : BOOL ;	//PULSE 8
   PULSE_9 : BOOL ;	//PULSE 9
   PULSE_10 : BOOL ;	//PULSE 10
   PULSE_11 : BOOL ;	//PULSE 11
   PULSE_12 : BOOL ;	//PULSE 12
   PULSE_13 : BOOL ;	//PULSE 13
   PULSE_14 : BOOL ;	//PULSE 14
   PULSE_15 : BOOL ;	//PULSE 15
   PULSE_16 : BOOL ;	//PULSE 16
   GC_LOC_SS : BOOL ;	//GUIDE CAGE LOCAL SELECTOR SWITCH
   GC_AUTO_FWD_STA_BIT : BOOL ;	//GUIDE CAGE AUTO FORWARD START BIT
   GC_HME_POS_BIT : BOOL ;	//GUIDE CAGE HOME POSITION BIT
   GC_AUTO_RET_STA_BIT : BOOL ;	//GUIDE CAGE AUTO RETRACT START BIT
   GC_AUTO_OPER_FIN : BOOL ;	//GUIDE CAGE AUTO OPERATIONS FINISHED BIT
   GC_AUTO_OPER_IND : BOOL ;	//GUIDE CAGE AUTO OPERATIONS INDICATOR
   GC_PERM : BOOL ;	//GUIDE CAGE PERMISSION
  END_STRUCT ;	
BEGIN
   GC_TRA_AUTO_FWD_DEL := 3;
   GC_TRA_AUTO_RET_DEL := 3;
END_DATA_BLOCK

